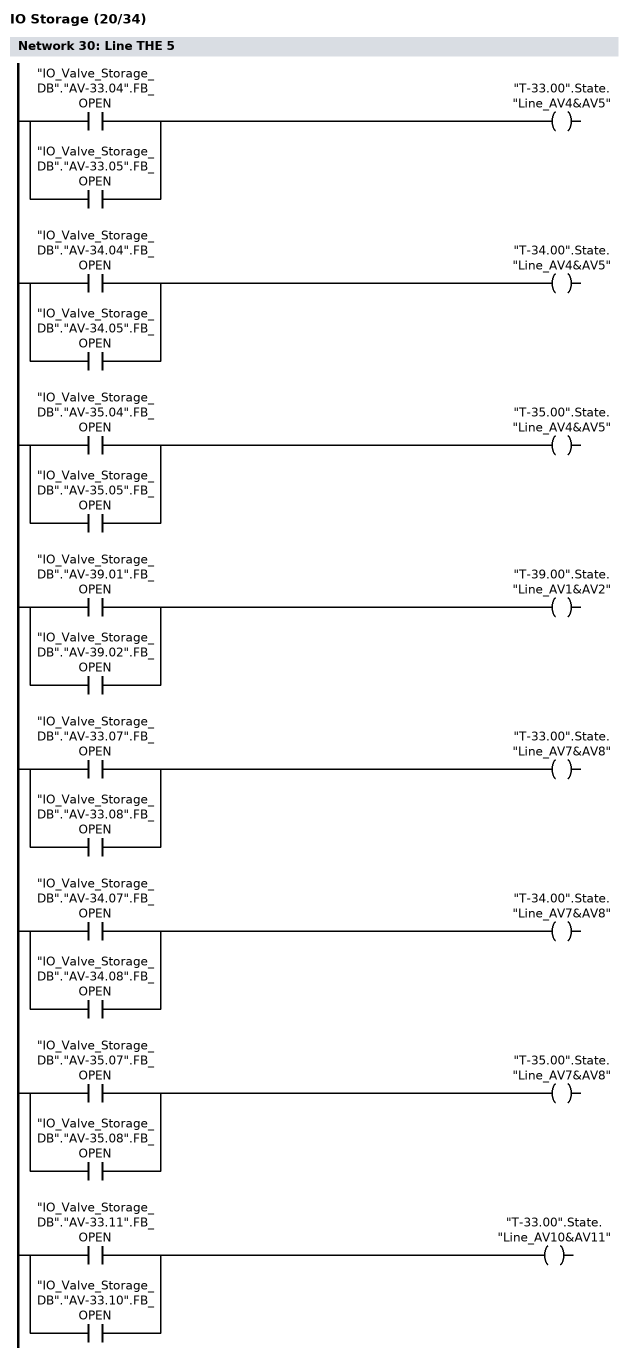
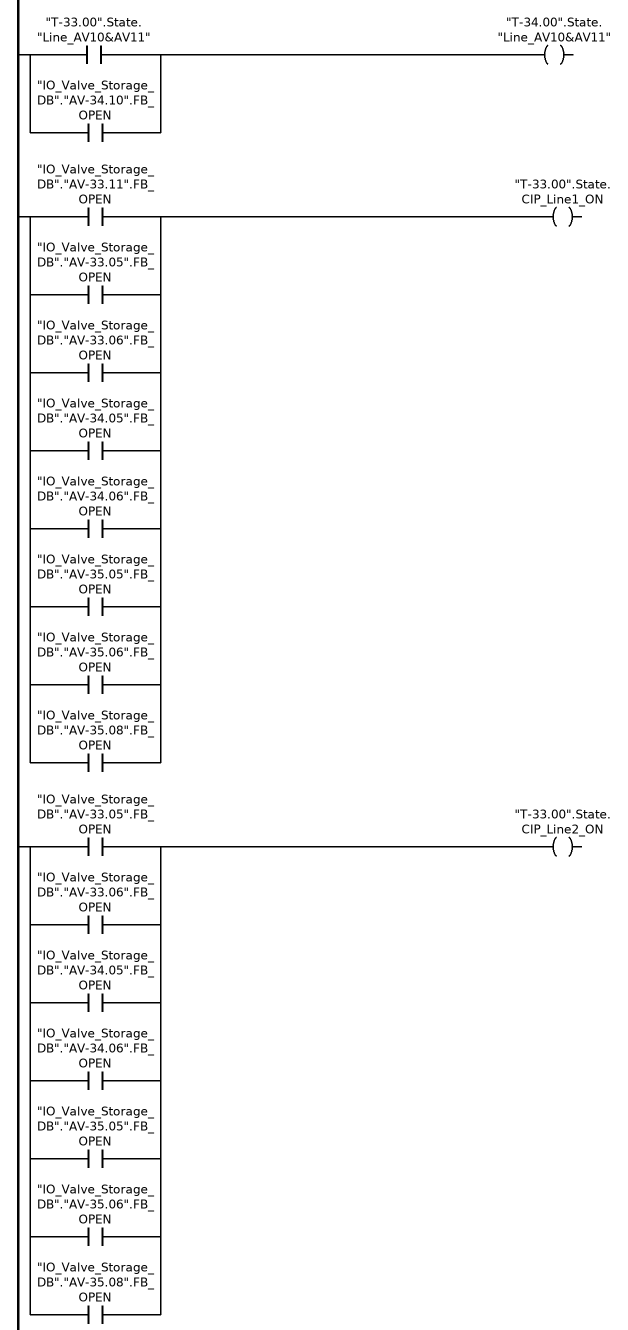
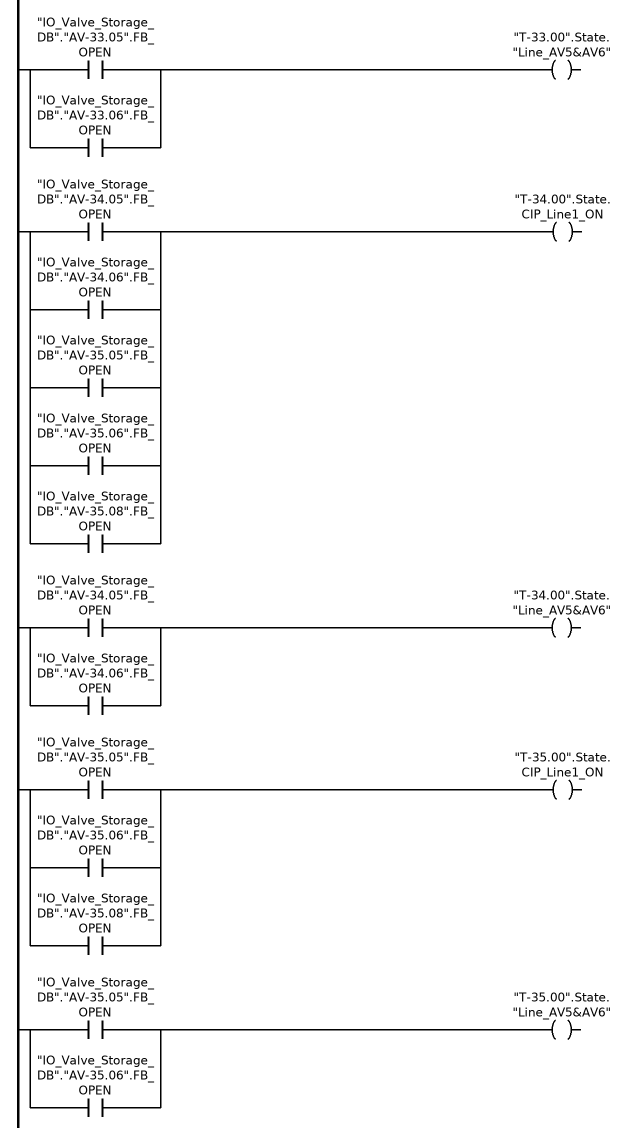
   RUNG wire#powerrail
      Contact( "IO_Valve_Storage_DB"."AV-33.04".FB_OPEN )
      wire#w1
      Coil( "T-33.00".State."Line_AV4&AV5" )
   END_RUNG
   RUNG wire#powerrail
      Contact( "IO_Valve_Storage_DB"."AV-33.05".FB_OPEN )
   END_RUNG wire#w1
   RUNG wire#powerrail
      Contact( "IO_Valve_Storage_DB"."AV-34.04".FB_OPEN )
      wire#w2
      Coil( "T-34.00".State."Line_AV4&AV5" )
   END_RUNG
   RUNG wire#powerrail
      Contact( "IO_Valve_Storage_DB"."AV-34.05".FB_OPEN )
   END_RUNG wire#w2
   RUNG wire#powerrail
      Contact( "IO_Valve_Storage_DB"."AV-35.04".FB_OPEN )
      wire#w3
      Coil( "T-35.00".State."Line_AV4&AV5" )
   END_RUNG
   RUNG wire#powerrail
      Contact( "IO_Valve_Storage_DB"."AV-35.05".FB_OPEN )
   END_RUNG wire#w3
   RUNG wire#powerrail
      Contact( "IO_Valve_Storage_DB"."AV-39.01".FB_OPEN )
      wire#w4
      Coil( "T-39.00".State."Line_AV1&AV2" )
   END_RUNG
   RUNG wire#powerrail
      Contact( "IO_Valve_Storage_DB"."AV-39.02".FB_OPEN )
   END_RUNG wire#w4
   RUNG wire#powerrail
      Contact( "IO_Valve_Storage_DB"."AV-33.07".FB_OPEN )
      wire#w5
      Coil( "T-33.00".State."Line_AV7&AV8" )
   END_RUNG
   RUNG wire#powerrail
      Contact( "IO_Valve_Storage_DB"."AV-33.08".FB_OPEN )
   END_RUNG wire#w5
   RUNG wire#powerrail
      Contact( "IO_Valve_Storage_DB"."AV-34.07".FB_OPEN )
      wire#w6
      Coil( "T-34.00".State."Line_AV7&AV8" )
   END_RUNG
   RUNG wire#powerrail
      Contact( "IO_Valve_Storage_DB"."AV-34.08".FB_OPEN )
   END_RUNG wire#w6
   RUNG wire#powerrail
      Contact( "IO_Valve_Storage_DB"."AV-35.07".FB_OPEN )
      wire#w7
      Coil( "T-35.00".State."Line_AV7&AV8" )
   END_RUNG
   RUNG wire#powerrail
      Contact( "IO_Valve_Storage_DB"."AV-35.08".FB_OPEN )
   END_RUNG wire#w7
   RUNG wire#powerrail
      Contact( "IO_Valve_Storage_DB"."AV-33.11".FB_OPEN )
      wire#w8
      Coil( "T-33.00".State."Line_AV10&AV11" )
   END_RUNG
   RUNG wire#powerrail
      Contact( "IO_Valve_Storage_DB"."AV-33.10".FB_OPEN )
   END_RUNG wire#w8
   RUNG wire#powerrail
      Contact( "T-33.00".State."Line_AV10&AV11" )
      wire#w9
      Coil( "T-34.00".State."Line_AV10&AV11" )
   END_RUNG
   RUNG wire#powerrail
      Contact( "IO_Valve_Storage_DB"."AV-34.10".FB_OPEN )
   END_RUNG wire#w9
   RUNG wire#powerrail
      Contact( "IO_Valve_Storage_DB"."AV-33.11".FB_OPEN )
      wire#w10
      Coil( "T-33.00".State.CIP_Line1_ON )
   END_RUNG
   RUNG wire#powerrail
      Contact( "IO_Valve_Storage_DB"."AV-33.05".FB_OPEN )
   END_RUNG wire#w10
   RUNG wire#powerrail
      Contact( "IO_Valve_Storage_DB"."AV-33.06".FB_OPEN )
   END_RUNG wire#w10
   RUNG wire#powerrail
      Contact( "IO_Valve_Storage_DB"."AV-34.05".FB_OPEN )
   END_RUNG wire#w10
   RUNG wire#powerrail
      Contact( "IO_Valve_Storage_DB"."AV-34.06".FB_OPEN )
   END_RUNG wire#w10
   RUNG wire#powerrail
      Contact( "IO_Valve_Storage_DB"."AV-35.05".FB_OPEN )
   END_RUNG wire#w10
   RUNG wire#powerrail
      Contact( "IO_Valve_Storage_DB"."AV-35.06".FB_OPEN )
   END_RUNG wire#w10
   RUNG wire#powerrail
      Contact( "IO_Valve_Storage_DB"."AV-35.08".FB_OPEN )
   END_RUNG wire#w10
   RUNG wire#powerrail
      Contact( "IO_Valve_Storage_DB"."AV-33.05".FB_OPEN )
      wire#w11
      Coil( "T-33.00".State.CIP_Line2_ON )
   END_RUNG
   RUNG wire#powerrail
      Contact( "IO_Valve_Storage_DB"."AV-33.06".FB_OPEN )
   END_RUNG wire#w11
   RUNG wire#powerrail
      Contact( "IO_Valve_Storage_DB"."AV-34.05".FB_OPEN )
   END_RUNG wire#w11
   RUNG wire#powerrail
      Contact( "IO_Valve_Storage_DB"."AV-34.06".FB_OPEN )
   END_RUNG wire#w11
   RUNG wire#powerrail
      Contact( "IO_Valve_Storage_DB"."AV-35.05".FB_OPEN )
   END_RUNG wire#w11
   RUNG wire#powerrail
      Contact( "IO_Valve_Storage_DB"."AV-35.06".FB_OPEN )
   END_RUNG wire#w11
   RUNG wire#powerrail
      Contact( "IO_Valve_Storage_DB"."AV-35.08".FB_OPEN )
   END_RUNG wire#w11
   RUNG wire#powerrail
      Contact( "IO_Valve_Storage_DB"."AV-33.05".FB_OPEN )
      wire#w12
      Coil( "T-33.00".State."Line_AV5&AV6" )
   END_RUNG
   RUNG wire#powerrail
      Contact( "IO_Valve_Storage_DB"."AV-33.06".FB_OPEN )
   END_RUNG wire#w12
   RUNG wire#powerrail
      Contact( "IO_Valve_Storage_DB"."AV-34.05".FB_OPEN )
      wire#w13
      Coil( "T-34.00".State.CIP_Line1_ON )
   END_RUNG
   RUNG wire#powerrail
      Contact( "IO_Valve_Storage_DB"."AV-34.06".FB_OPEN )
   END_RUNG wire#w13
   RUNG wire#powerrail
      Contact( "IO_Valve_Storage_DB"."AV-35.05".FB_OPEN )
   END_RUNG wire#w13
   RUNG wire#powerrail
      Contact( "IO_Valve_Storage_DB"."AV-35.06".FB_OPEN )
   END_RUNG wire#w13
   RUNG wire#powerrail
      Contact( "IO_Valve_Storage_DB"."AV-35.08".FB_OPEN )
   END_RUNG wire#w13
   RUNG wire#powerrail
      Contact( "IO_Valve_Storage_DB"."AV-34.05".FB_OPEN )
      wire#w14
      Coil( "T-34.00".State."Line_AV5&AV6" )
   END_RUNG
   RUNG wire#powerrail
      Contact( "IO_Valve_Storage_DB"."AV-34.06".FB_OPEN )
   END_RUNG wire#w14
   RUNG wire#powerrail
      Contact( "IO_Valve_Storage_DB"."AV-35.05".FB_OPEN )
      wire#w15
      Coil( "T-35.00".State.CIP_Line1_ON )
   END_RUNG
   RUNG wire#powerrail
      Contact( "IO_Valve_Storage_DB"."AV-35.06".FB_OPEN )
   END_RUNG wire#w15
   RUNG wire#powerrail
      Contact( "IO_Valve_Storage_DB"."AV-35.08".FB_OPEN )
   END_RUNG wire#w15
   RUNG wire#powerrail
      Contact( "IO_Valve_Storage_DB"."AV-35.05".FB_OPEN )
      wire#w16
      Coil( "T-35.00".State."Line_AV5&AV6" )
   END_RUNG
   RUNG wire#powerrail
      Contact( "IO_Valve_Storage_DB"."AV-35.06".FB_OPEN )
   END_RUNG wire#w16
   // the same network as SCL:
   "T-33.00".State."Line_AV4&AV5" := "IO_Valve_Storage_DB"."AV-33.04".FB_OPEN OR "IO_Valve_Storage_DB"."AV-33.05".FB_OPEN;
   "T-34.00".State."Line_AV4&AV5" := "IO_Valve_Storage_DB"."AV-34.04".FB_OPEN OR "IO_Valve_Storage_DB"."AV-34.05".FB_OPEN;
   "T-35.00".State."Line_AV4&AV5" := "IO_Valve_Storage_DB"."AV-35.04".FB_OPEN OR "IO_Valve_Storage_DB"."AV-35.05".FB_OPEN;
   "T-39.00".State."Line_AV1&AV2" := "IO_Valve_Storage_DB"."AV-39.01".FB_OPEN OR "IO_Valve_Storage_DB"."AV-39.02".FB_OPEN;
   "T-33.00".State."Line_AV7&AV8" := "IO_Valve_Storage_DB"."AV-33.07".FB_OPEN OR "IO_Valve_Storage_DB"."AV-33.08".FB_OPEN;
   "T-34.00".State."Line_AV7&AV8" := "IO_Valve_Storage_DB"."AV-34.07".FB_OPEN OR "IO_Valve_Storage_DB"."AV-34.08".FB_OPEN;
   "T-35.00".State."Line_AV7&AV8" := "IO_Valve_Storage_DB"."AV-35.07".FB_OPEN OR "IO_Valve_Storage_DB"."AV-35.08".FB_OPEN;
   "T-33.00".State."Line_AV10&AV11" := "IO_Valve_Storage_DB"."AV-33.11".FB_OPEN OR "IO_Valve_Storage_DB"."AV-33.10".FB_OPEN;
   "T-34.00".State."Line_AV10&AV11" := "T-33.00".State."Line_AV10&AV11" OR "IO_Valve_Storage_DB"."AV-34.10".FB_OPEN;
   "T-33.00".State.CIP_Line1_ON := "IO_Valve_Storage_DB"."AV-33.11".FB_OPEN OR "IO_Valve_Storage_DB"."AV-33.05".FB_OPEN OR "IO_Valve_Storage_DB"."AV-33.06".FB_OPEN OR "IO_Valve_Storage_DB"."AV-34.05".FB_OPEN OR "IO_Valve_Storage_DB"."AV-34.06".FB_OPEN OR "IO_Valve_Storage_DB"."AV-35.05".FB_OPEN OR "IO_Valve_Storage_DB"."AV-35.06".FB_OPEN OR "IO_Valve_Storage_DB"."AV-35.08".FB_OPEN;
   "T-33.00".State.CIP_Line2_ON := "IO_Valve_Storage_DB"."AV-33.05".FB_OPEN OR "IO_Valve_Storage_DB"."AV-33.06".FB_OPEN OR "IO_Valve_Storage_DB"."AV-34.05".FB_OPEN OR "IO_Valve_Storage_DB"."AV-34.06".FB_OPEN OR "IO_Valve_Storage_DB"."AV-35.05".FB_OPEN OR "IO_Valve_Storage_DB"."AV-35.06".FB_OPEN OR "IO_Valve_Storage_DB"."AV-35.08".FB_OPEN;
   "T-33.00".State."Line_AV5&AV6" := "IO_Valve_Storage_DB"."AV-33.05".FB_OPEN OR "IO_Valve_Storage_DB"."AV-33.06".FB_OPEN;
   "T-34.00".State.CIP_Line1_ON := "IO_Valve_Storage_DB"."AV-34.05".FB_OPEN OR "IO_Valve_Storage_DB"."AV-34.06".FB_OPEN OR "IO_Valve_Storage_DB"."AV-35.05".FB_OPEN OR "IO_Valve_Storage_DB"."AV-35.06".FB_OPEN OR "IO_Valve_Storage_DB"."AV-35.08".FB_OPEN;
   "T-34.00".State."Line_AV5&AV6" := "IO_Valve_Storage_DB"."AV-34.05".FB_OPEN OR "IO_Valve_Storage_DB"."AV-34.06".FB_OPEN;
   "T-35.00".State.CIP_Line1_ON := "IO_Valve_Storage_DB"."AV-35.05".FB_OPEN OR "IO_Valve_Storage_DB"."AV-35.06".FB_OPEN OR "IO_Valve_Storage_DB"."AV-35.08".FB_OPEN;
   "T-35.00".State."Line_AV5&AV6" := "IO_Valve_Storage_DB"."AV-35.05".FB_OPEN OR "IO_Valve_Storage_DB"."AV-35.06".FB_OPEN;
END_REGION

REGION Network 32: T-81.00
   // Inload 1 : PHE-2
   // Inload 2 : THE-1
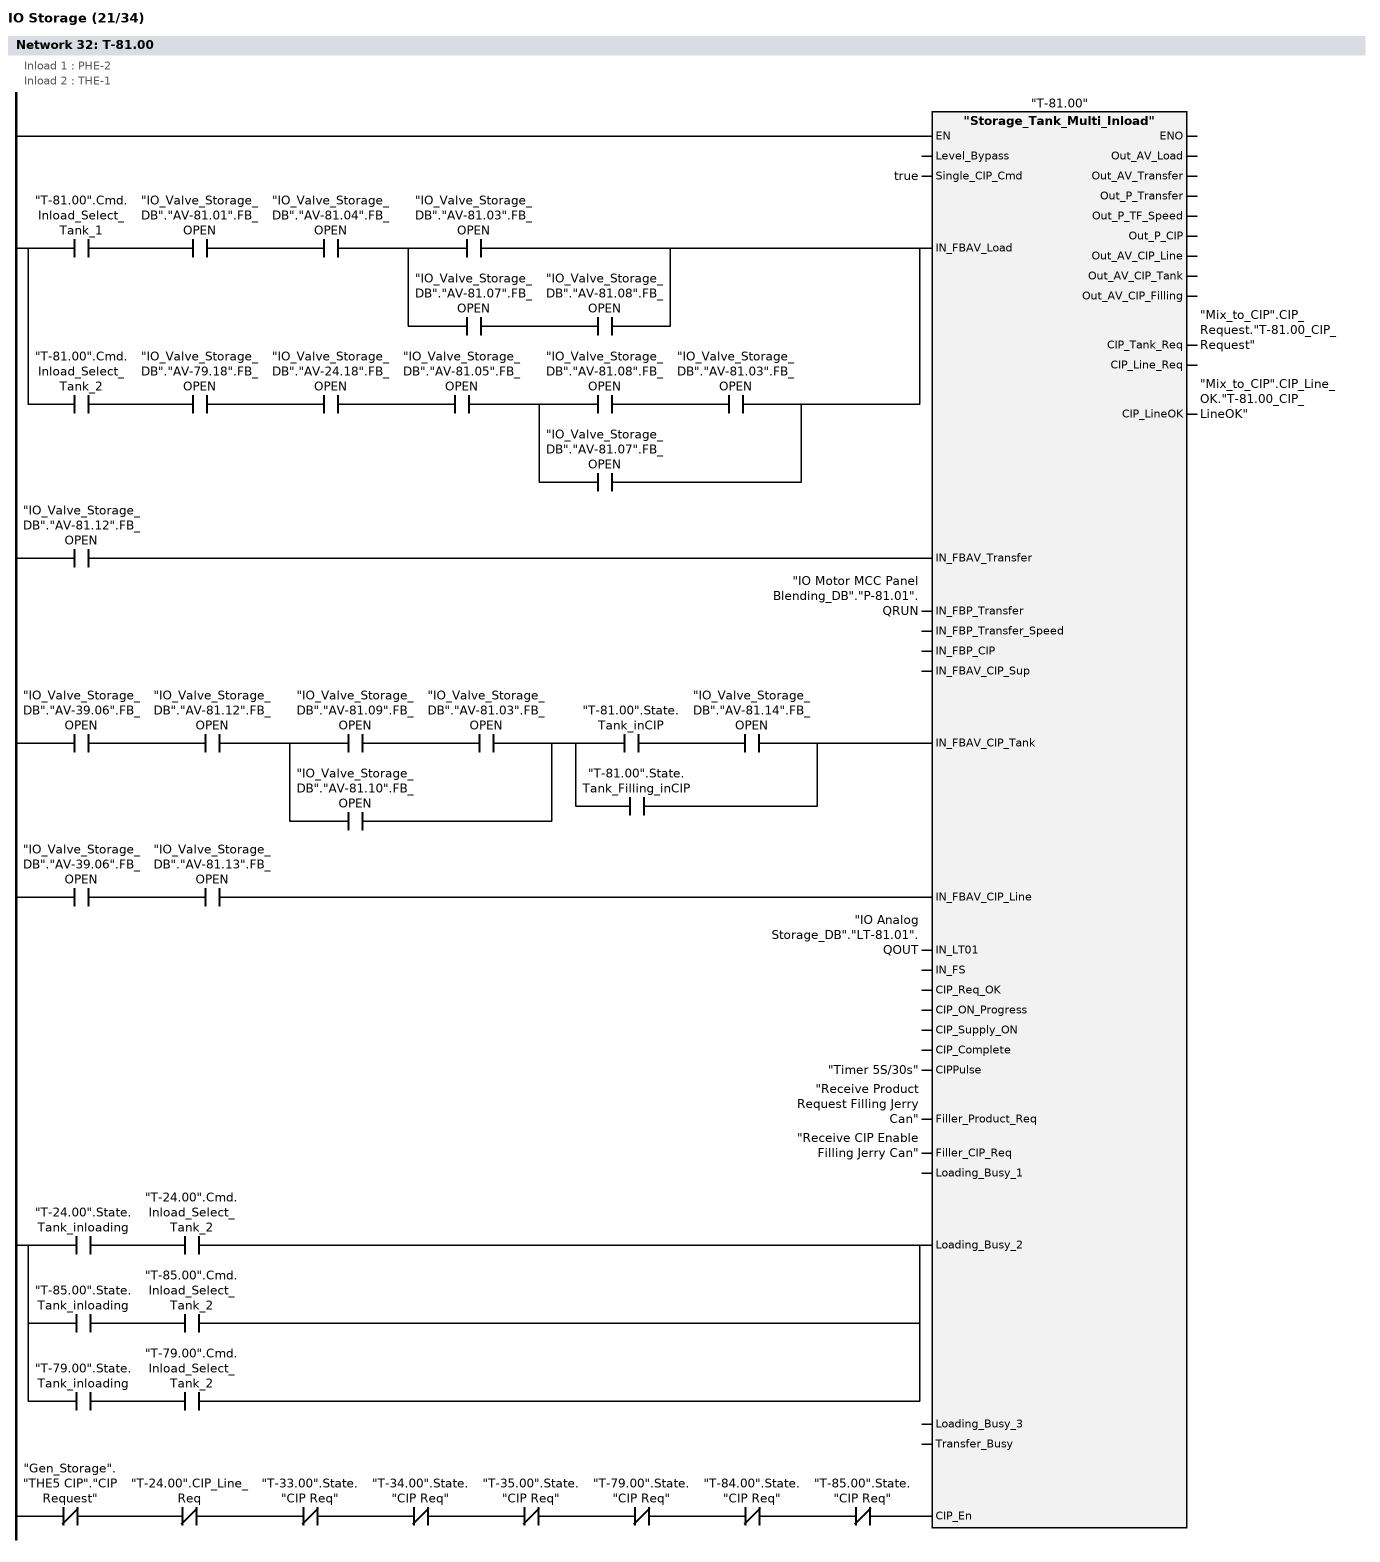
   RUNG wire#powerrail
      "T-81.00"(IN_FBAV_Load := wire#w3, IN_FBAV_Transfer := wire#w4, IN_FBAV_CIP_Tank := wire#w7, IN_FBAV_CIP_Line := wire#w8, Loading_Busy_2 := wire#w9, CIP_En := wire#w10, Level_Bypass :=, Single_CIP_Cmd := true, IN_FBP_Transfer := "IO Motor MCC Panel Blending_DB"."P-81.01".QRUN, IN_FBP_Transfer_Speed :=, IN_FBP_CIP :=, IN_FBAV_CIP_Sup :=, IN_LT01 := "IO Analog Storage_DB"."LT-81.01".QOUT, IN_FS :=, CIP_Req_OK :=, CIP_ON_Progress :=, CIP_Supply_ON :=, CIP_Complete :=, CIPPulse := "Timer 5S/30s", Filler_Product_Req := "Receive Product Request Filling Jerry Can", Filler_CIP_Req := "Receive CIP Enable Filling Jerry Can", Loading_Busy_1 :=, Loading_Busy_3 :=, Transfer_Busy :=, Out_AV_Load =>, Out_AV_Transfer =>, Out_P_Transfer =>, Out_P_TF_Speed =>, Out_P_CIP =>, Out_AV_CIP_Line =>, Out_AV_CIP_Tank =>, Out_AV_CIP_Filling =>, CIP_Tank_Req => "Mix_to_CIP".CIP_Request."T-81.00_CIP_Request", CIP_Line_Req =>, CIP_LineOK => "Mix_to_CIP".CIP_Line_OK."T-81.00_CIP_LineOK")
   END_RUNG
   RUNG wire#powerrail
      Contact( "T-81.00".Cmd.Inload_Select_Tank_1 )
      Contact( "IO_Valve_Storage_DB"."AV-81.01".FB_OPEN )
      Contact( "IO_Valve_Storage_DB"."AV-81.04".FB_OPEN )
      wire#w1
      Contact( "IO_Valve_Storage_DB"."AV-81.03".FB_OPEN )
   END_RUNG wire#w3
   RUNG wire#w1
      Contact( "IO_Valve_Storage_DB"."AV-81.07".FB_OPEN )
      Contact( "IO_Valve_Storage_DB"."AV-81.08".FB_OPEN )
   END_RUNG wire#w3
   RUNG wire#powerrail
      Contact( "T-81.00".Cmd.Inload_Select_Tank_2 )
      Contact( "IO_Valve_Storage_DB"."AV-79.18".FB_OPEN )
      Contact( "IO_Valve_Storage_DB"."AV-24.18".FB_OPEN )
      Contact( "IO_Valve_Storage_DB"."AV-81.05".FB_OPEN )
      wire#w2
      Contact( "IO_Valve_Storage_DB"."AV-81.08".FB_OPEN )
      Contact( "IO_Valve_Storage_DB"."AV-81.03".FB_OPEN )
   END_RUNG wire#w3
   RUNG wire#w2
      Contact( "IO_Valve_Storage_DB"."AV-81.07".FB_OPEN )
   END_RUNG wire#w3
   RUNG wire#powerrail
      Contact( "IO_Valve_Storage_DB"."AV-81.12".FB_OPEN )
   END_RUNG wire#w4
   RUNG wire#powerrail
      Contact( "IO_Valve_Storage_DB"."AV-39.06".FB_OPEN )
      Contact( "IO_Valve_Storage_DB"."AV-81.12".FB_OPEN )
      wire#w5
      Contact( "IO_Valve_Storage_DB"."AV-81.09".FB_OPEN )
      Contact( "IO_Valve_Storage_DB"."AV-81.03".FB_OPEN )
      wire#w6
      Contact( "T-81.00".State.Tank_inCIP )
      Contact( "IO_Valve_Storage_DB"."AV-81.14".FB_OPEN )
   END_RUNG wire#w7
   RUNG wire#w5
      Contact( "IO_Valve_Storage_DB"."AV-81.10".FB_OPEN )
   END_RUNG wire#w6
   RUNG wire#w6
      Contact( "T-81.00".State.Tank_Filling_inCIP )
   END_RUNG wire#w7
   RUNG wire#powerrail
      Contact( "IO_Valve_Storage_DB"."AV-39.06".FB_OPEN )
      Contact( "IO_Valve_Storage_DB"."AV-81.13".FB_OPEN )
   END_RUNG wire#w8
   RUNG wire#powerrail
      Contact( "T-24.00".State.Tank_inloading )
      Contact( "T-24.00".Cmd.Inload_Select_Tank_2 )
   END_RUNG wire#w9
   RUNG wire#powerrail
      Contact( "T-85.00".State.Tank_inloading )
      Contact( "T-85.00".Cmd.Inload_Select_Tank_2 )
   END_RUNG wire#w9
   RUNG wire#powerrail
      Contact( "T-79.00".State.Tank_inloading )
      Contact( "T-79.00".Cmd.Inload_Select_Tank_2 )
   END_RUNG wire#w9
   RUNG wire#powerrail
      I_Contact( "Gen_Storage"."THE5 CIP"."CIP Request" )
      I_Contact( "T-24.00".CIP_Line_Req )
      I_Contact( "T-33.00".State."CIP Req" )
      I_Contact( "T-34.00".State."CIP Req" )
      I_Contact( "T-35.00".State."CIP Req" )
      I_Contact( "T-79.00".State."CIP Req" )
      I_Contact( "T-84.00".State."CIP Req" )
      I_Contact( "T-85.00".State."CIP Req" )
   END_RUNG wire#w10
   // the same network as SCL:
   "T-81.00"(Single_CIP_Cmd := true,   // "Storage_Tank_Multi_Inload"
             IN_FBAV_Load := ("T-81.00".Cmd.Inload_Select_Tank_1 AND "IO_Valve_Storage_DB"."AV-81.01".FB_OPEN AND "IO_Valve_Storage_DB"."AV-81.04".FB_OPEN AND ("IO_Valve_Storage_DB"."AV-81.03".FB_OPEN OR ("IO_Valve_Storage_DB"."AV-81.07".FB_OPEN AND "IO_Valve_Storage_DB"."AV-81.08".FB_OPEN))) OR ("T-81.00".Cmd.Inload_Select_Tank_2 AND "IO_Valve_Storage_DB"."AV-79.18".FB_OPEN AND "IO_Valve_Storage_DB"."AV-24.18".FB_OPEN AND "IO_Valve_Storage_DB"."AV-81.05".FB_OPEN AND (("IO_Valve_Storage_DB"."AV-81.08".FB_OPEN AND "IO_Valve_Storage_DB"."AV-81.03".FB_OPEN) OR "IO_Valve_Storage_DB"."AV-81.07".FB_OPEN)),
             IN_FBAV_Transfer := "IO_Valve_Storage_DB"."AV-81.12".FB_OPEN,
             IN_FBP_Transfer := "IO Motor MCC Panel Blending_DB"."P-81.01".QRUN,
             IN_FBAV_CIP_Tank := "IO_Valve_Storage_DB"."AV-39.06".FB_OPEN AND "IO_Valve_Storage_DB"."AV-81.12".FB_OPEN AND (("IO_Valve_Storage_DB"."AV-81.09".FB_OPEN AND "IO_Valve_Storage_DB"."AV-81.03".FB_OPEN) OR "IO_Valve_Storage_DB"."AV-81.10".FB_OPEN) AND (("T-81.00".State.Tank_inCIP AND "IO_Valve_Storage_DB"."AV-81.14".FB_OPEN) OR "T-81.00".State.Tank_Filling_inCIP),
             IN_FBAV_CIP_Line := "IO_Valve_Storage_DB"."AV-39.06".FB_OPEN AND "IO_Valve_Storage_DB"."AV-81.13".FB_OPEN,
             IN_LT01 := "IO Analog Storage_DB"."LT-81.01".QOUT,
             CIPPulse := "Timer 5S/30s",
             Filler_Product_Req := "Receive Product Request Filling Jerry Can",
             Filler_CIP_Req := "Receive CIP Enable Filling Jerry Can",
             Loading_Busy_2 := ("T-24.00".State.Tank_inloading AND "T-24.00".Cmd.Inload_Select_Tank_2) OR ("T-85.00".State.Tank_inloading AND "T-85.00".Cmd.Inload_Select_Tank_2) OR ("T-79.00".State.Tank_inloading AND "T-79.00".Cmd.Inload_Select_Tank_2),
             CIP_En := NOT "Gen_Storage"."THE5 CIP"."CIP Request" AND NOT "T-24.00".CIP_Line_Req AND NOT "T-33.00".State."CIP Req" AND NOT "T-34.00".State."CIP Req" AND NOT "T-35.00".State."CIP Req" AND NOT "T-79.00".State."CIP Req" AND NOT "T-84.00".State."CIP Req" AND NOT "T-85.00".State."CIP Req",
             CIP_Tank_Req => "Mix_to_CIP".CIP_Request."T-81.00_CIP_Request",
             CIP_LineOK => "Mix_to_CIP".CIP_Line_OK."T-81.00_CIP_LineOK");
END_REGION

REGION Network 33: T-81 Valve
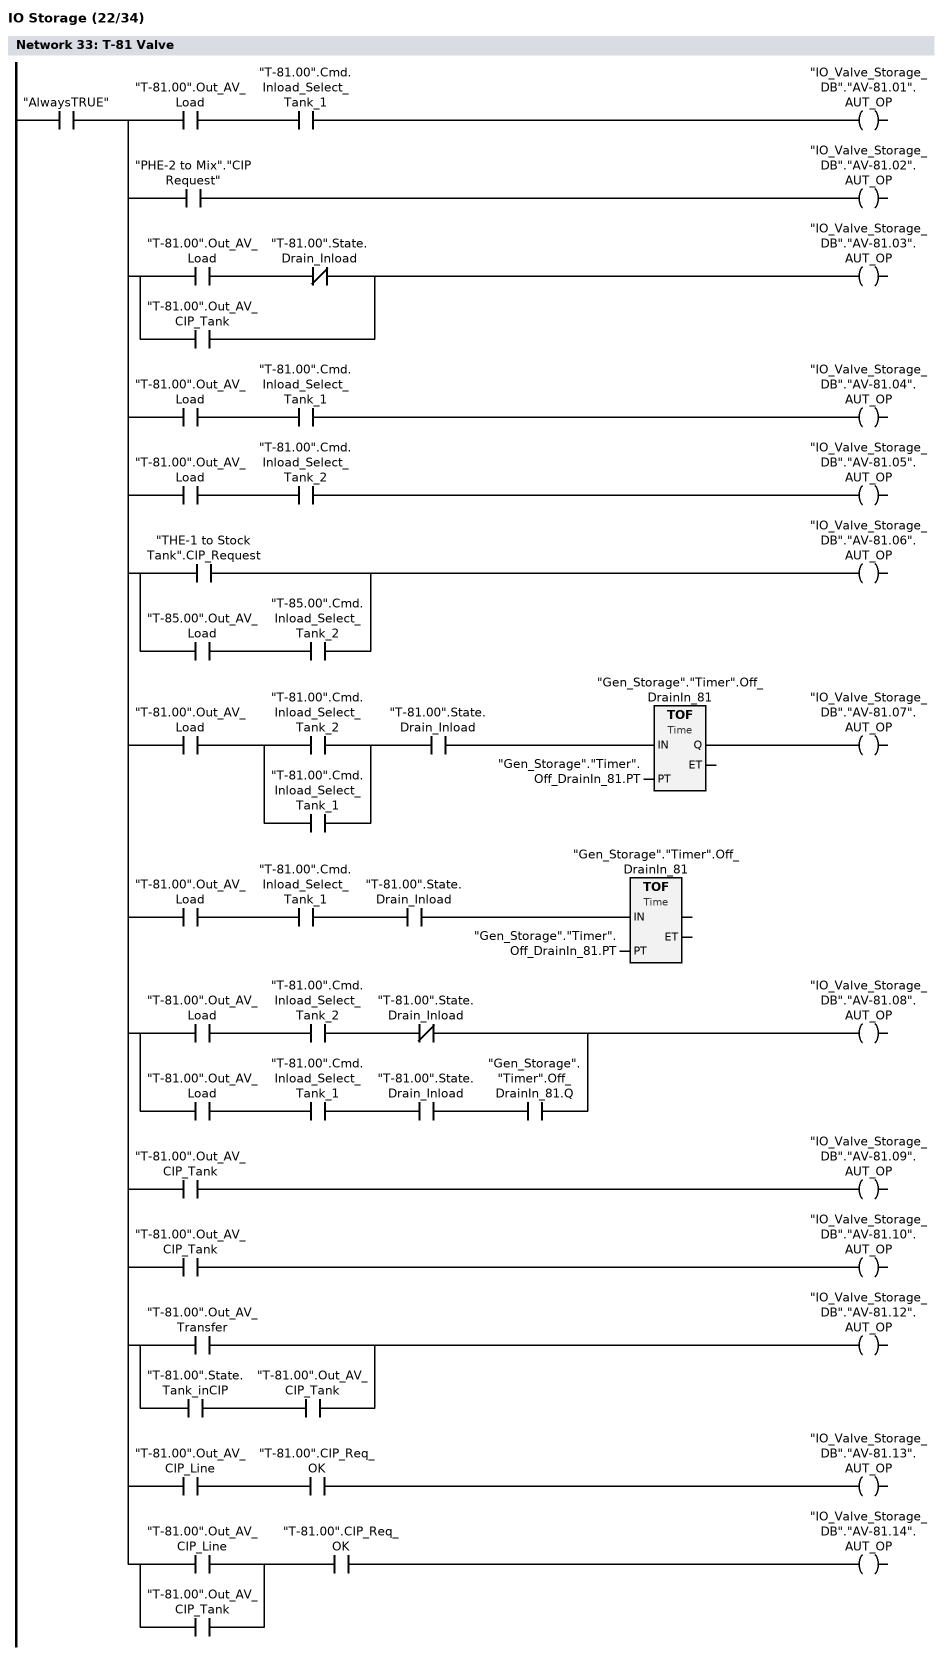
   RUNG wire#powerrail
      Contact( "AlwaysTRUE" )
      wire#w1
      Contact( "T-81.00".Out_AV_Load )
      Contact( "T-81.00".Cmd.Inload_Select_Tank_1 )
      Coil( "IO_Valve_Storage_DB"."AV-81.01".AUT_OP )
   END_RUNG
   RUNG wire#w1
      Contact( "PHE-2 to Mix"."CIP Request" )
      Coil( "IO_Valve_Storage_DB"."AV-81.02".AUT_OP )
   END_RUNG
   RUNG wire#w1
      Contact( "T-81.00".Out_AV_Load )
      I_Contact( "T-81.00".State.Drain_Inload )
      wire#w2
      Coil( "IO_Valve_Storage_DB"."AV-81.03".AUT_OP )
   END_RUNG
   RUNG wire#w1
      Contact( "T-81.00".Out_AV_CIP_Tank )
   END_RUNG wire#w2
   RUNG wire#w1
      Contact( "T-81.00".Out_AV_Load )
      Contact( "T-81.00".Cmd.Inload_Select_Tank_1 )
      Coil( "IO_Valve_Storage_DB"."AV-81.04".AUT_OP )
   END_RUNG
   RUNG wire#w1
      Contact( "T-81.00".Out_AV_Load )
      Contact( "T-81.00".Cmd.Inload_Select_Tank_2 )
      Coil( "IO_Valve_Storage_DB"."AV-81.05".AUT_OP )
   END_RUNG
   RUNG wire#w1
      Contact( "THE-1 to Stock Tank".CIP_Request )
      wire#w3
      Coil( "IO_Valve_Storage_DB"."AV-81.06".AUT_OP )
   END_RUNG
   RUNG wire#w1
      Contact( "T-85.00".Out_AV_Load )
      Contact( "T-85.00".Cmd.Inload_Select_Tank_2 )
   END_RUNG wire#w3
   RUNG wire#w1
      Contact( "T-81.00".Out_AV_Load )
      wire#w4
      Contact( "T-81.00".Cmd.Inload_Select_Tank_2 )
      wire#w5
      Contact( "T-81.00".State.Drain_Inload )
      { S7_Templates := "time_type := Time" } "Gen_Storage"."Timer".Off_DrainIn_81.TOF(pt := "Gen_Storage"."Timer".Off_DrainIn_81.PT, et =>)
      Coil( "IO_Valve_Storage_DB"."AV-81.07".AUT_OP )
   END_RUNG
   RUNG wire#w4
      Contact( "T-81.00".Cmd.Inload_Select_Tank_1 )
   END_RUNG wire#w5
   RUNG wire#w1
      Contact( "T-81.00".Out_AV_Load )
      Contact( "T-81.00".Cmd.Inload_Select_Tank_1 )
      Contact( "T-81.00".State.Drain_Inload )
      { S7_Templates := "time_type := Time" } "Gen_Storage"."Timer".Off_DrainIn_81.TOF(pt := "Gen_Storage"."Timer".Off_DrainIn_81.PT, et =>)
   END_RUNG
   RUNG wire#w1
      Contact( "T-81.00".Out_AV_Load )
      Contact( "T-81.00".Cmd.Inload_Select_Tank_2 )
      I_Contact( "T-81.00".State.Drain_Inload )
      wire#w6
      Coil( "IO_Valve_Storage_DB"."AV-81.08".AUT_OP )
   END_RUNG
   RUNG wire#w1
      Contact( "T-81.00".Out_AV_Load )
      Contact( "T-81.00".Cmd.Inload_Select_Tank_1 )
      Contact( "T-81.00".State.Drain_Inload )
      Contact( "Gen_Storage"."Timer".Off_DrainIn_81.Q )
   END_RUNG wire#w6
   RUNG wire#w1
      Contact( "T-81.00".Out_AV_CIP_Tank )
      Coil( "IO_Valve_Storage_DB"."AV-81.09".AUT_OP )
   END_RUNG
   RUNG wire#w1
      Contact( "T-81.00".Out_AV_CIP_Tank )
      Coil( "IO_Valve_Storage_DB"."AV-81.10".AUT_OP )
   END_RUNG
   RUNG wire#w1
      Contact( "T-81.00".Out_AV_Transfer )
      wire#w7
      Coil( "IO_Valve_Storage_DB"."AV-81.12".AUT_OP )
   END_RUNG
   RUNG wire#w1
      Contact( "T-81.00".State.Tank_inCIP )
      Contact( "T-81.00".Out_AV_CIP_Tank )
   END_RUNG wire#w7
   RUNG wire#w1
      Contact( "T-81.00".Out_AV_CIP_Line )
      Contact( "T-81.00".CIP_Req_OK )
      Coil( "IO_Valve_Storage_DB"."AV-81.13".AUT_OP )
   END_RUNG
   RUNG wire#w1
      Contact( "T-81.00".Out_AV_CIP_Line )
      wire#w8
      Contact( "T-81.00".CIP_Req_OK )
      Coil( "IO_Valve_Storage_DB"."AV-81.14".AUT_OP )
   END_RUNG
   RUNG wire#w1
      Contact( "T-81.00".Out_AV_CIP_Tank )
   END_RUNG wire#w8
   // the same network as SCL:
   "IO_Valve_Storage_DB"."AV-81.01".AUT_OP := "AlwaysTRUE" AND "T-81.00".Out_AV_Load AND "T-81.00".Cmd.Inload_Select_Tank_1;
   "IO_Valve_Storage_DB"."AV-81.02".AUT_OP := "AlwaysTRUE" AND "PHE-2 to Mix"."CIP Request";
   "IO_Valve_Storage_DB"."AV-81.03".AUT_OP := "AlwaysTRUE" AND (("T-81.00".Out_AV_Load AND NOT "T-81.00".State.Drain_Inload) OR "T-81.00".Out_AV_CIP_Tank);
   "IO_Valve_Storage_DB"."AV-81.04".AUT_OP := "AlwaysTRUE" AND "T-81.00".Out_AV_Load AND "T-81.00".Cmd.Inload_Select_Tank_1;
   "IO_Valve_Storage_DB"."AV-81.05".AUT_OP := "AlwaysTRUE" AND "T-81.00".Out_AV_Load AND "T-81.00".Cmd.Inload_Select_Tank_2;
   "IO_Valve_Storage_DB"."AV-81.06".AUT_OP := "AlwaysTRUE" AND ("THE-1 to Stock Tank".CIP_Request OR ("T-85.00".Out_AV_Load AND "T-85.00".Cmd.Inload_Select_Tank_2));
   "Gen_Storage"."Timer".Off_DrainIn_81.TOF(IN := "AlwaysTRUE" AND "T-81.00".Out_AV_Load AND ("T-81.00".Cmd.Inload_Select_Tank_2 OR "T-81.00".Cmd.Inload_Select_Tank_1) AND "T-81.00".State.Drain_Inload,
                           PT := "Gen_Storage"."Timer".Off_DrainIn_81.PT);
   "IO_Valve_Storage_DB"."AV-81.07".AUT_OP := "Gen_Storage"."Timer".Off_DrainIn_81.Q;
   "Gen_Storage"."Timer".Off_DrainIn_81.TOF(IN := "AlwaysTRUE" AND "T-81.00".Out_AV_Load AND "T-81.00".Cmd.Inload_Select_Tank_1 AND "T-81.00".State.Drain_Inload,
                           PT := "Gen_Storage"."Timer".Off_DrainIn_81.PT);
   "IO_Valve_Storage_DB"."AV-81.08".AUT_OP := "AlwaysTRUE" AND (("T-81.00".Out_AV_Load AND "T-81.00".Cmd.Inload_Select_Tank_2 AND NOT "T-81.00".State.Drain_Inload) OR ("T-81.00".Out_AV_Load AND "T-81.00".Cmd.Inload_Select_Tank_1 AND "T-81.00".State.Drain_Inload AND "Gen_Storage"."Timer".Off_DrainIn_81.Q));
   "IO_Valve_Storage_DB"."AV-81.09".AUT_OP := "AlwaysTRUE" AND "T-81.00".Out_AV_CIP_Tank;
   "IO_Valve_Storage_DB"."AV-81.10".AUT_OP := "AlwaysTRUE" AND "T-81.00".Out_AV_CIP_Tank;
   "IO_Valve_Storage_DB"."AV-81.12".AUT_OP := "AlwaysTRUE" AND ("T-81.00".Out_AV_Transfer OR ("T-81.00".State.Tank_inCIP AND "T-81.00".Out_AV_CIP_Tank));
   "IO_Valve_Storage_DB"."AV-81.13".AUT_OP := "AlwaysTRUE" AND "T-81.00".Out_AV_CIP_Line AND "T-81.00".CIP_Req_OK;
   "IO_Valve_Storage_DB"."AV-81.14".AUT_OP := "AlwaysTRUE" AND ("T-81.00".Out_AV_CIP_Line OR "T-81.00".Out_AV_CIP_Tank) AND "T-81.00".CIP_Req_OK;
END_REGION

REGION Network 34: Comm T-81 to THE-1
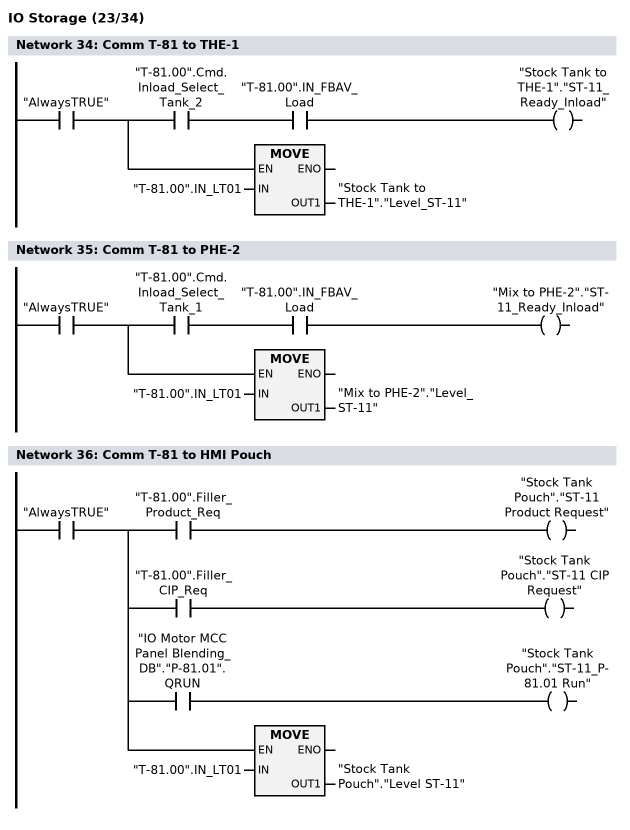
   RUNG wire#powerrail
      Contact( "AlwaysTRUE" )
      wire#w1
      Contact( "T-81.00".Cmd.Inload_Select_Tank_2 )
      Contact( "T-81.00".IN_FBAV_Load )
      Coil( "Stock Tank to THE-1"."ST-11_Ready_Inload" )
   END_RUNG
   RUNG wire#w1
      Move(in := "T-81.00".IN_LT01, out1 => "Stock Tank to THE-1"."Level_ST-11")
   END_RUNG
   // the same network as SCL:
   "Stock Tank to THE-1"."ST-11_Ready_Inload" := "AlwaysTRUE" AND "T-81.00".Cmd.Inload_Select_Tank_2 AND "T-81.00".IN_FBAV_Load;
   IF "AlwaysTRUE" THEN "Stock Tank to THE-1"."Level_ST-11" := "T-81.00".IN_LT01; END_IF;
END_REGION

REGION Network 35: Comm T-81 to PHE-2
   RUNG wire#powerrail
      Contact( "AlwaysTRUE" )
      wire#w1
      Contact( "T-81.00".Cmd.Inload_Select_Tank_1 )
      Contact( "T-81.00".IN_FBAV_Load )
      Coil( "Mix to PHE-2"."ST-11_Ready_Inload" )
   END_RUNG
   RUNG wire#w1
      Move(in := "T-81.00".IN_LT01, out1 => "Mix to PHE-2"."Level_ST-11")
   END_RUNG
   // the same network as SCL:
   "Mix to PHE-2"."ST-11_Ready_Inload" := "AlwaysTRUE" AND "T-81.00".Cmd.Inload_Select_Tank_1 AND "T-81.00".IN_FBAV_Load;
   IF "AlwaysTRUE" THEN "Mix to PHE-2"."Level_ST-11" := "T-81.00".IN_LT01; END_IF;
END_REGION

REGION Network 36: Comm T-81 to HMI Pouch
   RUNG wire#powerrail
      Contact( "AlwaysTRUE" )
      wire#w1
      Contact( "T-81.00".Filler_Product_Req )
      Coil( "Stock Tank Pouch"."ST-11 Product Request" )
   END_RUNG
   RUNG wire#w1
      Contact( "T-81.00".Filler_CIP_Req )
      Coil( "Stock Tank Pouch"."ST-11 CIP Request" )
   END_RUNG
   RUNG wire#w1
      Contact( "IO Motor MCC Panel Blending_DB"."P-81.01".QRUN )
      Coil( "Stock Tank Pouch"."ST-11_P-81.01 Run" )
   END_RUNG
   RUNG wire#w1
      Move(in := "T-81.00".IN_LT01, out1 => "Stock Tank Pouch"."Level ST-11")
   END_RUNG
   // the same network as SCL:
   "Stock Tank Pouch"."ST-11 Product Request" := "AlwaysTRUE" AND "T-81.00".Filler_Product_Req;
   "Stock Tank Pouch"."ST-11 CIP Request" := "AlwaysTRUE" AND "T-81.00".Filler_CIP_Req;
   "Stock Tank Pouch"."ST-11_P-81.01 Run" := "AlwaysTRUE" AND "IO Motor MCC Panel Blending_DB"."P-81.01".QRUN;
   IF "AlwaysTRUE" THEN "Stock Tank Pouch"."Level ST-11" := "T-81.00".IN_LT01; END_IF;
END_REGION

REGION Network 38: T-85.00 ST-16
   // Inload 1 : PHE-1
   // Inload 2 : THE-1
   // Inload 3 : THE-3
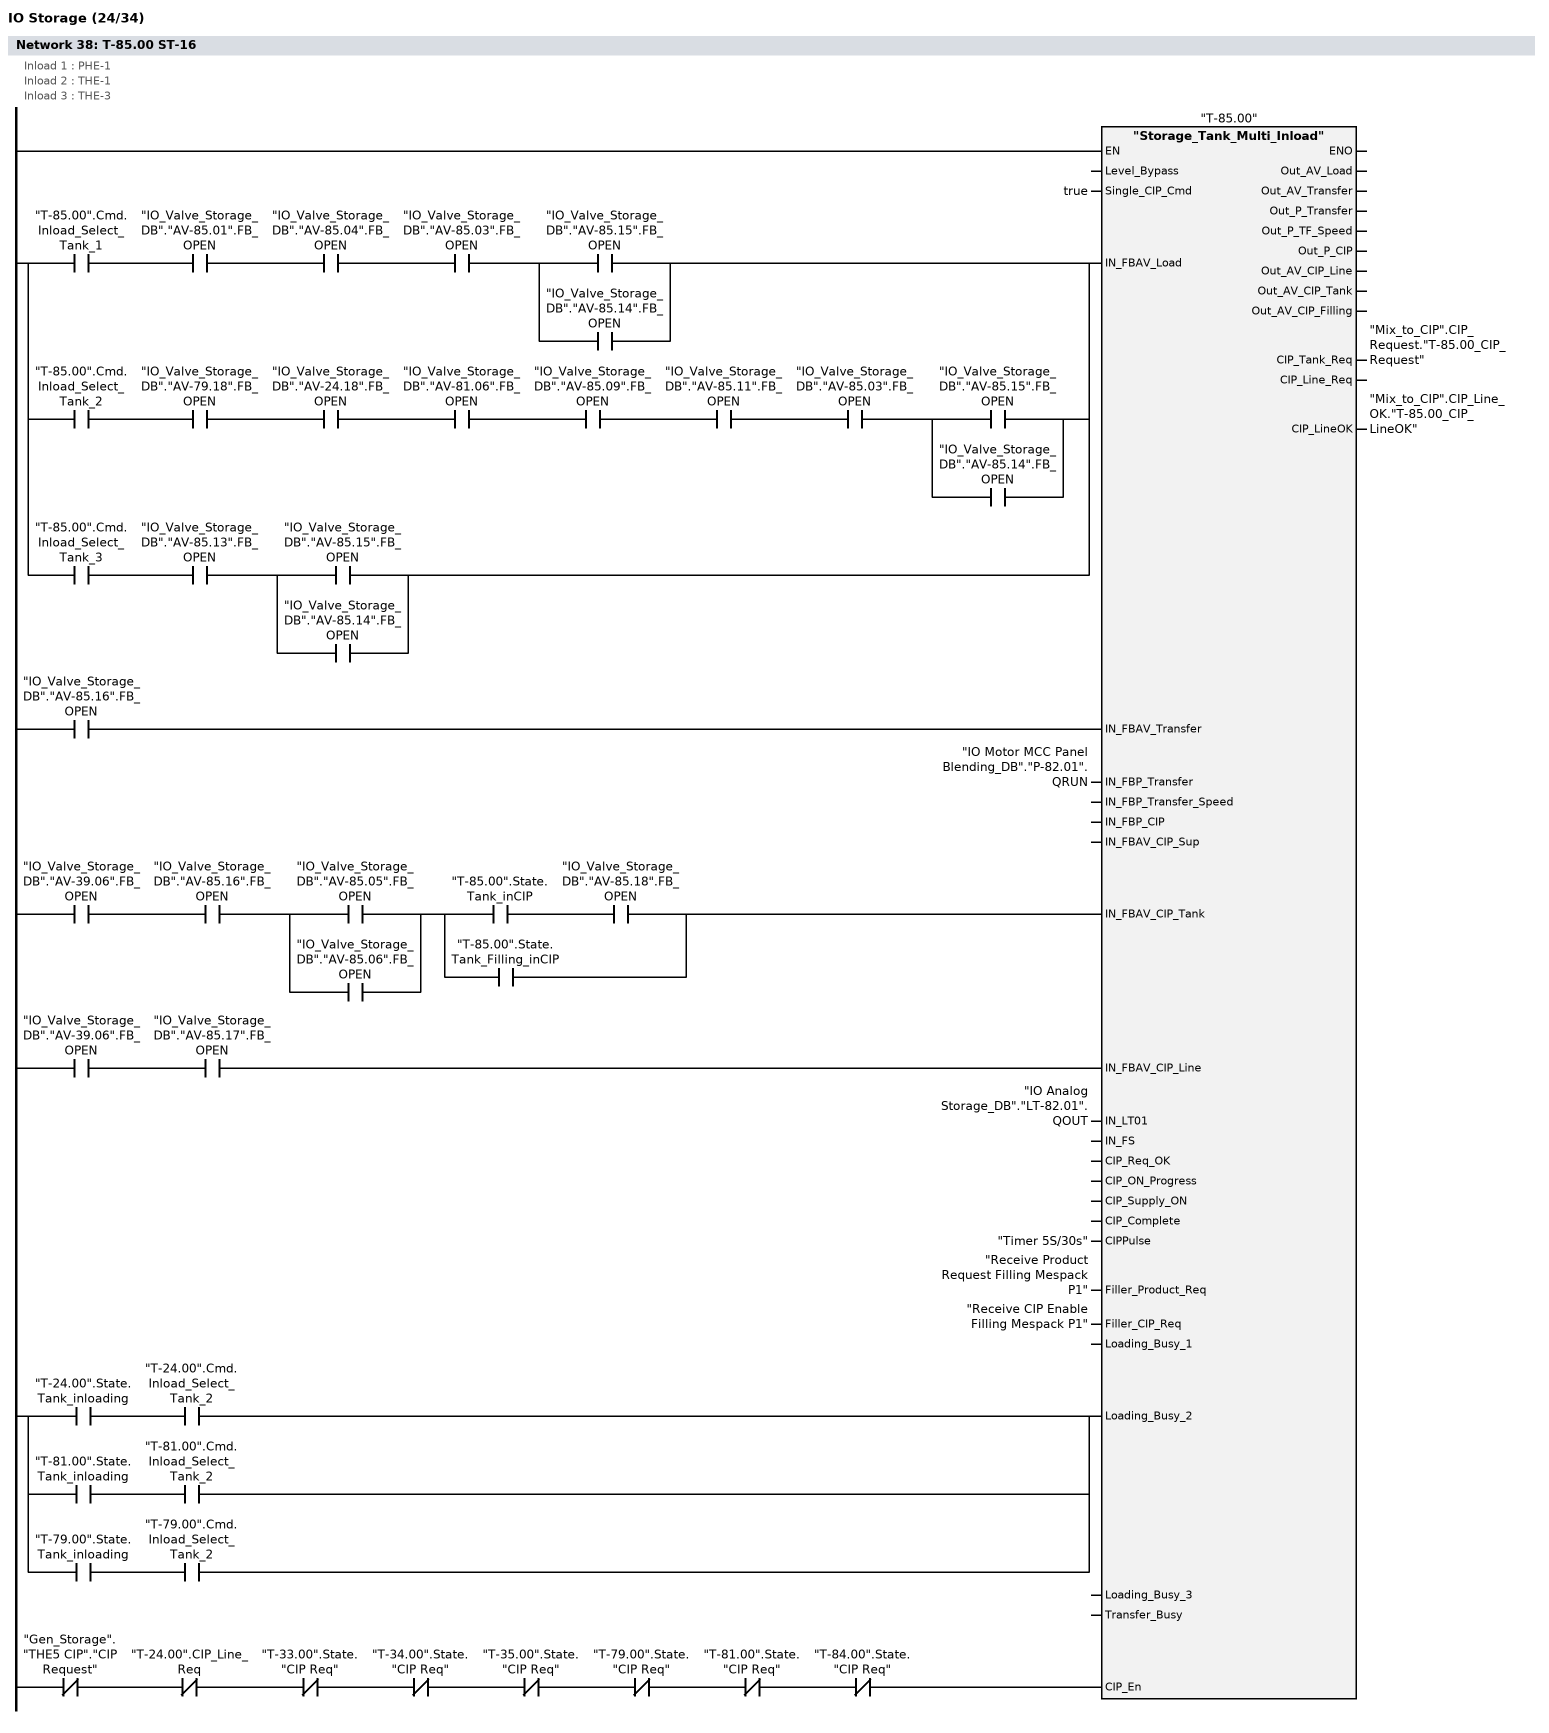
   RUNG wire#powerrail
      "T-85.00"(IN_FBAV_Load := wire#w4, IN_FBAV_Transfer := wire#w5, IN_FBAV_CIP_Tank := wire#w8, IN_FBAV_CIP_Line := wire#w9, Loading_Busy_2 := wire#w10, CIP_En := wire#w11, Level_Bypass :=, Single_CIP_Cmd := true, IN_FBP_Transfer := "IO Motor MCC Panel Blending_DB"."P-82.01".QRUN, IN_FBP_Transfer_Speed :=, IN_FBP_CIP :=, IN_FBAV_CIP_Sup :=, IN_LT01 := "IO Analog Storage_DB"."LT-82.01".QOUT, IN_FS :=, CIP_Req_OK :=, CIP_ON_Progress :=, CIP_Supply_ON :=, CIP_Complete :=, CIPPulse := "Timer 5S/30s", Filler_Product_Req := "Receive Product Request Filling Mespack P1", Filler_CIP_Req := "Receive CIP Enable Filling Mespack P1", Loading_Busy_1 :=, Loading_Busy_3 :=, Transfer_Busy :=, Out_AV_Load =>, Out_AV_Transfer =>, Out_P_Transfer =>, Out_P_TF_Speed =>, Out_P_CIP =>, Out_AV_CIP_Line =>, Out_AV_CIP_Tank =>, Out_AV_CIP_Filling =>, CIP_Tank_Req => "Mix_to_CIP".CIP_Request."T-85.00_CIP_Request", CIP_Line_Req =>, CIP_LineOK => "Mix_to_CIP".CIP_Line_OK."T-85.00_CIP_LineOK")
   END_RUNG
   RUNG wire#powerrail
      Contact( "T-85.00".Cmd.Inload_Select_Tank_1 )
      Contact( "IO_Valve_Storage_DB"."AV-85.01".FB_OPEN )
      Contact( "IO_Valve_Storage_DB"."AV-85.04".FB_OPEN )
      Contact( "IO_Valve_Storage_DB"."AV-85.03".FB_OPEN )
      wire#w1
      Contact( "IO_Valve_Storage_DB"."AV-85.15".FB_OPEN )
   END_RUNG wire#w4
   RUNG wire#w1
      Contact( "IO_Valve_Storage_DB"."AV-85.14".FB_OPEN )
   END_RUNG wire#w4
   RUNG wire#powerrail
      Contact( "T-85.00".Cmd.Inload_Select_Tank_2 )
      Contact( "IO_Valve_Storage_DB"."AV-79.18".FB_OPEN )
      Contact( "IO_Valve_Storage_DB"."AV-24.18".FB_OPEN )
      Contact( "IO_Valve_Storage_DB"."AV-81.06".FB_OPEN )
      Contact( "IO_Valve_Storage_DB"."AV-85.09".FB_OPEN )
      Contact( "IO_Valve_Storage_DB"."AV-85.11".FB_OPEN )
      Contact( "IO_Valve_Storage_DB"."AV-85.03".FB_OPEN )
      wire#w2
      Contact( "IO_Valve_Storage_DB"."AV-85.15".FB_OPEN )
   END_RUNG wire#w4
   RUNG wire#w2
      Contact( "IO_Valve_Storage_DB"."AV-85.14".FB_OPEN )
   END_RUNG wire#w4
   RUNG wire#powerrail
      Contact( "T-85.00".Cmd.Inload_Select_Tank_3 )
      Contact( "IO_Valve_Storage_DB"."AV-85.13".FB_OPEN )
      wire#w3
      Contact( "IO_Valve_Storage_DB"."AV-85.15".FB_OPEN )
   END_RUNG wire#w4
   RUNG wire#w3
      Contact( "IO_Valve_Storage_DB"."AV-85.14".FB_OPEN )
   END_RUNG wire#w4
   RUNG wire#powerrail
      Contact( "IO_Valve_Storage_DB"."AV-85.16".FB_OPEN )
   END_RUNG wire#w5
   RUNG wire#powerrail
      Contact( "IO_Valve_Storage_DB"."AV-39.06".FB_OPEN )
      Contact( "IO_Valve_Storage_DB"."AV-85.16".FB_OPEN )
      wire#w6
      Contact( "IO_Valve_Storage_DB"."AV-85.05".FB_OPEN )
      wire#w7
      Contact( "T-85.00".State.Tank_inCIP )
      Contact( "IO_Valve_Storage_DB"."AV-85.18".FB_OPEN )
   END_RUNG wire#w8
   RUNG wire#w6
      Contact( "IO_Valve_Storage_DB"."AV-85.06".FB_OPEN )
   END_RUNG wire#w7
   RUNG wire#w7
      Contact( "T-85.00".State.Tank_Filling_inCIP )
   END_RUNG wire#w8
   RUNG wire#powerrail
      Contact( "IO_Valve_Storage_DB"."AV-39.06".FB_OPEN )
      Contact( "IO_Valve_Storage_DB"."AV-85.17".FB_OPEN )
   END_RUNG wire#w9
   RUNG wire#powerrail
      Contact( "T-24.00".State.Tank_inloading )
      Contact( "T-24.00".Cmd.Inload_Select_Tank_2 )
   END_RUNG wire#w10
   RUNG wire#powerrail
      Contact( "T-81.00".State.Tank_inloading )
      Contact( "T-81.00".Cmd.Inload_Select_Tank_2 )
   END_RUNG wire#w10
   RUNG wire#powerrail
      Contact( "T-79.00".State.Tank_inloading )
      Contact( "T-79.00".Cmd.Inload_Select_Tank_2 )
   END_RUNG wire#w10
   RUNG wire#powerrail
      I_Contact( "Gen_Storage"."THE5 CIP"."CIP Request" )
      I_Contact( "T-24.00".CIP_Line_Req )
      I_Contact( "T-33.00".State."CIP Req" )
      I_Contact( "T-34.00".State."CIP Req" )
      I_Contact( "T-35.00".State."CIP Req" )
      I_Contact( "T-79.00".State."CIP Req" )
      I_Contact( "T-81.00".State."CIP Req" )
      I_Contact( "T-84.00".State."CIP Req" )
   END_RUNG wire#w11
   // the same network as SCL:
   "T-85.00"(Single_CIP_Cmd := true,   // "Storage_Tank_Multi_Inload"
             IN_FBAV_Load := ("T-85.00".Cmd.Inload_Select_Tank_1 AND "IO_Valve_Storage_DB"."AV-85.01".FB_OPEN AND "IO_Valve_Storage_DB"."AV-85.04".FB_OPEN AND "IO_Valve_Storage_DB"."AV-85.03".FB_OPEN AND ("IO_Valve_Storage_DB"."AV-85.15".FB_OPEN OR "IO_Valve_Storage_DB"."AV-85.14".FB_OPEN)) OR ("T-85.00".Cmd.Inload_Select_Tank_2 AND "IO_Valve_Storage_DB"."AV-79.18".FB_OPEN AND "IO_Valve_Storage_DB"."AV-24.18".FB_OPEN AND "IO_Valve_Storage_DB"."AV-81.06".FB_OPEN AND "IO_Valve_Storage_DB"."AV-85.09".FB_OPEN AND "IO_Valve_Storage_DB"."AV-85.11".FB_OPEN AND "IO_Valve_Storage_DB"."AV-85.03".FB_OPEN AND ("IO_Valve_Storage_DB"."AV-85.15".FB_OPEN OR "IO_Valve_Storage_DB"."AV-85.14".FB_OPEN)) OR ("T-85.00".Cmd.Inload_Select_Tank_3 AND "IO_Valve_Storage_DB"."AV-85.13".FB_OPEN AND ("IO_Valve_Storage_DB"."AV-85.15".FB_OPEN OR "IO_Valve_Storage_DB"."AV-85.14".FB_OPEN)),
             IN_FBAV_Transfer := "IO_Valve_Storage_DB"."AV-85.16".FB_OPEN,
             IN_FBP_Transfer := "IO Motor MCC Panel Blending_DB"."P-82.01".QRUN,
             IN_FBAV_CIP_Tank := "IO_Valve_Storage_DB"."AV-39.06".FB_OPEN AND "IO_Valve_Storage_DB"."AV-85.16".FB_OPEN AND ("IO_Valve_Storage_DB"."AV-85.05".FB_OPEN OR "IO_Valve_Storage_DB"."AV-85.06".FB_OPEN) AND (("T-85.00".State.Tank_inCIP AND "IO_Valve_Storage_DB"."AV-85.18".FB_OPEN) OR "T-85.00".State.Tank_Filling_inCIP),
             IN_FBAV_CIP_Line := "IO_Valve_Storage_DB"."AV-39.06".FB_OPEN AND "IO_Valve_Storage_DB"."AV-85.17".FB_OPEN,
             IN_LT01 := "IO Analog Storage_DB"."LT-82.01".QOUT,
             CIPPulse := "Timer 5S/30s",
             Filler_Product_Req := "Receive Product Request Filling Mespack P1",
             Filler_CIP_Req := "Receive CIP Enable Filling Mespack P1",
             Loading_Busy_2 := ("T-24.00".State.Tank_inloading AND "T-24.00".Cmd.Inload_Select_Tank_2) OR ("T-81.00".State.Tank_inloading AND "T-81.00".Cmd.Inload_Select_Tank_2) OR ("T-79.00".State.Tank_inloading AND "T-79.00".Cmd.Inload_Select_Tank_2),
             CIP_En := NOT "Gen_Storage"."THE5 CIP"."CIP Request" AND NOT "T-24.00".CIP_Line_Req AND NOT "T-33.00".State."CIP Req" AND NOT "T-34.00".State."CIP Req" AND NOT "T-35.00".State."CIP Req" AND NOT "T-79.00".State."CIP Req" AND NOT "T-81.00".State."CIP Req" AND NOT "T-84.00".State."CIP Req",
             CIP_Tank_Req => "Mix_to_CIP".CIP_Request."T-85.00_CIP_Request",
             CIP_LineOK => "Mix_to_CIP".CIP_Line_OK."T-85.00_CIP_LineOK");
END_REGION

REGION Network 39: T-85 Valve
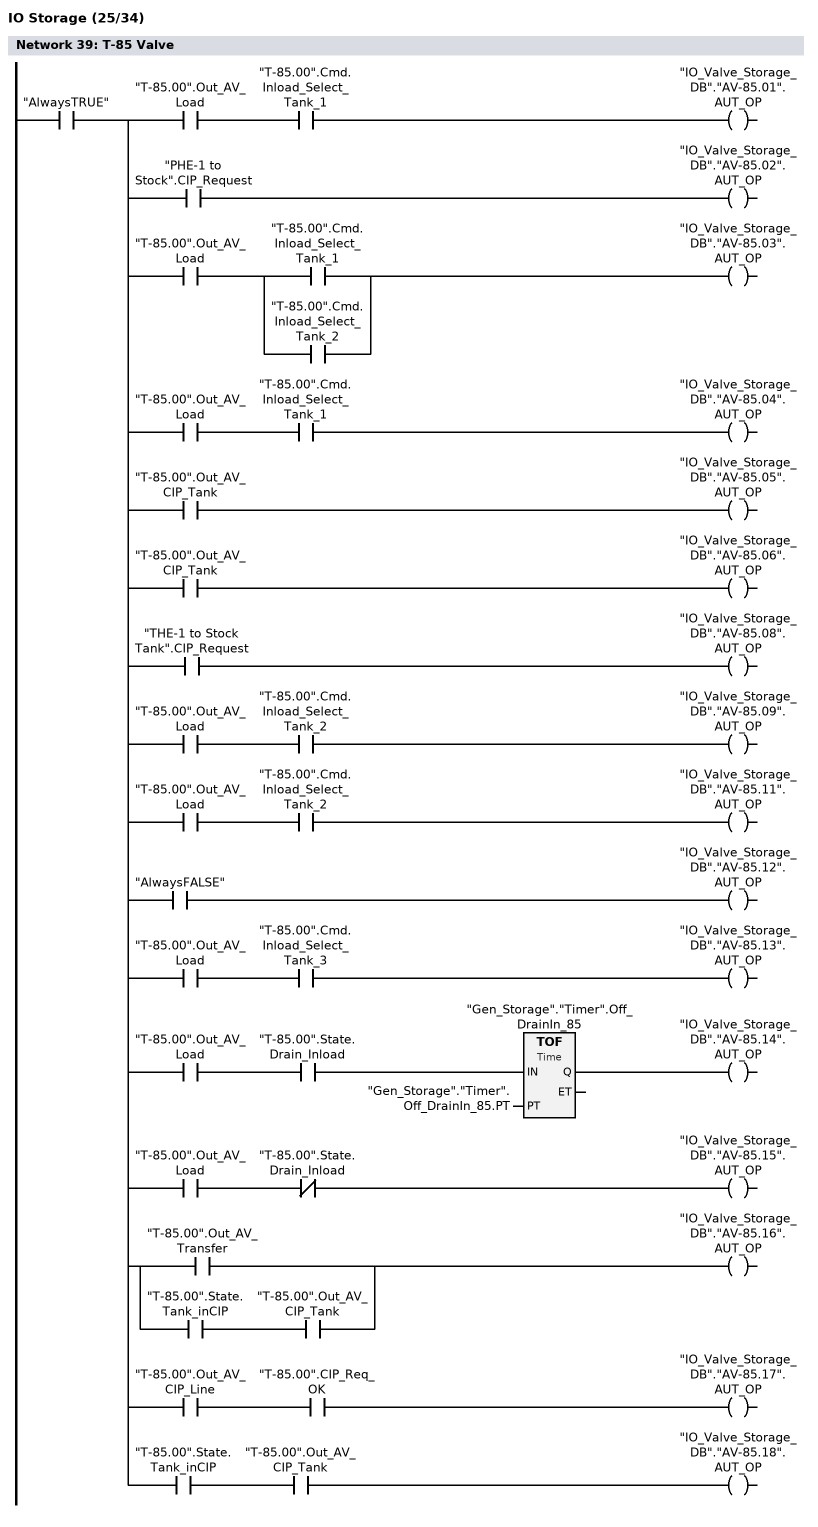
   RUNG wire#powerrail
      Contact( "AlwaysTRUE" )
      wire#w1
      Contact( "T-85.00".Out_AV_Load )
      Contact( "T-85.00".Cmd.Inload_Select_Tank_1 )
      Coil( "IO_Valve_Storage_DB"."AV-85.01".AUT_OP )
   END_RUNG
   RUNG wire#w1
      Contact( "PHE-1 to Stock".CIP_Request )
      Coil( "IO_Valve_Storage_DB"."AV-85.02".AUT_OP )
   END_RUNG
   RUNG wire#w1
      Contact( "T-85.00".Out_AV_Load )
      wire#w2
      Contact( "T-85.00".Cmd.Inload_Select_Tank_1 )
      wire#w3
      Coil( "IO_Valve_Storage_DB"."AV-85.03".AUT_OP )
   END_RUNG
   RUNG wire#w2
      Contact( "T-85.00".Cmd.Inload_Select_Tank_2 )
   END_RUNG wire#w3
   RUNG wire#w1
      Contact( "T-85.00".Out_AV_Load )
      Contact( "T-85.00".Cmd.Inload_Select_Tank_1 )
      Coil( "IO_Valve_Storage_DB"."AV-85.04".AUT_OP )
   END_RUNG
   RUNG wire#w1
      Contact( "T-85.00".Out_AV_CIP_Tank )
      Coil( "IO_Valve_Storage_DB"."AV-85.05".AUT_OP )
   END_RUNG
   RUNG wire#w1
      Contact( "T-85.00".Out_AV_CIP_Tank )
      Coil( "IO_Valve_Storage_DB"."AV-85.06".AUT_OP )
   END_RUNG
   RUNG wire#w1
      Contact( "THE-1 to Stock Tank".CIP_Request )
      Coil( "IO_Valve_Storage_DB"."AV-85.08".AUT_OP )
   END_RUNG
   RUNG wire#w1
      Contact( "T-85.00".Out_AV_Load )
      Contact( "T-85.00".Cmd.Inload_Select_Tank_2 )
      Coil( "IO_Valve_Storage_DB"."AV-85.09".AUT_OP )
   END_RUNG
   RUNG wire#w1
      Contact( "T-85.00".Out_AV_Load )
      Contact( "T-85.00".Cmd.Inload_Select_Tank_2 )
      Coil( "IO_Valve_Storage_DB"."AV-85.11".AUT_OP )
   END_RUNG
   RUNG wire#w1
      Contact( "AlwaysFALSE" )
      Coil( "IO_Valve_Storage_DB"."AV-85.12".AUT_OP )
   END_RUNG
   RUNG wire#w1
      Contact( "T-85.00".Out_AV_Load )
      Contact( "T-85.00".Cmd.Inload_Select_Tank_3 )
      Coil( "IO_Valve_Storage_DB"."AV-85.13".AUT_OP )
   END_RUNG
   RUNG wire#w1
      Contact( "T-85.00".Out_AV_Load )
      Contact( "T-85.00".State.Drain_Inload )
      { S7_Templates := "time_type := Time" } "Gen_Storage"."Timer".Off_DrainIn_85.TOF(pt := "Gen_Storage"."Timer".Off_DrainIn_85.PT, et =>)
      Coil( "IO_Valve_Storage_DB"."AV-85.14".AUT_OP )
   END_RUNG
   RUNG wire#w1
      Contact( "T-85.00".Out_AV_Load )
      I_Contact( "T-85.00".State.Drain_Inload )
      Coil( "IO_Valve_Storage_DB"."AV-85.15".AUT_OP )
   END_RUNG
   RUNG wire#w1
      Contact( "T-85.00".Out_AV_Transfer )
      wire#w4
      Coil( "IO_Valve_Storage_DB"."AV-85.16".AUT_OP )
   END_RUNG
   RUNG wire#w1
      Contact( "T-85.00".State.Tank_inCIP )
      Contact( "T-85.00".Out_AV_CIP_Tank )
   END_RUNG wire#w4
   RUNG wire#w1
      Contact( "T-85.00".Out_AV_CIP_Line )
      Contact( "T-85.00".CIP_Req_OK )
      Coil( "IO_Valve_Storage_DB"."AV-85.17".AUT_OP )
   END_RUNG
   RUNG wire#w1
      Contact( "T-85.00".State.Tank_inCIP )
      Contact( "T-85.00".Out_AV_CIP_Tank )
      Coil( "IO_Valve_Storage_DB"."AV-85.18".AUT_OP )
   END_RUNG
   // the same network as SCL:
   "IO_Valve_Storage_DB"."AV-85.01".AUT_OP := "AlwaysTRUE" AND "T-85.00".Out_AV_Load AND "T-85.00".Cmd.Inload_Select_Tank_1;
   "IO_Valve_Storage_DB"."AV-85.02".AUT_OP := "AlwaysTRUE" AND "PHE-1 to Stock".CIP_Request;
   "IO_Valve_Storage_DB"."AV-85.03".AUT_OP := "AlwaysTRUE" AND "T-85.00".Out_AV_Load AND ("T-85.00".Cmd.Inload_Select_Tank_1 OR "T-85.00".Cmd.Inload_Select_Tank_2);
   "IO_Valve_Storage_DB"."AV-85.04".AUT_OP := "AlwaysTRUE" AND "T-85.00".Out_AV_Load AND "T-85.00".Cmd.Inload_Select_Tank_1;
   "IO_Valve_Storage_DB"."AV-85.05".AUT_OP := "AlwaysTRUE" AND "T-85.00".Out_AV_CIP_Tank;
   "IO_Valve_Storage_DB"."AV-85.06".AUT_OP := "AlwaysTRUE" AND "T-85.00".Out_AV_CIP_Tank;
   "IO_Valve_Storage_DB"."AV-85.08".AUT_OP := "AlwaysTRUE" AND "THE-1 to Stock Tank".CIP_Request;
   "IO_Valve_Storage_DB"."AV-85.09".AUT_OP := "AlwaysTRUE" AND "T-85.00".Out_AV_Load AND "T-85.00".Cmd.Inload_Select_Tank_2;
   "IO_Valve_Storage_DB"."AV-85.11".AUT_OP := "AlwaysTRUE" AND "T-85.00".Out_AV_Load AND "T-85.00".Cmd.Inload_Select_Tank_2;
   "IO_Valve_Storage_DB"."AV-85.12".AUT_OP := "AlwaysTRUE" AND "AlwaysFALSE";
   "IO_Valve_Storage_DB"."AV-85.13".AUT_OP := "AlwaysTRUE" AND "T-85.00".Out_AV_Load AND "T-85.00".Cmd.Inload_Select_Tank_3;
   "Gen_Storage"."Timer".Off_DrainIn_85.TOF(IN := "AlwaysTRUE" AND "T-85.00".Out_AV_Load AND "T-85.00".State.Drain_Inload,
                           PT := "Gen_Storage"."Timer".Off_DrainIn_85.PT);
   "IO_Valve_Storage_DB"."AV-85.14".AUT_OP := "Gen_Storage"."Timer".Off_DrainIn_85.Q;
   "IO_Valve_Storage_DB"."AV-85.15".AUT_OP := "AlwaysTRUE" AND "T-85.00".Out_AV_Load AND NOT "T-85.00".State.Drain_Inload;
   "IO_Valve_Storage_DB"."AV-85.16".AUT_OP := "AlwaysTRUE" AND ("T-85.00".Out_AV_Transfer OR ("T-85.00".State.Tank_inCIP AND "T-85.00".Out_AV_CIP_Tank));
   "IO_Valve_Storage_DB"."AV-85.17".AUT_OP := "AlwaysTRUE" AND "T-85.00".Out_AV_CIP_Line AND "T-85.00".CIP_Req_OK;
   "IO_Valve_Storage_DB"."AV-85.18".AUT_OP := "AlwaysTRUE" AND "T-85.00".State.Tank_inCIP AND "T-85.00".Out_AV_CIP_Tank;
END_REGION

REGION Network 40: Comm T-85 to THE-1
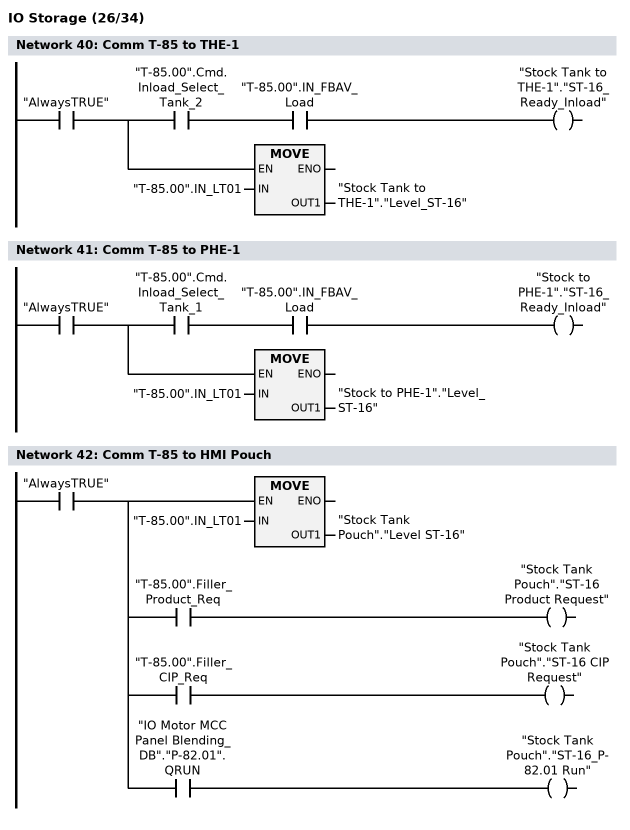
   RUNG wire#powerrail
      Contact( "AlwaysTRUE" )
      wire#w1
      Contact( "T-85.00".Cmd.Inload_Select_Tank_2 )
      Contact( "T-85.00".IN_FBAV_Load )
      Coil( "Stock Tank to THE-1"."ST-16_Ready_Inload" )
   END_RUNG
   RUNG wire#w1
      Move(in := "T-85.00".IN_LT01, out1 => "Stock Tank to THE-1"."Level_ST-16")
   END_RUNG
   // the same network as SCL:
   "Stock Tank to THE-1"."ST-16_Ready_Inload" := "AlwaysTRUE" AND "T-85.00".Cmd.Inload_Select_Tank_2 AND "T-85.00".IN_FBAV_Load;
   IF "AlwaysTRUE" THEN "Stock Tank to THE-1"."Level_ST-16" := "T-85.00".IN_LT01; END_IF;
END_REGION

REGION Network 41: Comm T-85 to PHE-1
   RUNG wire#powerrail
      Contact( "AlwaysTRUE" )
      wire#w1
      Contact( "T-85.00".Cmd.Inload_Select_Tank_1 )
      Contact( "T-85.00".IN_FBAV_Load )
      Coil( "Stock to PHE-1"."ST-16_Ready_Inload" )
   END_RUNG
   RUNG wire#w1
      Move(in := "T-85.00".IN_LT01, out1 => "Stock to PHE-1"."Level_ST-16")
   END_RUNG
   // the same network as SCL:
   "Stock to PHE-1"."ST-16_Ready_Inload" := "AlwaysTRUE" AND "T-85.00".Cmd.Inload_Select_Tank_1 AND "T-85.00".IN_FBAV_Load;
   IF "AlwaysTRUE" THEN "Stock to PHE-1"."Level_ST-16" := "T-85.00".IN_LT01; END_IF;
END_REGION

REGION Network 42: Comm T-85 to HMI Pouch
   RUNG wire#powerrail
      Contact( "AlwaysTRUE" )
      wire#w1
      Move(in := "T-85.00".IN_LT01, out1 => "Stock Tank Pouch"."Level ST-16")
   END_RUNG
   RUNG wire#w1
      Contact( "T-85.00".Filler_Product_Req )
      Coil( "Stock Tank Pouch"."ST-16 Product Request" )
   END_RUNG
   RUNG wire#w1
      Contact( "T-85.00".Filler_CIP_Req )
      Coil( "Stock Tank Pouch"."ST-16 CIP Request" )
   END_RUNG
   RUNG wire#w1
      Contact( "IO Motor MCC Panel Blending_DB"."P-82.01".QRUN )
      Coil( "Stock Tank Pouch"."ST-16_P-82.01 Run" )
   END_RUNG
   // the same network as SCL:
   IF "AlwaysTRUE" THEN "Stock Tank Pouch"."Level ST-16" := "T-85.00".IN_LT01; END_IF;
   "Stock Tank Pouch"."ST-16 Product Request" := "AlwaysTRUE" AND "T-85.00".Filler_Product_Req;
   "Stock Tank Pouch"."ST-16 CIP Request" := "AlwaysTRUE" AND "T-85.00".Filler_CIP_Req;
   "Stock Tank Pouch"."ST-16_P-82.01 Run" := "AlwaysTRUE" AND "IO Motor MCC Panel Blending_DB"."P-82.01".QRUN;
END_REGION

REGION Network 44: T-84.00 ST-14
   // Inload 1 : THE 5
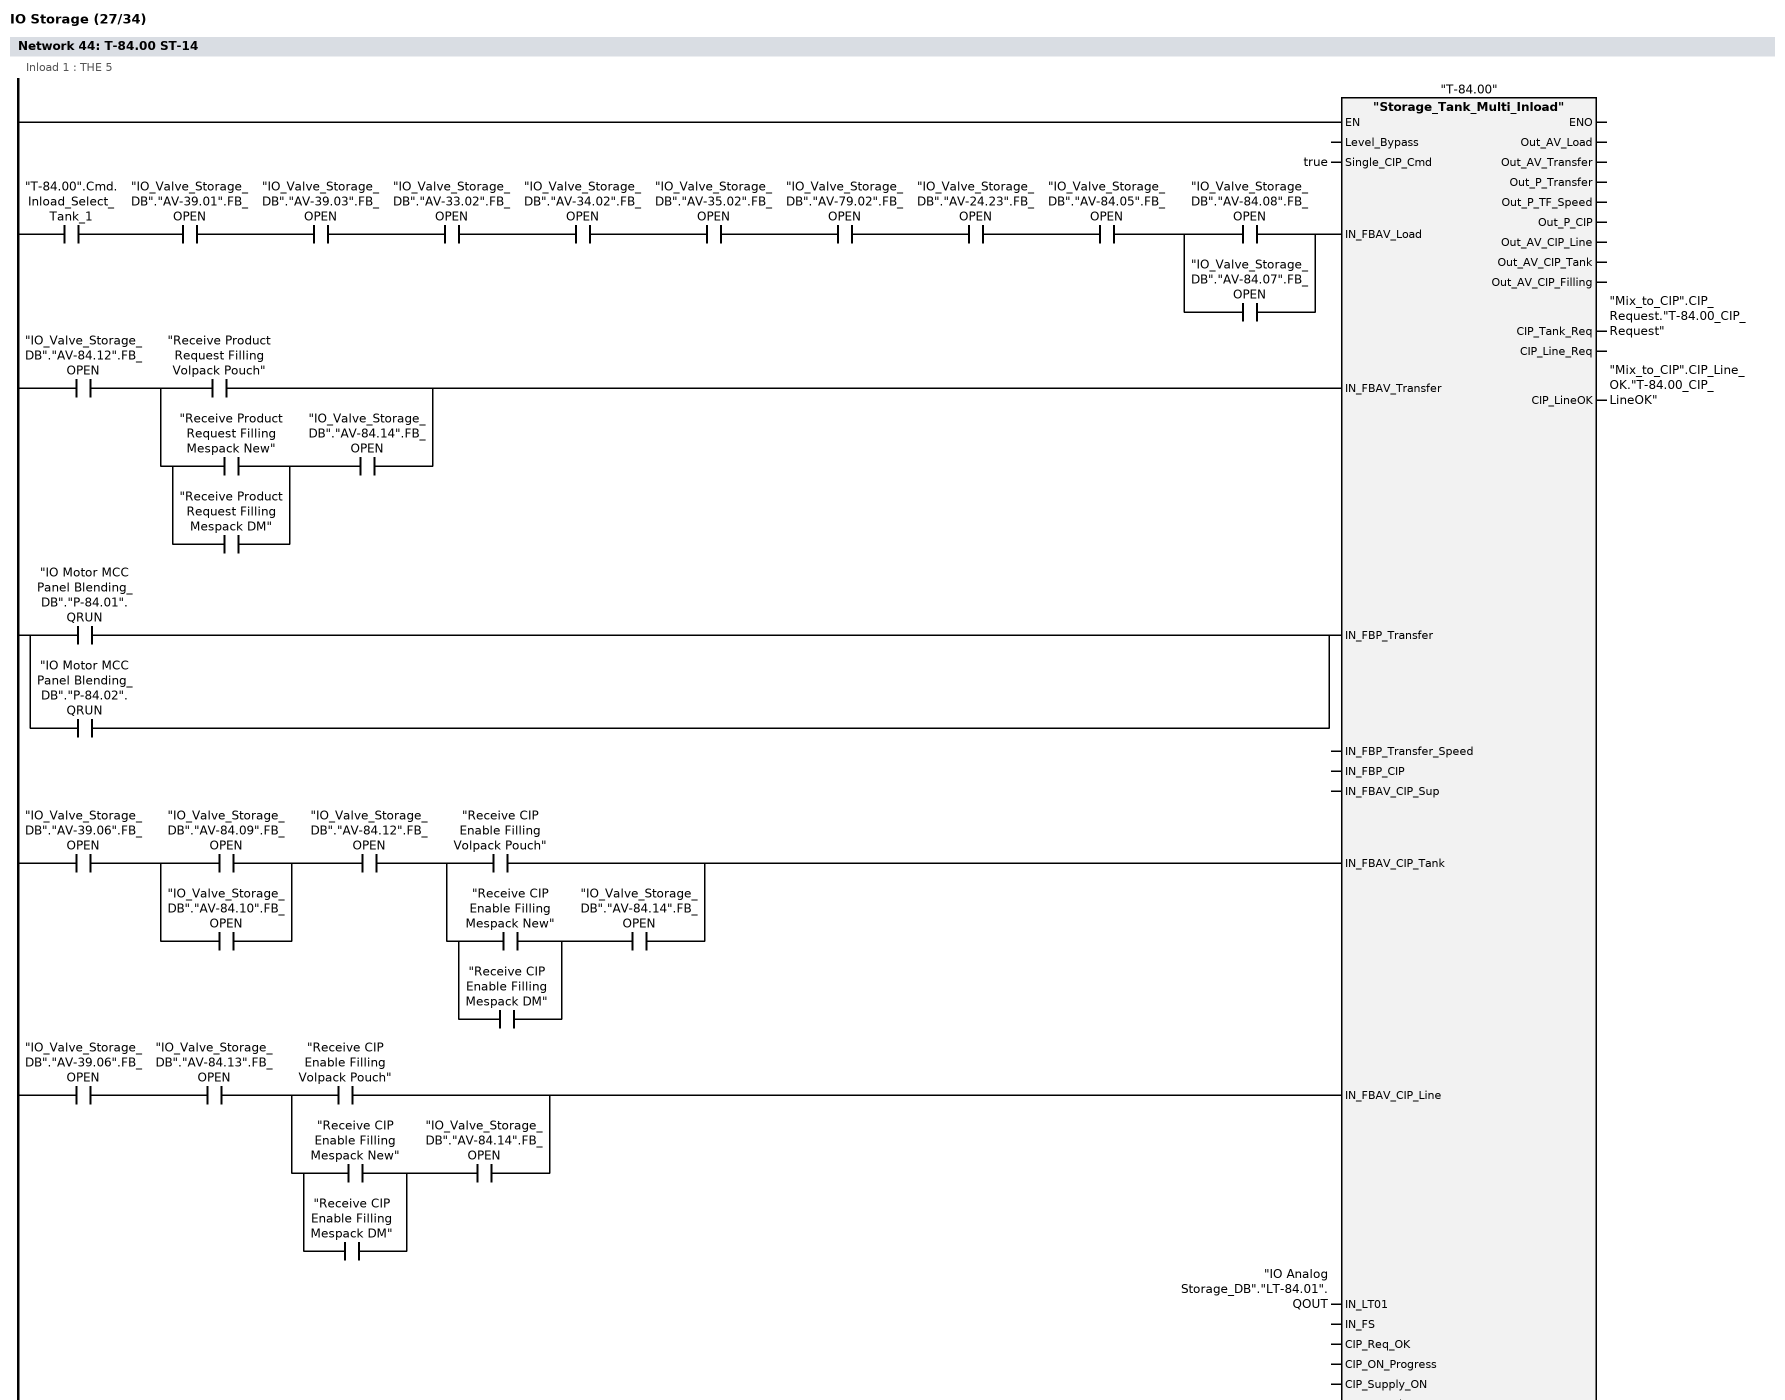
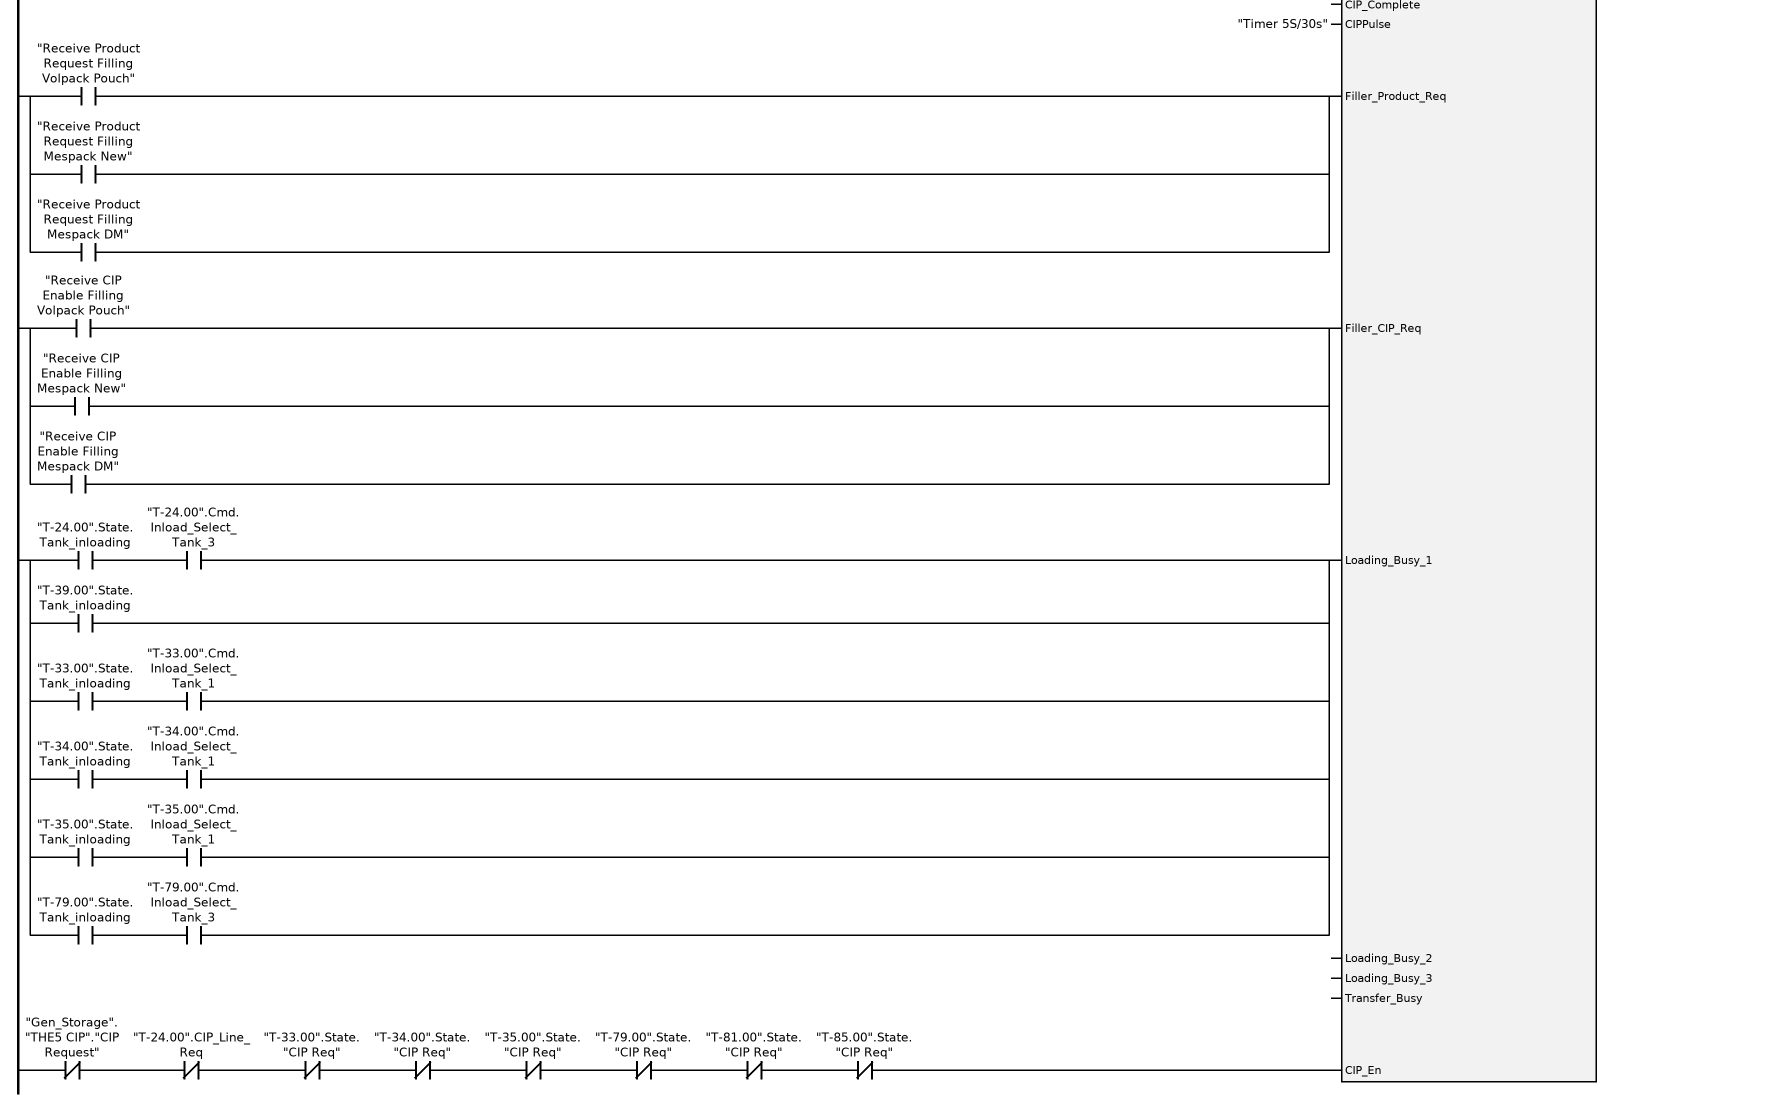
   RUNG wire#powerrail
      "T-84.00"(IN_FBAV_Load := wire#w2, IN_FBAV_Transfer := wire#w5, IN_FBP_Transfer := wire#w6, IN_FBAV_CIP_Tank := wire#w11, IN_FBAV_CIP_Line := wire#w14, Filler_Product_Req := wire#w15, Filler_CIP_Req := wire#w16, Loading_Busy_1 := wire#w17, CIP_En := wire#w18, Level_Bypass :=, Single_CIP_Cmd := true, IN_FBP_Transfer_Speed :=, IN_FBP_CIP :=, IN_FBAV_CIP_Sup :=, IN_LT01 := "IO Analog Storage_DB"."LT-84.01".QOUT, IN_FS :=, CIP_Req_OK :=, CIP_ON_Progress :=, CIP_Supply_ON :=, CIP_Complete :=, CIPPulse := "Timer 5S/30s", Loading_Busy_2 :=, Loading_Busy_3 :=, Transfer_Busy :=, Out_AV_Load =>, Out_AV_Transfer =>, Out_P_Transfer =>, Out_P_TF_Speed =>, Out_P_CIP =>, Out_AV_CIP_Line =>, Out_AV_CIP_Tank =>, Out_AV_CIP_Filling =>, CIP_Tank_Req => "Mix_to_CIP".CIP_Request."T-84.00_CIP_Request", CIP_Line_Req =>, CIP_LineOK => "Mix_to_CIP".CIP_Line_OK."T-84.00_CIP_LineOK")
   END_RUNG
   RUNG wire#powerrail
      Contact( "T-84.00".Cmd.Inload_Select_Tank_1 )
      Contact( "IO_Valve_Storage_DB"."AV-39.01".FB_OPEN )
      Contact( "IO_Valve_Storage_DB"."AV-39.03".FB_OPEN )
      Contact( "IO_Valve_Storage_DB"."AV-33.02".FB_OPEN )
      Contact( "IO_Valve_Storage_DB"."AV-34.02".FB_OPEN )
      Contact( "IO_Valve_Storage_DB"."AV-35.02".FB_OPEN )
      Contact( "IO_Valve_Storage_DB"."AV-79.02".FB_OPEN )
      Contact( "IO_Valve_Storage_DB"."AV-24.23".FB_OPEN )
      Contact( "IO_Valve_Storage_DB"."AV-84.05".FB_OPEN )
      wire#w1
      Contact( "IO_Valve_Storage_DB"."AV-84.08".FB_OPEN )
   END_RUNG wire#w2
   RUNG wire#w1
      Contact( "IO_Valve_Storage_DB"."AV-84.07".FB_OPEN )
   END_RUNG wire#w2
   RUNG wire#powerrail
      Contact( "IO_Valve_Storage_DB"."AV-84.12".FB_OPEN )
      wire#w3
      Contact( "Receive Product Request Filling Volpack Pouch" )
   END_RUNG wire#w5
   RUNG wire#w3
      Contact( "Receive Product Request Filling Mespack New" )
      wire#w4
      Contact( "IO_Valve_Storage_DB"."AV-84.14".FB_OPEN )
   END_RUNG wire#w5
   RUNG wire#w3
      Contact( "Receive Product Request Filling Mespack DM" )
   END_RUNG wire#w4
   RUNG wire#powerrail
      Contact( "IO Motor MCC Panel Blending_DB"."P-84.01".QRUN )
   END_RUNG wire#w6
   RUNG wire#powerrail
      Contact( "IO Motor MCC Panel Blending_DB"."P-84.02".QRUN )
   END_RUNG wire#w6
   RUNG wire#powerrail
      Contact( "IO_Valve_Storage_DB"."AV-39.06".FB_OPEN )
      wire#w7
      Contact( "IO_Valve_Storage_DB"."AV-84.09".FB_OPEN )
      wire#w8
      Contact( "IO_Valve_Storage_DB"."AV-84.12".FB_OPEN )
      wire#w9
      Contact( "Receive CIP Enable Filling Volpack Pouch" )
   END_RUNG wire#w11
   RUNG wire#w7
      Contact( "IO_Valve_Storage_DB"."AV-84.10".FB_OPEN )
   END_RUNG wire#w8
   RUNG wire#w9
      Contact( "Receive CIP Enable Filling Mespack New" )
      wire#w10
      Contact( "IO_Valve_Storage_DB"."AV-84.14".FB_OPEN )
   END_RUNG wire#w11
   RUNG wire#w9
      Contact( "Receive CIP Enable Filling Mespack DM" )
   END_RUNG wire#w10
   RUNG wire#powerrail
      Contact( "IO_Valve_Storage_DB"."AV-39.06".FB_OPEN )
      Contact( "IO_Valve_Storage_DB"."AV-84.13".FB_OPEN )
      wire#w12
      Contact( "Receive CIP Enable Filling Volpack Pouch" )
   END_RUNG wire#w14
   RUNG wire#w12
      Contact( "Receive CIP Enable Filling Mespack New" )
      wire#w13
      Contact( "IO_Valve_Storage_DB"."AV-84.14".FB_OPEN )
   END_RUNG wire#w14
   RUNG wire#w12
      Contact( "Receive CIP Enable Filling Mespack DM" )
   END_RUNG wire#w13
   RUNG wire#powerrail
      Contact( "Receive Product Request Filling Volpack Pouch" )
   END_RUNG wire#w15
   RUNG wire#powerrail
      Contact( "Receive Product Request Filling Mespack New" )
   END_RUNG wire#w15
   RUNG wire#powerrail
      Contact( "Receive Product Request Filling Mespack DM" )
   END_RUNG wire#w15
   RUNG wire#powerrail
      Contact( "Receive CIP Enable Filling Volpack Pouch" )
   END_RUNG wire#w16
   RUNG wire#powerrail
      Contact( "Receive CIP Enable Filling Mespack New" )
   END_RUNG wire#w16
   RUNG wire#powerrail
      Contact( "Receive CIP Enable Filling Mespack DM" )
   END_RUNG wire#w16
   RUNG wire#powerrail
      Contact( "T-24.00".State.Tank_inloading )
      Contact( "T-24.00".Cmd.Inload_Select_Tank_3 )
   END_RUNG wire#w17
   RUNG wire#powerrail
      Contact( "T-39.00".State.Tank_inloading )
   END_RUNG wire#w17
   RUNG wire#powerrail
      Contact( "T-33.00".State.Tank_inloading )
      Contact( "T-33.00".Cmd.Inload_Select_Tank_1 )
   END_RUNG wire#w17
   RUNG wire#powerrail
      Contact( "T-34.00".State.Tank_inloading )
      Contact( "T-34.00".Cmd.Inload_Select_Tank_1 )
   END_RUNG wire#w17
   RUNG wire#powerrail
      Contact( "T-35.00".State.Tank_inloading )
      Contact( "T-35.00".Cmd.Inload_Select_Tank_1 )
   END_RUNG wire#w17
   RUNG wire#powerrail
      Contact( "T-79.00".State.Tank_inloading )
      Contact( "T-79.00".Cmd.Inload_Select_Tank_3 )
   END_RUNG wire#w17
   RUNG wire#powerrail
      I_Contact( "Gen_Storage"."THE5 CIP"."CIP Request" )
      I_Contact( "T-24.00".CIP_Line_Req )
      I_Contact( "T-33.00".State."CIP Req" )
      I_Contact( "T-34.00".State."CIP Req" )
      I_Contact( "T-35.00".State."CIP Req" )
      I_Contact( "T-79.00".State."CIP Req" )
      I_Contact( "T-81.00".State."CIP Req" )
      I_Contact( "T-85.00".State."CIP Req" )
   END_RUNG wire#w18
   // the same network as SCL:
   "T-84.00"(Single_CIP_Cmd := true,   // "Storage_Tank_Multi_Inload"
             IN_FBAV_Load := "T-84.00".Cmd.Inload_Select_Tank_1 AND "IO_Valve_Storage_DB"."AV-39.01".FB_OPEN AND "IO_Valve_Storage_DB"."AV-39.03".FB_OPEN AND "IO_Valve_Storage_DB"."AV-33.02".FB_OPEN AND "IO_Valve_Storage_DB"."AV-34.02".FB_OPEN AND "IO_Valve_Storage_DB"."AV-35.02".FB_OPEN AND "IO_Valve_Storage_DB"."AV-79.02".FB_OPEN AND "IO_Valve_Storage_DB"."AV-24.23".FB_OPEN AND "IO_Valve_Storage_DB"."AV-84.05".FB_OPEN AND ("IO_Valve_Storage_DB"."AV-84.08".FB_OPEN OR "IO_Valve_Storage_DB"."AV-84.07".FB_OPEN),
             IN_FBAV_Transfer := "IO_Valve_Storage_DB"."AV-84.12".FB_OPEN AND ("Receive Product Request Filling Volpack Pouch" OR (("Receive Product Request Filling Mespack New" OR "Receive Product Request Filling Mespack DM") AND "IO_Valve_Storage_DB"."AV-84.14".FB_OPEN)),
             IN_FBP_Transfer := "IO Motor MCC Panel Blending_DB"."P-84.01".QRUN OR "IO Motor MCC Panel Blending_DB"."P-84.02".QRUN,
             IN_FBAV_CIP_Tank := "IO_Valve_Storage_DB"."AV-39.06".FB_OPEN AND ("IO_Valve_Storage_DB"."AV-84.09".FB_OPEN OR "IO_Valve_Storage_DB"."AV-84.10".FB_OPEN) AND "IO_Valve_Storage_DB"."AV-84.12".FB_OPEN AND ("Receive CIP Enable Filling Volpack Pouch" OR (("Receive CIP Enable Filling Mespack New" OR "Receive CIP Enable Filling Mespack DM") AND "IO_Valve_Storage_DB"."AV-84.14".FB_OPEN)),
             IN_FBAV_CIP_Line := "IO_Valve_Storage_DB"."AV-39.06".FB_OPEN AND "IO_Valve_Storage_DB"."AV-84.13".FB_OPEN AND ("Receive CIP Enable Filling Volpack Pouch" OR (("Receive CIP Enable Filling Mespack New" OR "Receive CIP Enable Filling Mespack DM") AND "IO_Valve_Storage_DB"."AV-84.14".FB_OPEN)),
             IN_LT01 := "IO Analog Storage_DB"."LT-84.01".QOUT,
             CIPPulse := "Timer 5S/30s",
             Filler_Product_Req := "Receive Product Request Filling Volpack Pouch" OR "Receive Product Request Filling Mespack New" OR "Receive Product Request Filling Mespack DM",
             Filler_CIP_Req := "Receive CIP Enable Filling Volpack Pouch" OR "Receive CIP Enable Filling Mespack New" OR "Receive CIP Enable Filling Mespack DM",
             Loading_Busy_1 := ("T-24.00".State.Tank_inloading AND "T-24.00".Cmd.Inload_Select_Tank_3) OR "T-39.00".State.Tank_inloading OR ("T-33.00".State.Tank_inloading AND "T-33.00".Cmd.Inload_Select_Tank_1) OR ("T-34.00".State.Tank_inloading AND "T-34.00".Cmd.Inload_Select_Tank_1) OR ("T-35.00".State.Tank_inloading AND "T-35.00".Cmd.Inload_Select_Tank_1) OR ("T-79.00".State.Tank_inloading AND "T-79.00".Cmd.Inload_Select_Tank_3),
             CIP_En := NOT "Gen_Storage"."THE5 CIP"."CIP Request" AND NOT "T-24.00".CIP_Line_Req AND NOT "T-33.00".State."CIP Req" AND NOT "T-34.00".State."CIP Req" AND NOT "T-35.00".State."CIP Req" AND NOT "T-79.00".State."CIP Req" AND NOT "T-81.00".State."CIP Req" AND NOT "T-85.00".State."CIP Req",
             CIP_Tank_Req => "Mix_to_CIP".CIP_Request."T-84.00_CIP_Request",
             CIP_LineOK => "Mix_to_CIP".CIP_Line_OK."T-84.00_CIP_LineOK");
END_REGION

REGION Network 45: T-84 Valve
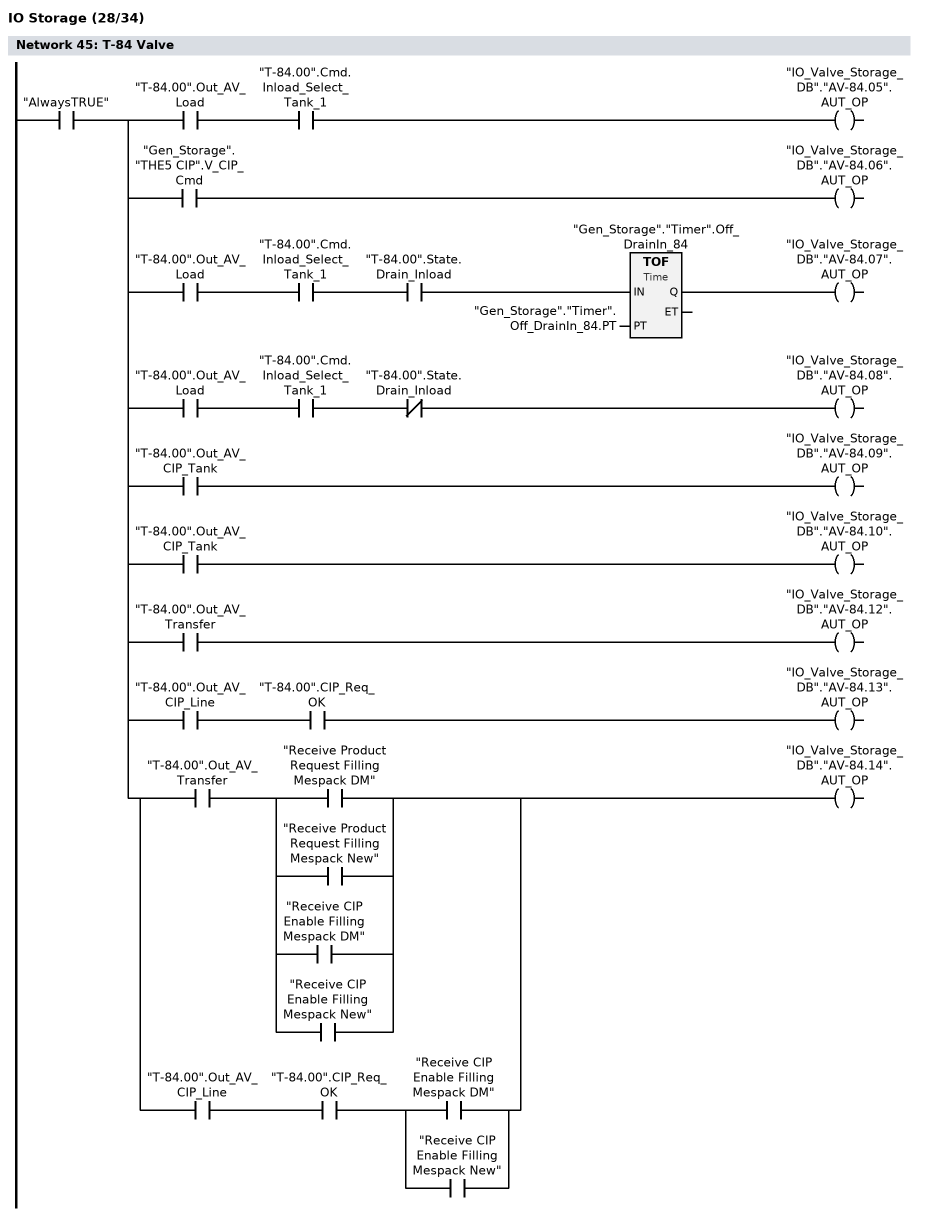
   RUNG wire#powerrail
      Contact( "AlwaysTRUE" )
      wire#w1
      Contact( "T-84.00".Out_AV_Load )
      Contact( "T-84.00".Cmd.Inload_Select_Tank_1 )
      Coil( "IO_Valve_Storage_DB"."AV-84.05".AUT_OP )
   END_RUNG
   RUNG wire#w1
      Contact( "Gen_Storage"."THE5 CIP".V_CIP_Cmd )
      Coil( "IO_Valve_Storage_DB"."AV-84.06".AUT_OP )
   END_RUNG
   RUNG wire#w1
      Contact( "T-84.00".Out_AV_Load )
      Contact( "T-84.00".Cmd.Inload_Select_Tank_1 )
      Contact( "T-84.00".State.Drain_Inload )
      { S7_Templates := "time_type := Time" } "Gen_Storage"."Timer".Off_DrainIn_84.TOF(pt := "Gen_Storage"."Timer".Off_DrainIn_84.PT, et =>)
      Coil( "IO_Valve_Storage_DB"."AV-84.07".AUT_OP )
   END_RUNG
   RUNG wire#w1
      Contact( "T-84.00".Out_AV_Load )
      Contact( "T-84.00".Cmd.Inload_Select_Tank_1 )
      I_Contact( "T-84.00".State.Drain_Inload )
      Coil( "IO_Valve_Storage_DB"."AV-84.08".AUT_OP )
   END_RUNG
   RUNG wire#w1
      Contact( "T-84.00".Out_AV_CIP_Tank )
      Coil( "IO_Valve_Storage_DB"."AV-84.09".AUT_OP )
   END_RUNG
   RUNG wire#w1
      Contact( "T-84.00".Out_AV_CIP_Tank )
      Coil( "IO_Valve_Storage_DB"."AV-84.10".AUT_OP )
   END_RUNG
   RUNG wire#w1
      Contact( "T-84.00".Out_AV_Transfer )
      Coil( "IO_Valve_Storage_DB"."AV-84.12".AUT_OP )
   END_RUNG
   RUNG wire#w1
      Contact( "T-84.00".Out_AV_CIP_Line )
      Contact( "T-84.00".CIP_Req_OK )
      Coil( "IO_Valve_Storage_DB"."AV-84.13".AUT_OP )
   END_RUNG
   RUNG wire#w1
      Contact( "T-84.00".Out_AV_Transfer )
      wire#w2
      Contact( "Receive Product Request Filling Mespack DM" )
      wire#w3
      Coil( "IO_Valve_Storage_DB"."AV-84.14".AUT_OP )
   END_RUNG
   RUNG wire#w2
      Contact( "Receive Product Request Filling Mespack New" )
   END_RUNG wire#w3
   RUNG wire#w2
      Contact( "Receive CIP Enable Filling Mespack DM" )
   END_RUNG wire#w3
   RUNG wire#w2
      Contact( "Receive CIP Enable Filling Mespack New" )
   END_RUNG wire#w3
   RUNG wire#w1
      Contact( "T-84.00".Out_AV_CIP_Line )
      Contact( "T-84.00".CIP_Req_OK )
      wire#w4
      Contact( "Receive CIP Enable Filling Mespack DM" )
   END_RUNG wire#w3
   RUNG wire#w4
      Contact( "Receive CIP Enable Filling Mespack New" )
   END_RUNG wire#w3
   // the same network as SCL:
   "IO_Valve_Storage_DB"."AV-84.05".AUT_OP := "AlwaysTRUE" AND "T-84.00".Out_AV_Load AND "T-84.00".Cmd.Inload_Select_Tank_1;
   "IO_Valve_Storage_DB"."AV-84.06".AUT_OP := "AlwaysTRUE" AND "Gen_Storage"."THE5 CIP".V_CIP_Cmd;
   "Gen_Storage"."Timer".Off_DrainIn_84.TOF(IN := "AlwaysTRUE" AND "T-84.00".Out_AV_Load AND "T-84.00".Cmd.Inload_Select_Tank_1 AND "T-84.00".State.Drain_Inload,
                           PT := "Gen_Storage"."Timer".Off_DrainIn_84.PT);
   "IO_Valve_Storage_DB"."AV-84.07".AUT_OP := "Gen_Storage"."Timer".Off_DrainIn_84.Q;
   "IO_Valve_Storage_DB"."AV-84.08".AUT_OP := "AlwaysTRUE" AND "T-84.00".Out_AV_Load AND "T-84.00".Cmd.Inload_Select_Tank_1 AND NOT "T-84.00".State.Drain_Inload;
   "IO_Valve_Storage_DB"."AV-84.09".AUT_OP := "AlwaysTRUE" AND "T-84.00".Out_AV_CIP_Tank;
   "IO_Valve_Storage_DB"."AV-84.10".AUT_OP := "AlwaysTRUE" AND "T-84.00".Out_AV_CIP_Tank;
   "IO_Valve_Storage_DB"."AV-84.12".AUT_OP := "AlwaysTRUE" AND "T-84.00".Out_AV_Transfer;
   "IO_Valve_Storage_DB"."AV-84.13".AUT_OP := "AlwaysTRUE" AND "T-84.00".Out_AV_CIP_Line AND "T-84.00".CIP_Req_OK;
   "IO_Valve_Storage_DB"."AV-84.14".AUT_OP := "AlwaysTRUE" AND (("T-84.00".Out_AV_Transfer AND ("Receive Product Request Filling Mespack DM" OR "Receive Product Request Filling Mespack New" OR "Receive CIP Enable Filling Mespack DM" OR "Receive CIP Enable Filling Mespack New")) OR ("T-84.00".Out_AV_CIP_Line AND "T-84.00".CIP_Req_OK AND ("Receive CIP Enable Filling Mespack DM" OR "Receive CIP Enable Filling Mespack New")));
END_REGION

REGION Network 46: Comm T-84 to HMI Pouch
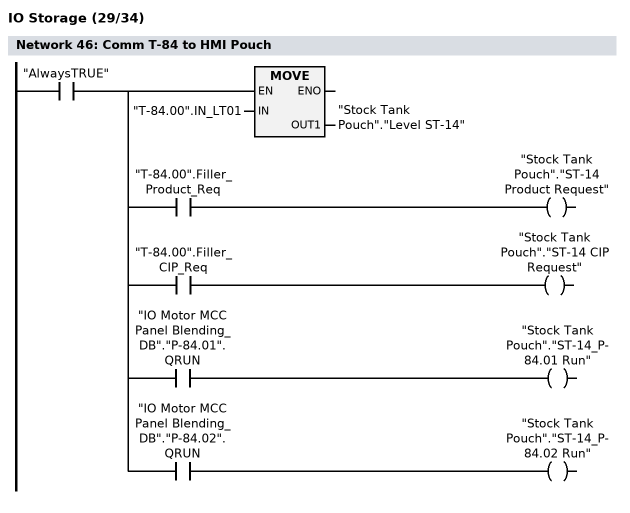
   RUNG wire#powerrail
      Contact( "AlwaysTRUE" )
      wire#w1
      Move(in := "T-84.00".IN_LT01, out1 => "Stock Tank Pouch"."Level ST-14")
   END_RUNG
   RUNG wire#w1
      Contact( "T-84.00".Filler_Product_Req )
      Coil( "Stock Tank Pouch"."ST-14 Product Request" )
   END_RUNG
   RUNG wire#w1
      Contact( "T-84.00".Filler_CIP_Req )
      Coil( "Stock Tank Pouch"."ST-14 CIP Request" )
   END_RUNG
   RUNG wire#w1
      Contact( "IO Motor MCC Panel Blending_DB"."P-84.01".QRUN )
      Coil( "Stock Tank Pouch"."ST-14_P-84.01 Run" )
   END_RUNG
   RUNG wire#w1
      Contact( "IO Motor MCC Panel Blending_DB"."P-84.02".QRUN )
      Coil( "Stock Tank Pouch"."ST-14_P-84.02 Run" )
   END_RUNG
   // the same network as SCL:
   IF "AlwaysTRUE" THEN "Stock Tank Pouch"."Level ST-14" := "T-84.00".IN_LT01; END_IF;
   "Stock Tank Pouch"."ST-14 Product Request" := "AlwaysTRUE" AND "T-84.00".Filler_Product_Req;
   "Stock Tank Pouch"."ST-14 CIP Request" := "AlwaysTRUE" AND "T-84.00".Filler_CIP_Req;
   "Stock Tank Pouch"."ST-14_P-84.01 Run" := "AlwaysTRUE" AND "IO Motor MCC Panel Blending_DB"."P-84.01".QRUN;
   "Stock Tank Pouch"."ST-14_P-84.02 Run" := "AlwaysTRUE" AND "IO Motor MCC Panel Blending_DB"."P-84.02".QRUN;
END_REGION

REGION Network 48: T-79.00 ST-9
   // Inload 1 : THE 4
   // Inload 2 : THE 1
   // Inload 3 : THE 5
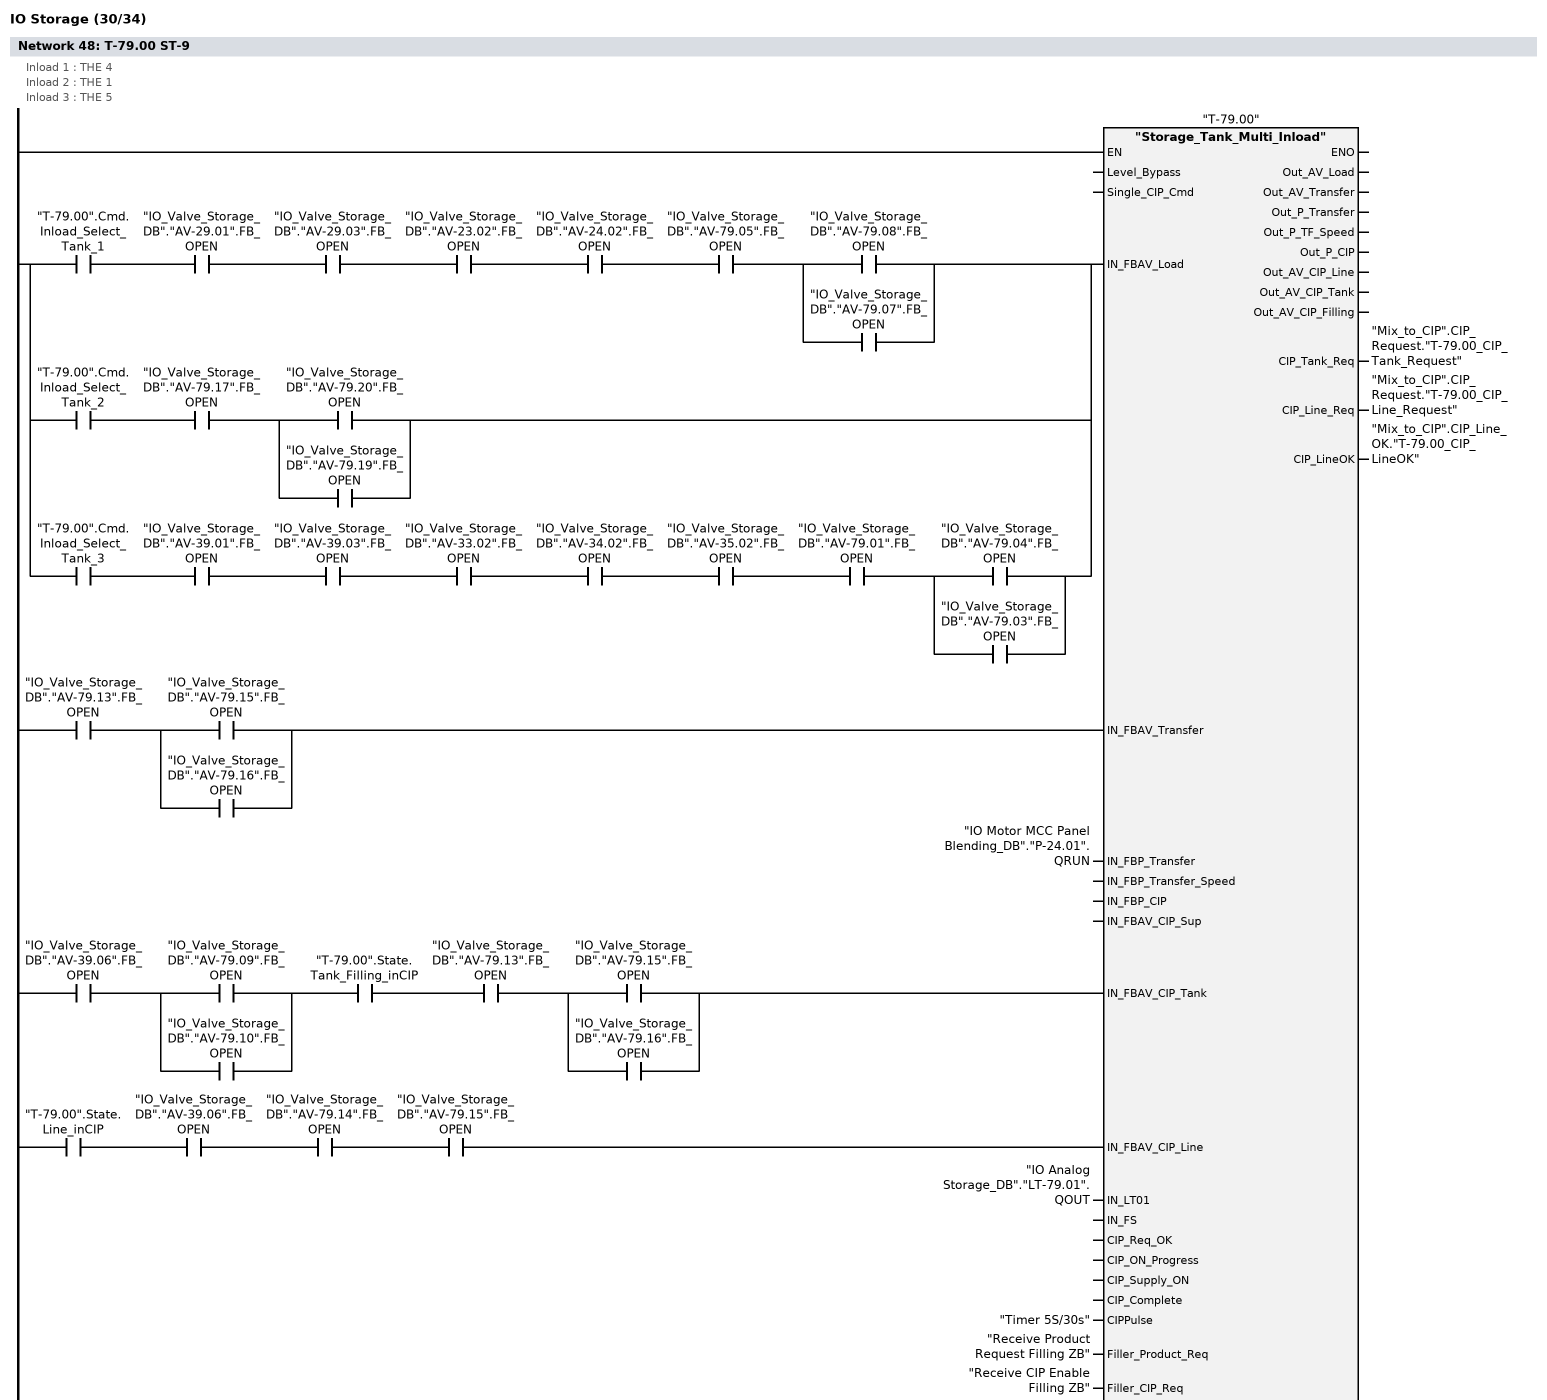
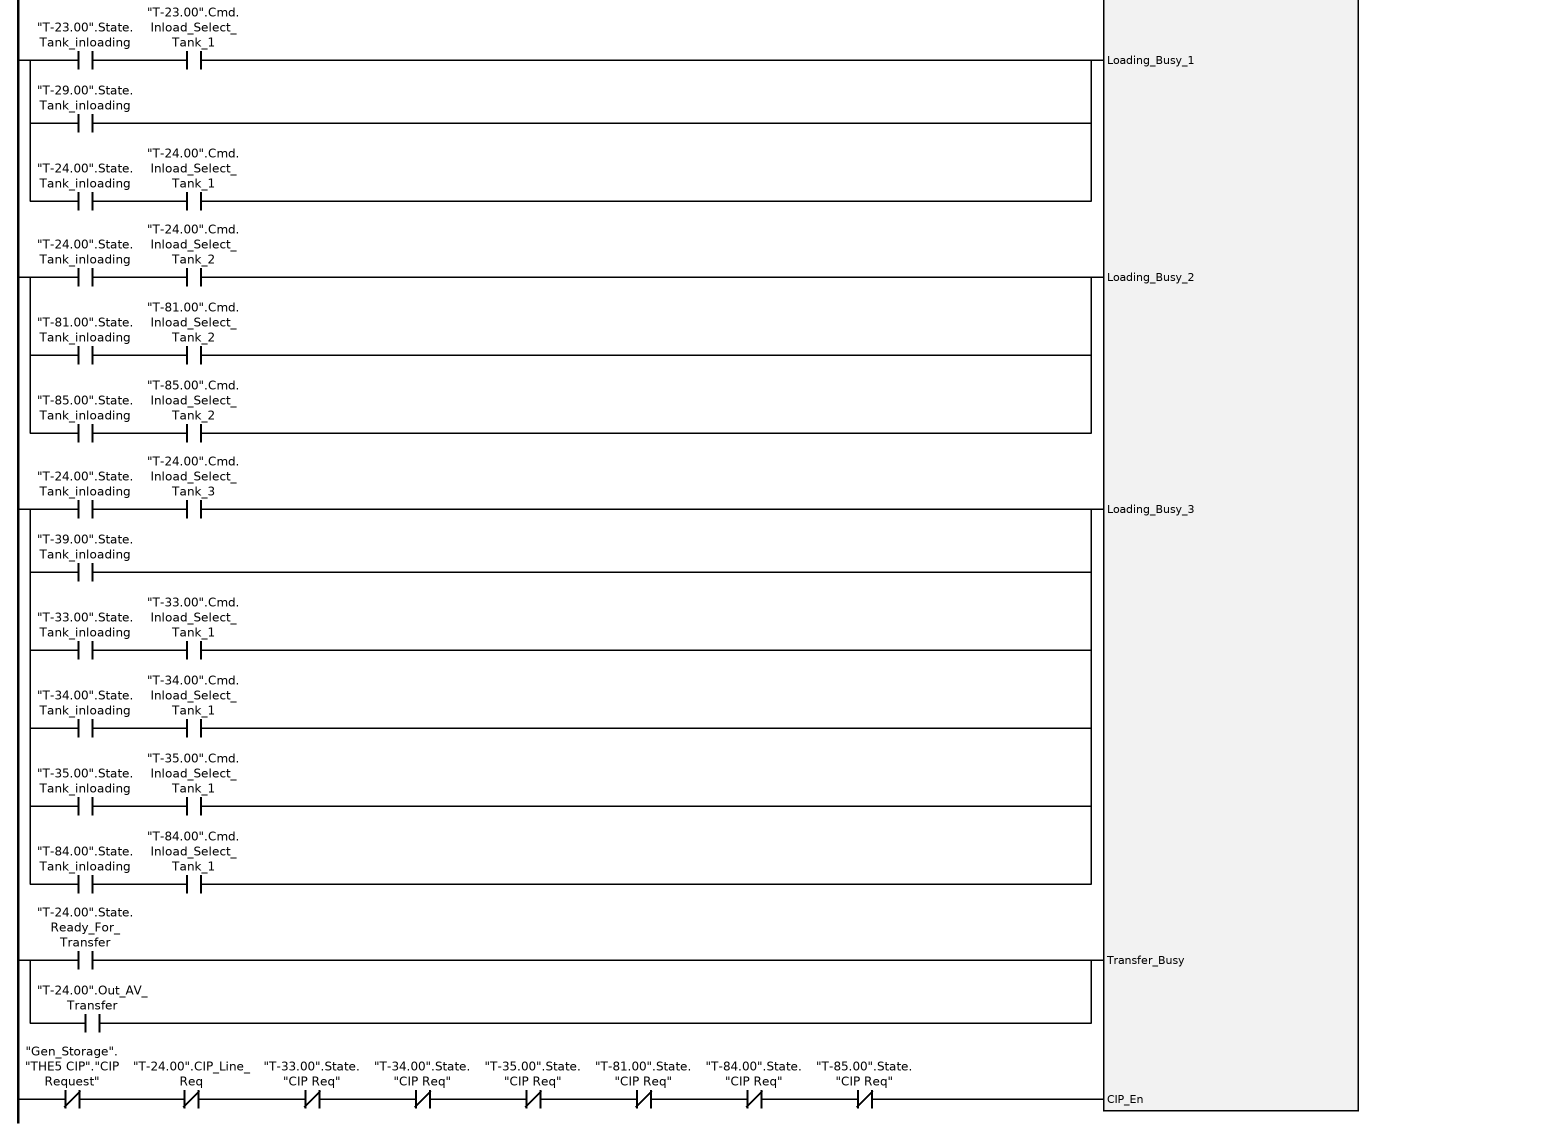
   RUNG wire#powerrail
      "T-79.00"(IN_FBAV_Load := wire#w4, IN_FBAV_Transfer := wire#w6, IN_FBAV_CIP_Tank := wire#w10, IN_FBAV_CIP_Line := wire#w11, Loading_Busy_1 := wire#w12, Loading_Busy_2 := wire#w13, Loading_Busy_3 := wire#w14, Transfer_Busy := wire#w15, CIP_En := wire#w16, Level_Bypass :=, Single_CIP_Cmd :=, IN_FBP_Transfer := "IO Motor MCC Panel Blending_DB"."P-24.01".QRUN, IN_FBP_Transfer_Speed :=, IN_FBP_CIP :=, IN_FBAV_CIP_Sup :=, IN_LT01 := "IO Analog Storage_DB"."LT-79.01".QOUT, IN_FS :=, CIP_Req_OK :=, CIP_ON_Progress :=, CIP_Supply_ON :=, CIP_Complete :=, CIPPulse := "Timer 5S/30s", Filler_Product_Req := "Receive Product Request Filling ZB", Filler_CIP_Req := "Receive CIP Enable Filling ZB", Out_AV_Load =>, Out_AV_Transfer =>, Out_P_Transfer =>, Out_P_TF_Speed =>, Out_P_CIP =>, Out_AV_CIP_Line =>, Out_AV_CIP_Tank =>, Out_AV_CIP_Filling =>, CIP_Tank_Req => "Mix_to_CIP".CIP_Request."T-79.00_CIP_Tank_Request", CIP_Line_Req => "Mix_to_CIP".CIP_Request."T-79.00_CIP_Line_Request", CIP_LineOK => "Mix_to_CIP".CIP_Line_OK."T-79.00_CIP_LineOK")
   END_RUNG
   RUNG wire#powerrail
      Contact( "T-79.00".Cmd.Inload_Select_Tank_1 )
      Contact( "IO_Valve_Storage_DB"."AV-29.01".FB_OPEN )
      Contact( "IO_Valve_Storage_DB"."AV-29.03".FB_OPEN )
      Contact( "IO_Valve_Storage_DB"."AV-23.02".FB_OPEN )
      Contact( "IO_Valve_Storage_DB"."AV-24.02".FB_OPEN )
      Contact( "IO_Valve_Storage_DB"."AV-79.05".FB_OPEN )
      wire#w1
      Contact( "IO_Valve_Storage_DB"."AV-79.08".FB_OPEN )
   END_RUNG wire#w4
   RUNG wire#w1
      Contact( "IO_Valve_Storage_DB"."AV-79.07".FB_OPEN )
   END_RUNG wire#w4
   RUNG wire#powerrail
      Contact( "T-79.00".Cmd.Inload_Select_Tank_2 )
      Contact( "IO_Valve_Storage_DB"."AV-79.17".FB_OPEN )
      wire#w2
      Contact( "IO_Valve_Storage_DB"."AV-79.20".FB_OPEN )
   END_RUNG wire#w4
   RUNG wire#w2
      Contact( "IO_Valve_Storage_DB"."AV-79.19".FB_OPEN )
   END_RUNG wire#w4
   RUNG wire#powerrail
      Contact( "T-79.00".Cmd.Inload_Select_Tank_3 )
      Contact( "IO_Valve_Storage_DB"."AV-39.01".FB_OPEN )
      Contact( "IO_Valve_Storage_DB"."AV-39.03".FB_OPEN )
      Contact( "IO_Valve_Storage_DB"."AV-33.02".FB_OPEN )
      Contact( "IO_Valve_Storage_DB"."AV-34.02".FB_OPEN )
      Contact( "IO_Valve_Storage_DB"."AV-35.02".FB_OPEN )
      Contact( "IO_Valve_Storage_DB"."AV-79.01".FB_OPEN )
      wire#w3
      Contact( "IO_Valve_Storage_DB"."AV-79.04".FB_OPEN )
   END_RUNG wire#w4
   RUNG wire#w3
      Contact( "IO_Valve_Storage_DB"."AV-79.03".FB_OPEN )
   END_RUNG wire#w4
   RUNG wire#powerrail
      Contact( "IO_Valve_Storage_DB"."AV-79.13".FB_OPEN )
      wire#w5
      Contact( "IO_Valve_Storage_DB"."AV-79.15".FB_OPEN )
   END_RUNG wire#w6
   RUNG wire#w5
      Contact( "IO_Valve_Storage_DB"."AV-79.16".FB_OPEN )
   END_RUNG wire#w6
   RUNG wire#powerrail
      Contact( "IO_Valve_Storage_DB"."AV-39.06".FB_OPEN )
      wire#w7
      Contact( "IO_Valve_Storage_DB"."AV-79.09".FB_OPEN )
      wire#w8
      Contact( "T-79.00".State.Tank_Filling_inCIP )
      Contact( "IO_Valve_Storage_DB"."AV-79.13".FB_OPEN )
      wire#w9
      Contact( "IO_Valve_Storage_DB"."AV-79.15".FB_OPEN )
   END_RUNG wire#w10
   RUNG wire#w7
      Contact( "IO_Valve_Storage_DB"."AV-79.10".FB_OPEN )
   END_RUNG wire#w8
   RUNG wire#w9
      Contact( "IO_Valve_Storage_DB"."AV-79.16".FB_OPEN )
   END_RUNG wire#w10
   RUNG wire#powerrail
      Contact( "T-79.00".State.Line_inCIP )
      Contact( "IO_Valve_Storage_DB"."AV-39.06".FB_OPEN )
      Contact( "IO_Valve_Storage_DB"."AV-79.14".FB_OPEN )
      Contact( "IO_Valve_Storage_DB"."AV-79.15".FB_OPEN )
   END_RUNG wire#w11
   RUNG wire#powerrail
      Contact( "T-23.00".State.Tank_inloading )
      Contact( "T-23.00".Cmd.Inload_Select_Tank_1 )
   END_RUNG wire#w12
   RUNG wire#powerrail
      Contact( "T-29.00".State.Tank_inloading )
   END_RUNG wire#w12
   RUNG wire#powerrail
      Contact( "T-24.00".State.Tank_inloading )
      Contact( "T-24.00".Cmd.Inload_Select_Tank_1 )
   END_RUNG wire#w12
   RUNG wire#powerrail
      Contact( "T-24.00".State.Tank_inloading )
      Contact( "T-24.00".Cmd.Inload_Select_Tank_2 )
   END_RUNG wire#w13
   RUNG wire#powerrail
      Contact( "T-81.00".State.Tank_inloading )
      Contact( "T-81.00".Cmd.Inload_Select_Tank_2 )
   END_RUNG wire#w13
   RUNG wire#powerrail
      Contact( "T-85.00".State.Tank_inloading )
      Contact( "T-85.00".Cmd.Inload_Select_Tank_2 )
   END_RUNG wire#w13
   RUNG wire#powerrail
      Contact( "T-24.00".State.Tank_inloading )
      Contact( "T-24.00".Cmd.Inload_Select_Tank_3 )
   END_RUNG wire#w14
   RUNG wire#powerrail
      Contact( "T-39.00".State.Tank_inloading )
   END_RUNG wire#w14
   RUNG wire#powerrail
      Contact( "T-33.00".State.Tank_inloading )
      Contact( "T-33.00".Cmd.Inload_Select_Tank_1 )
   END_RUNG wire#w14
   RUNG wire#powerrail
      Contact( "T-34.00".State.Tank_inloading )
      Contact( "T-34.00".Cmd.Inload_Select_Tank_1 )
   END_RUNG wire#w14
   RUNG wire#powerrail
      Contact( "T-35.00".State.Tank_inloading )
      Contact( "T-35.00".Cmd.Inload_Select_Tank_1 )
   END_RUNG wire#w14
   RUNG wire#powerrail
      Contact( "T-84.00".State.Tank_inloading )
      Contact( "T-84.00".Cmd.Inload_Select_Tank_1 )
   END_RUNG wire#w14
   RUNG wire#powerrail
      Contact( "T-24.00".State.Ready_For_Transfer )
   END_RUNG wire#w15
   RUNG wire#powerrail
      Contact( "T-24.00".Out_AV_Transfer )
   END_RUNG wire#w15
   RUNG wire#powerrail
      I_Contact( "Gen_Storage"."THE5 CIP"."CIP Request" )
      I_Contact( "T-24.00".CIP_Line_Req )
      I_Contact( "T-33.00".State."CIP Req" )
      I_Contact( "T-34.00".State."CIP Req" )
      I_Contact( "T-35.00".State."CIP Req" )
      I_Contact( "T-81.00".State."CIP Req" )
      I_Contact( "T-84.00".State."CIP Req" )
      I_Contact( "T-85.00".State."CIP Req" )
   END_RUNG wire#w16
   // the same network as SCL:
   "T-79.00"(IN_FBAV_Load := ("T-79.00".Cmd.Inload_Select_Tank_1 AND "IO_Valve_Storage_DB"."AV-29.01".FB_OPEN AND "IO_Valve_Storage_DB"."AV-29.03".FB_OPEN AND "IO_Valve_Storage_DB"."AV-23.02".FB_OPEN AND "IO_Valve_Storage_DB"."AV-24.02".FB_OPEN AND "IO_Valve_Storage_DB"."AV-79.05".FB_OPEN AND ("IO_Valve_Storage_DB"."AV-79.08".FB_OPEN OR "IO_Valve_Storage_DB"."AV-79.07".FB_OPEN)) OR ("T-79.00".Cmd.Inload_Select_Tank_2 AND "IO_Valve_Storage_DB"."AV-79.17".FB_OPEN AND ("IO_Valve_Storage_DB"."AV-79.20".FB_OPEN OR "IO_Valve_Storage_DB"."AV-79.19".FB_OPEN)) OR ("T-79.00".Cmd.Inload_Select_Tank_3 AND "IO_Valve_Storage_DB"."AV-39.01".FB_OPEN AND "IO_Valve_Storage_DB"."AV-39.03".FB_OPEN AND "IO_Valve_Storage_DB"."AV-33.02".FB_OPEN AND "IO_Valve_Storage_DB"."AV-34.02".FB_OPEN AND "IO_Valve_Storage_DB"."AV-35.02".FB_OPEN AND "IO_Valve_Storage_DB"."AV-79.01".FB_OPEN AND ("IO_Valve_Storage_DB"."AV-79.04".FB_OPEN OR "IO_Valve_Storage_DB"."AV-79.03".FB_OPEN)),   // "Storage_Tank_Multi_Inload"
             IN_FBAV_Transfer := "IO_Valve_Storage_DB"."AV-79.13".FB_OPEN AND ("IO_Valve_Storage_DB"."AV-79.15".FB_OPEN OR "IO_Valve_Storage_DB"."AV-79.16".FB_OPEN),
             IN_FBP_Transfer := "IO Motor MCC Panel Blending_DB"."P-24.01".QRUN,
             IN_FBAV_CIP_Tank := "IO_Valve_Storage_DB"."AV-39.06".FB_OPEN AND ("IO_Valve_Storage_DB"."AV-79.09".FB_OPEN OR "IO_Valve_Storage_DB"."AV-79.10".FB_OPEN) AND "T-79.00".State.Tank_Filling_inCIP AND "IO_Valve_Storage_DB"."AV-79.13".FB_OPEN AND ("IO_Valve_Storage_DB"."AV-79.15".FB_OPEN OR "IO_Valve_Storage_DB"."AV-79.16".FB_OPEN),
             IN_FBAV_CIP_Line := "T-79.00".State.Line_inCIP AND "IO_Valve_Storage_DB"."AV-39.06".FB_OPEN AND "IO_Valve_Storage_DB"."AV-79.14".FB_OPEN AND "IO_Valve_Storage_DB"."AV-79.15".FB_OPEN,
             IN_LT01 := "IO Analog Storage_DB"."LT-79.01".QOUT,
             CIPPulse := "Timer 5S/30s",
             Filler_Product_Req := "Receive Product Request Filling ZB",
             Filler_CIP_Req := "Receive CIP Enable Filling ZB",
             Loading_Busy_1 := ("T-23.00".State.Tank_inloading AND "T-23.00".Cmd.Inload_Select_Tank_1) OR "T-29.00".State.Tank_inloading OR ("T-24.00".State.Tank_inloading AND "T-24.00".Cmd.Inload_Select_Tank_1),
             Loading_Busy_2 := ("T-24.00".State.Tank_inloading AND "T-24.00".Cmd.Inload_Select_Tank_2) OR ("T-81.00".State.Tank_inloading AND "T-81.00".Cmd.Inload_Select_Tank_2) OR ("T-85.00".State.Tank_inloading AND "T-85.00".Cmd.Inload_Select_Tank_2),
             Loading_Busy_3 := ("T-24.00".State.Tank_inloading AND "T-24.00".Cmd.Inload_Select_Tank_3) OR "T-39.00".State.Tank_inloading OR ("T-33.00".State.Tank_inloading AND "T-33.00".Cmd.Inload_Select_Tank_1) OR ("T-34.00".State.Tank_inloading AND "T-34.00".Cmd.Inload_Select_Tank_1) OR ("T-35.00".State.Tank_inloading AND "T-35.00".Cmd.Inload_Select_Tank_1) OR ("T-84.00".State.Tank_inloading AND "T-84.00".Cmd.Inload_Select_Tank_1),
             Transfer_Busy := "T-24.00".State.Ready_For_Transfer OR "T-24.00".Out_AV_Transfer,
             CIP_En := NOT "Gen_Storage"."THE5 CIP"."CIP Request" AND NOT "T-24.00".CIP_Line_Req AND NOT "T-33.00".State."CIP Req" AND NOT "T-34.00".State."CIP Req" AND NOT "T-35.00".State."CIP Req" AND NOT "T-81.00".State."CIP Req" AND NOT "T-84.00".State."CIP Req" AND NOT "T-85.00".State."CIP Req",
             CIP_Tank_Req => "Mix_to_CIP".CIP_Request."T-79.00_CIP_Tank_Request",
             CIP_Line_Req => "Mix_to_CIP".CIP_Request."T-79.00_CIP_Line_Request",
             CIP_LineOK => "Mix_to_CIP".CIP_Line_OK."T-79.00_CIP_LineOK");
END_REGION

REGION Network 49: T-79 Valve
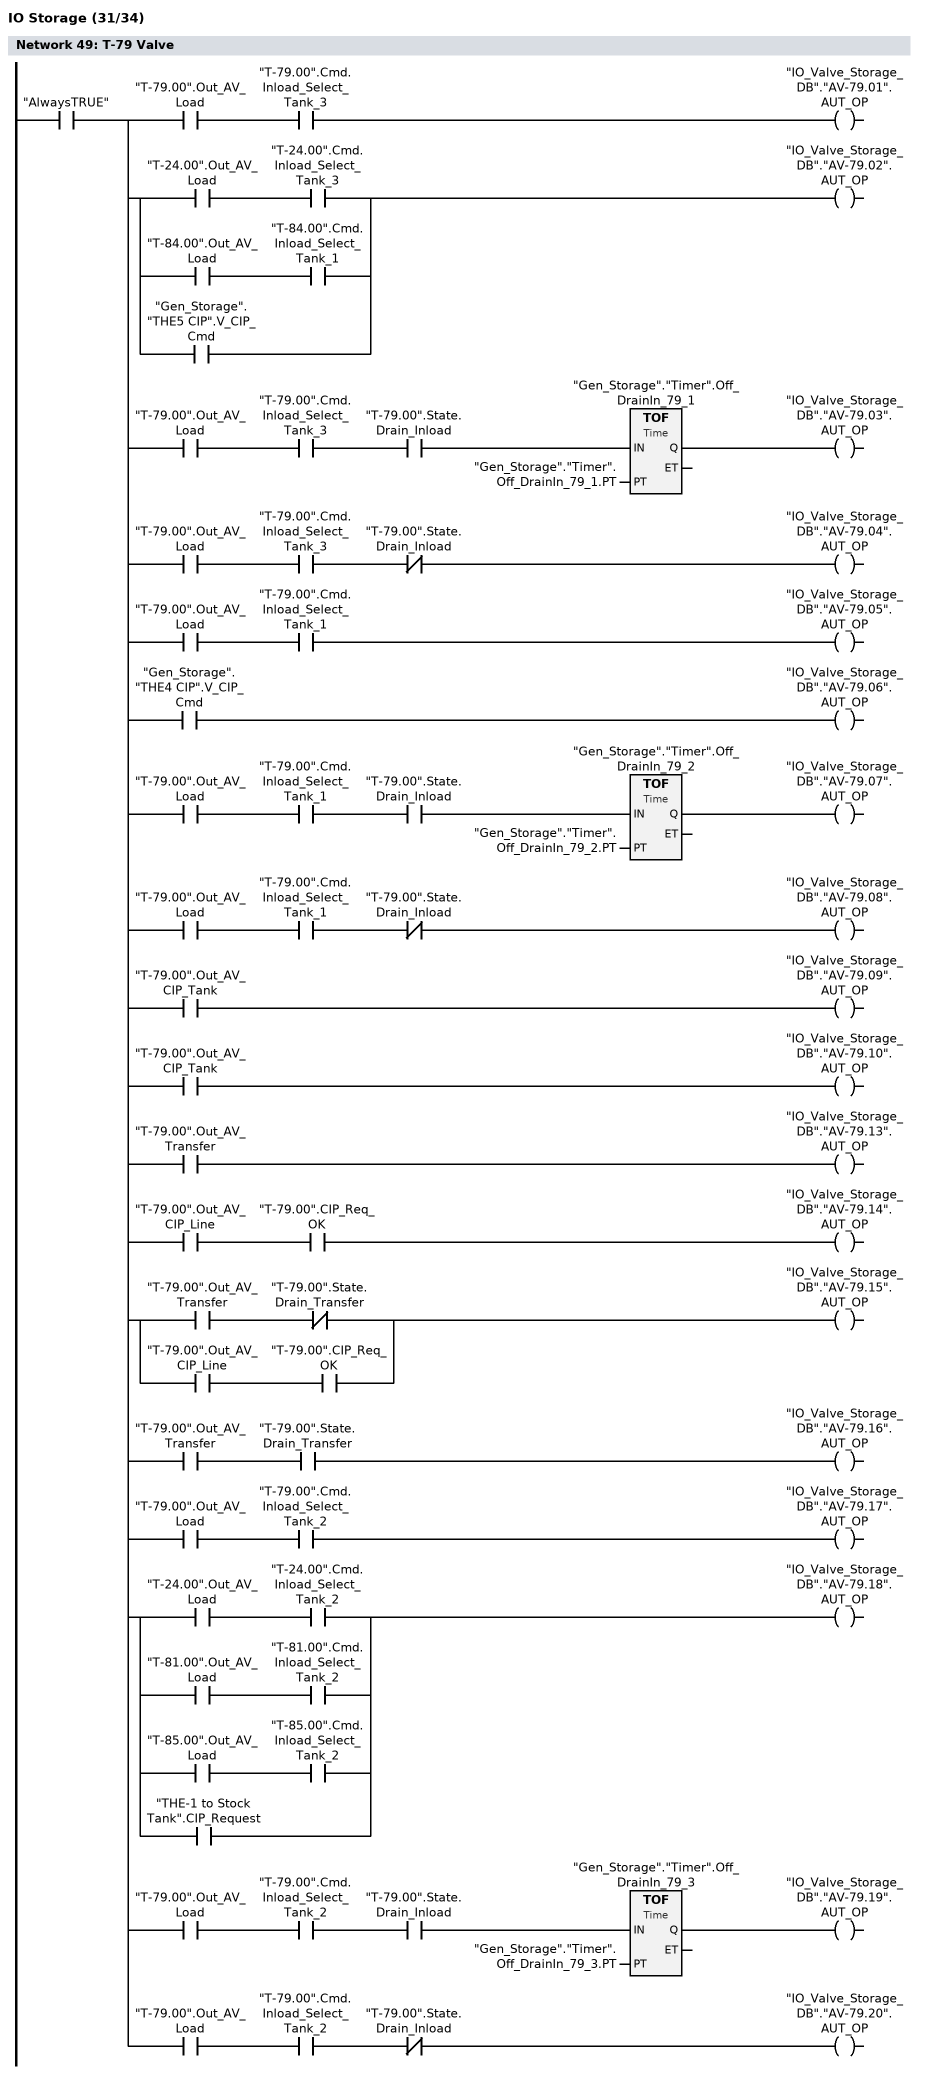
   RUNG wire#powerrail
      Contact( "AlwaysTRUE" )
      wire#w1
      Contact( "T-79.00".Out_AV_Load )
      Contact( "T-79.00".Cmd.Inload_Select_Tank_3 )
      Coil( "IO_Valve_Storage_DB"."AV-79.01".AUT_OP )
   END_RUNG
   RUNG wire#w1
      Contact( "T-24.00".Out_AV_Load )
      Contact( "T-24.00".Cmd.Inload_Select_Tank_3 )
      wire#w2
      Coil( "IO_Valve_Storage_DB"."AV-79.02".AUT_OP )
   END_RUNG
   RUNG wire#w1
      Contact( "T-84.00".Out_AV_Load )
      Contact( "T-84.00".Cmd.Inload_Select_Tank_1 )
   END_RUNG wire#w2
   RUNG wire#w1
      Contact( "Gen_Storage"."THE5 CIP".V_CIP_Cmd )
   END_RUNG wire#w2
   RUNG wire#w1
      Contact( "T-79.00".Out_AV_Load )
      Contact( "T-79.00".Cmd.Inload_Select_Tank_3 )
      Contact( "T-79.00".State.Drain_Inload )
      { S7_Templates := "time_type := Time" } "Gen_Storage"."Timer".Off_DrainIn_79_1.TOF(pt := "Gen_Storage"."Timer".Off_DrainIn_79_1.PT, et =>)
      Coil( "IO_Valve_Storage_DB"."AV-79.03".AUT_OP )
   END_RUNG
   RUNG wire#w1
      Contact( "T-79.00".Out_AV_Load )
      Contact( "T-79.00".Cmd.Inload_Select_Tank_3 )
      I_Contact( "T-79.00".State.Drain_Inload )
      Coil( "IO_Valve_Storage_DB"."AV-79.04".AUT_OP )
   END_RUNG
   RUNG wire#w1
      Contact( "T-79.00".Out_AV_Load )
      Contact( "T-79.00".Cmd.Inload_Select_Tank_1 )
      Coil( "IO_Valve_Storage_DB"."AV-79.05".AUT_OP )
   END_RUNG
   RUNG wire#w1
      Contact( "Gen_Storage"."THE4 CIP".V_CIP_Cmd )
      Coil( "IO_Valve_Storage_DB"."AV-79.06".AUT_OP )
   END_RUNG
   RUNG wire#w1
      Contact( "T-79.00".Out_AV_Load )
      Contact( "T-79.00".Cmd.Inload_Select_Tank_1 )
      Contact( "T-79.00".State.Drain_Inload )
      { S7_Templates := "time_type := Time" } "Gen_Storage"."Timer".Off_DrainIn_79_2.TOF(pt := "Gen_Storage"."Timer".Off_DrainIn_79_2.PT, et =>)
      Coil( "IO_Valve_Storage_DB"."AV-79.07".AUT_OP )
   END_RUNG
   RUNG wire#w1
      Contact( "T-79.00".Out_AV_Load )
      Contact( "T-79.00".Cmd.Inload_Select_Tank_1 )
      I_Contact( "T-79.00".State.Drain_Inload )
      Coil( "IO_Valve_Storage_DB"."AV-79.08".AUT_OP )
   END_RUNG
   RUNG wire#w1
      Contact( "T-79.00".Out_AV_CIP_Tank )
      Coil( "IO_Valve_Storage_DB"."AV-79.09".AUT_OP )
   END_RUNG
   RUNG wire#w1
      Contact( "T-79.00".Out_AV_CIP_Tank )
      Coil( "IO_Valve_Storage_DB"."AV-79.10".AUT_OP )
   END_RUNG
   RUNG wire#w1
      Contact( "T-79.00".Out_AV_Transfer )
      Coil( "IO_Valve_Storage_DB"."AV-79.13".AUT_OP )
   END_RUNG
   RUNG wire#w1
      Contact( "T-79.00".Out_AV_CIP_Line )
      Contact( "T-79.00".CIP_Req_OK )
      Coil( "IO_Valve_Storage_DB"."AV-79.14".AUT_OP )
   END_RUNG
   RUNG wire#w1
      Contact( "T-79.00".Out_AV_Transfer )
      I_Contact( "T-79.00".State.Drain_Transfer )
      wire#w3
      Coil( "IO_Valve_Storage_DB"."AV-79.15".AUT_OP )
   END_RUNG
   RUNG wire#w1
      Contact( "T-79.00".Out_AV_CIP_Line )
      Contact( "T-79.00".CIP_Req_OK )
   END_RUNG wire#w3
   RUNG wire#w1
      Contact( "T-79.00".Out_AV_Transfer )
      Contact( "T-79.00".State.Drain_Transfer )
      Coil( "IO_Valve_Storage_DB"."AV-79.16".AUT_OP )
   END_RUNG
   RUNG wire#w1
      Contact( "T-79.00".Out_AV_Load )
      Contact( "T-79.00".Cmd.Inload_Select_Tank_2 )
      Coil( "IO_Valve_Storage_DB"."AV-79.17".AUT_OP )
   END_RUNG
   RUNG wire#w1
      Contact( "T-24.00".Out_AV_Load )
      Contact( "T-24.00".Cmd.Inload_Select_Tank_2 )
      wire#w4
      Coil( "IO_Valve_Storage_DB"."AV-79.18".AUT_OP )
   END_RUNG
   RUNG wire#w1
      Contact( "T-81.00".Out_AV_Load )
      Contact( "T-81.00".Cmd.Inload_Select_Tank_2 )
   END_RUNG wire#w4
   RUNG wire#w1
      Contact( "T-85.00".Out_AV_Load )
      Contact( "T-85.00".Cmd.Inload_Select_Tank_2 )
   END_RUNG wire#w4
   RUNG wire#w1
      Contact( "THE-1 to Stock Tank".CIP_Request )
   END_RUNG wire#w4
   RUNG wire#w1
      Contact( "T-79.00".Out_AV_Load )
      Contact( "T-79.00".Cmd.Inload_Select_Tank_2 )
      Contact( "T-79.00".State.Drain_Inload )
      { S7_Templates := "time_type := Time" } "Gen_Storage"."Timer".Off_DrainIn_79_3.TOF(pt := "Gen_Storage"."Timer".Off_DrainIn_79_3.PT, et =>)
      Coil( "IO_Valve_Storage_DB"."AV-79.19".AUT_OP )
   END_RUNG
   RUNG wire#w1
      Contact( "T-79.00".Out_AV_Load )
      Contact( "T-79.00".Cmd.Inload_Select_Tank_2 )
      I_Contact( "T-79.00".State.Drain_Inload )
      Coil( "IO_Valve_Storage_DB"."AV-79.20".AUT_OP )
   END_RUNG
   // the same network as SCL:
   "IO_Valve_Storage_DB"."AV-79.01".AUT_OP := "AlwaysTRUE" AND "T-79.00".Out_AV_Load AND "T-79.00".Cmd.Inload_Select_Tank_3;
   "IO_Valve_Storage_DB"."AV-79.02".AUT_OP := "AlwaysTRUE" AND (("T-24.00".Out_AV_Load AND "T-24.00".Cmd.Inload_Select_Tank_3) OR ("T-84.00".Out_AV_Load AND "T-84.00".Cmd.Inload_Select_Tank_1) OR "Gen_Storage"."THE5 CIP".V_CIP_Cmd);
   "Gen_Storage"."Timer".Off_DrainIn_79_1.TOF(IN := "AlwaysTRUE" AND "T-79.00".Out_AV_Load AND "T-79.00".Cmd.Inload_Select_Tank_3 AND "T-79.00".State.Drain_Inload,
                           PT := "Gen_Storage"."Timer".Off_DrainIn_79_1.PT);
   "IO_Valve_Storage_DB"."AV-79.03".AUT_OP := "Gen_Storage"."Timer".Off_DrainIn_79_1.Q;
   "IO_Valve_Storage_DB"."AV-79.04".AUT_OP := "AlwaysTRUE" AND "T-79.00".Out_AV_Load AND "T-79.00".Cmd.Inload_Select_Tank_3 AND NOT "T-79.00".State.Drain_Inload;
   "IO_Valve_Storage_DB"."AV-79.05".AUT_OP := "AlwaysTRUE" AND "T-79.00".Out_AV_Load AND "T-79.00".Cmd.Inload_Select_Tank_1;
   "IO_Valve_Storage_DB"."AV-79.06".AUT_OP := "AlwaysTRUE" AND "Gen_Storage"."THE4 CIP".V_CIP_Cmd;
   "Gen_Storage"."Timer".Off_DrainIn_79_2.TOF(IN := "AlwaysTRUE" AND "T-79.00".Out_AV_Load AND "T-79.00".Cmd.Inload_Select_Tank_1 AND "T-79.00".State.Drain_Inload,
                           PT := "Gen_Storage"."Timer".Off_DrainIn_79_2.PT);
   "IO_Valve_Storage_DB"."AV-79.07".AUT_OP := "Gen_Storage"."Timer".Off_DrainIn_79_2.Q;
   "IO_Valve_Storage_DB"."AV-79.08".AUT_OP := "AlwaysTRUE" AND "T-79.00".Out_AV_Load AND "T-79.00".Cmd.Inload_Select_Tank_1 AND NOT "T-79.00".State.Drain_Inload;
   "IO_Valve_Storage_DB"."AV-79.09".AUT_OP := "AlwaysTRUE" AND "T-79.00".Out_AV_CIP_Tank;
   "IO_Valve_Storage_DB"."AV-79.10".AUT_OP := "AlwaysTRUE" AND "T-79.00".Out_AV_CIP_Tank;
   "IO_Valve_Storage_DB"."AV-79.13".AUT_OP := "AlwaysTRUE" AND "T-79.00".Out_AV_Transfer;
   "IO_Valve_Storage_DB"."AV-79.14".AUT_OP := "AlwaysTRUE" AND "T-79.00".Out_AV_CIP_Line AND "T-79.00".CIP_Req_OK;
   "IO_Valve_Storage_DB"."AV-79.15".AUT_OP := "AlwaysTRUE" AND (("T-79.00".Out_AV_Transfer AND NOT "T-79.00".State.Drain_Transfer) OR ("T-79.00".Out_AV_CIP_Line AND "T-79.00".CIP_Req_OK));
   "IO_Valve_Storage_DB"."AV-79.16".AUT_OP := "AlwaysTRUE" AND "T-79.00".Out_AV_Transfer AND "T-79.00".State.Drain_Transfer;
   "IO_Valve_Storage_DB"."AV-79.17".AUT_OP := "AlwaysTRUE" AND "T-79.00".Out_AV_Load AND "T-79.00".Cmd.Inload_Select_Tank_2;
   "IO_Valve_Storage_DB"."AV-79.18".AUT_OP := "AlwaysTRUE" AND (("T-24.00".Out_AV_Load AND "T-24.00".Cmd.Inload_Select_Tank_2) OR ("T-81.00".Out_AV_Load AND "T-81.00".Cmd.Inload_Select_Tank_2) OR ("T-85.00".Out_AV_Load AND "T-85.00".Cmd.Inload_Select_Tank_2) OR "THE-1 to Stock Tank".CIP_Request);
   "Gen_Storage"."Timer".Off_DrainIn_79_3.TOF(IN := "AlwaysTRUE" AND "T-79.00".Out_AV_Load AND "T-79.00".Cmd.Inload_Select_Tank_2 AND "T-79.00".State.Drain_Inload,
                           PT := "Gen_Storage"."Timer".Off_DrainIn_79_3.PT);
   "IO_Valve_Storage_DB"."AV-79.19".AUT_OP := "Gen_Storage"."Timer".Off_DrainIn_79_3.Q;
   "IO_Valve_Storage_DB"."AV-79.20".AUT_OP := "AlwaysTRUE" AND "T-79.00".Out_AV_Load AND "T-79.00".Cmd.Inload_Select_Tank_2 AND NOT "T-79.00".State.Drain_Inload;
END_REGION

REGION Network 50: Comm T-79 to THE-1
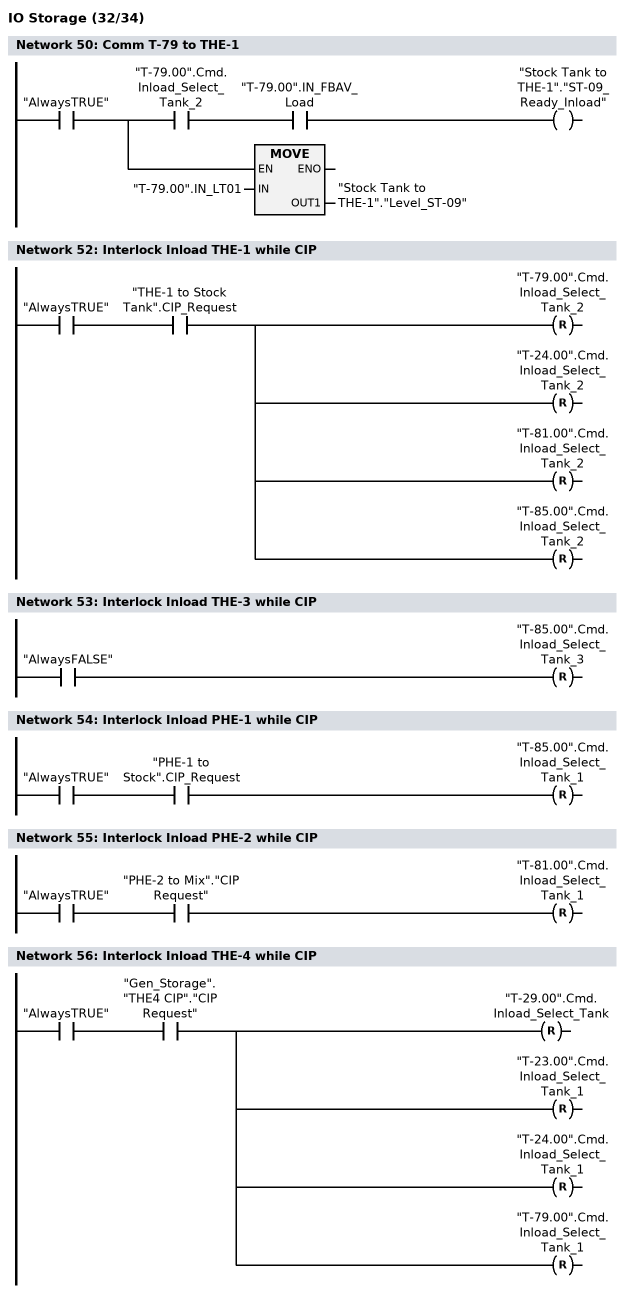
   RUNG wire#powerrail
      Contact( "AlwaysTRUE" )
      wire#w1
      Contact( "T-79.00".Cmd.Inload_Select_Tank_2 )
      Contact( "T-79.00".IN_FBAV_Load )
      Coil( "Stock Tank to THE-1"."ST-09_Ready_Inload" )
   END_RUNG
   RUNG wire#w1
      Move(in := "T-79.00".IN_LT01, out1 => "Stock Tank to THE-1"."Level_ST-09")
   END_RUNG
   // the same network as SCL:
   "Stock Tank to THE-1"."ST-09_Ready_Inload" := "AlwaysTRUE" AND "T-79.00".Cmd.Inload_Select_Tank_2 AND "T-79.00".IN_FBAV_Load;
   IF "AlwaysTRUE" THEN "Stock Tank to THE-1"."Level_ST-09" := "T-79.00".IN_LT01; END_IF;
END_REGION

REGION Network 52: Interlock Inload THE-1 while CIP
   RUNG wire#powerrail
      Contact( "AlwaysTRUE" )
      Contact( "THE-1 to Stock Tank".CIP_Request )
      wire#w1
      R_Coil( "T-79.00".Cmd.Inload_Select_Tank_2 )
   END_RUNG
   RUNG wire#w1
      R_Coil( "T-24.00".Cmd.Inload_Select_Tank_2 )
   END_RUNG
   RUNG wire#w1
      R_Coil( "T-81.00".Cmd.Inload_Select_Tank_2 )
   END_RUNG
   RUNG wire#w1
      R_Coil( "T-85.00".Cmd.Inload_Select_Tank_2 )
   END_RUNG
   // the same network as SCL:
   IF "AlwaysTRUE" AND "THE-1 to Stock Tank".CIP_Request THEN
       "T-79.00".Cmd.Inload_Select_Tank_2 := FALSE;
       "T-24.00".Cmd.Inload_Select_Tank_2 := FALSE;
       "T-81.00".Cmd.Inload_Select_Tank_2 := FALSE;
       "T-85.00".Cmd.Inload_Select_Tank_2 := FALSE;
   END_IF;
END_REGION

REGION Network 53: Interlock Inload THE-3 while CIP
   RUNG wire#powerrail
      Contact( "AlwaysFALSE" )
      R_Coil( "T-85.00".Cmd.Inload_Select_Tank_3 )
   END_RUNG
   // the same network as SCL:
   IF "AlwaysFALSE" THEN "T-85.00".Cmd.Inload_Select_Tank_3 := FALSE; END_IF;
END_REGION

REGION Network 54: Interlock Inload PHE-1 while CIP
   RUNG wire#powerrail
      Contact( "AlwaysTRUE" )
      Contact( "PHE-1 to Stock".CIP_Request )
      R_Coil( "T-85.00".Cmd.Inload_Select_Tank_1 )
   END_RUNG
   // the same network as SCL:
   IF "AlwaysTRUE" AND "PHE-1 to Stock".CIP_Request THEN "T-85.00".Cmd.Inload_Select_Tank_1 := FALSE; END_IF;
END_REGION

REGION Network 55: Interlock Inload PHE-2 while CIP
   RUNG wire#powerrail
      Contact( "AlwaysTRUE" )
      Contact( "PHE-2 to Mix"."CIP Request" )
      R_Coil( "T-81.00".Cmd.Inload_Select_Tank_1 )
   END_RUNG
   // the same network as SCL:
   IF "AlwaysTRUE" AND "PHE-2 to Mix"."CIP Request" THEN "T-81.00".Cmd.Inload_Select_Tank_1 := FALSE; END_IF;
END_REGION

REGION Network 56: Interlock Inload THE-4 while CIP
   RUNG wire#powerrail
      Contact( "AlwaysTRUE" )
      Contact( "Gen_Storage"."THE4 CIP"."CIP Request" )
      wire#w1
      R_Coil( "T-29.00".Cmd.Inload_Select_Tank )
   END_RUNG
   RUNG wire#w1
      R_Coil( "T-23.00".Cmd.Inload_Select_Tank_1 )
   END_RUNG
   RUNG wire#w1
      R_Coil( "T-24.00".Cmd.Inload_Select_Tank_1 )
   END_RUNG
   RUNG wire#w1
      R_Coil( "T-79.00".Cmd.Inload_Select_Tank_1 )
   END_RUNG
   // the same network as SCL:
   IF "AlwaysTRUE" AND "Gen_Storage"."THE4 CIP"."CIP Request" THEN
       "T-29.00".Cmd.Inload_Select_Tank := FALSE;
       "T-23.00".Cmd.Inload_Select_Tank_1 := FALSE;
       "T-24.00".Cmd.Inload_Select_Tank_1 := FALSE;
       "T-79.00".Cmd.Inload_Select_Tank_1 := FALSE;
   END_IF;
END_REGION

REGION Network 57: Interlock Inload THE-5 while CIP
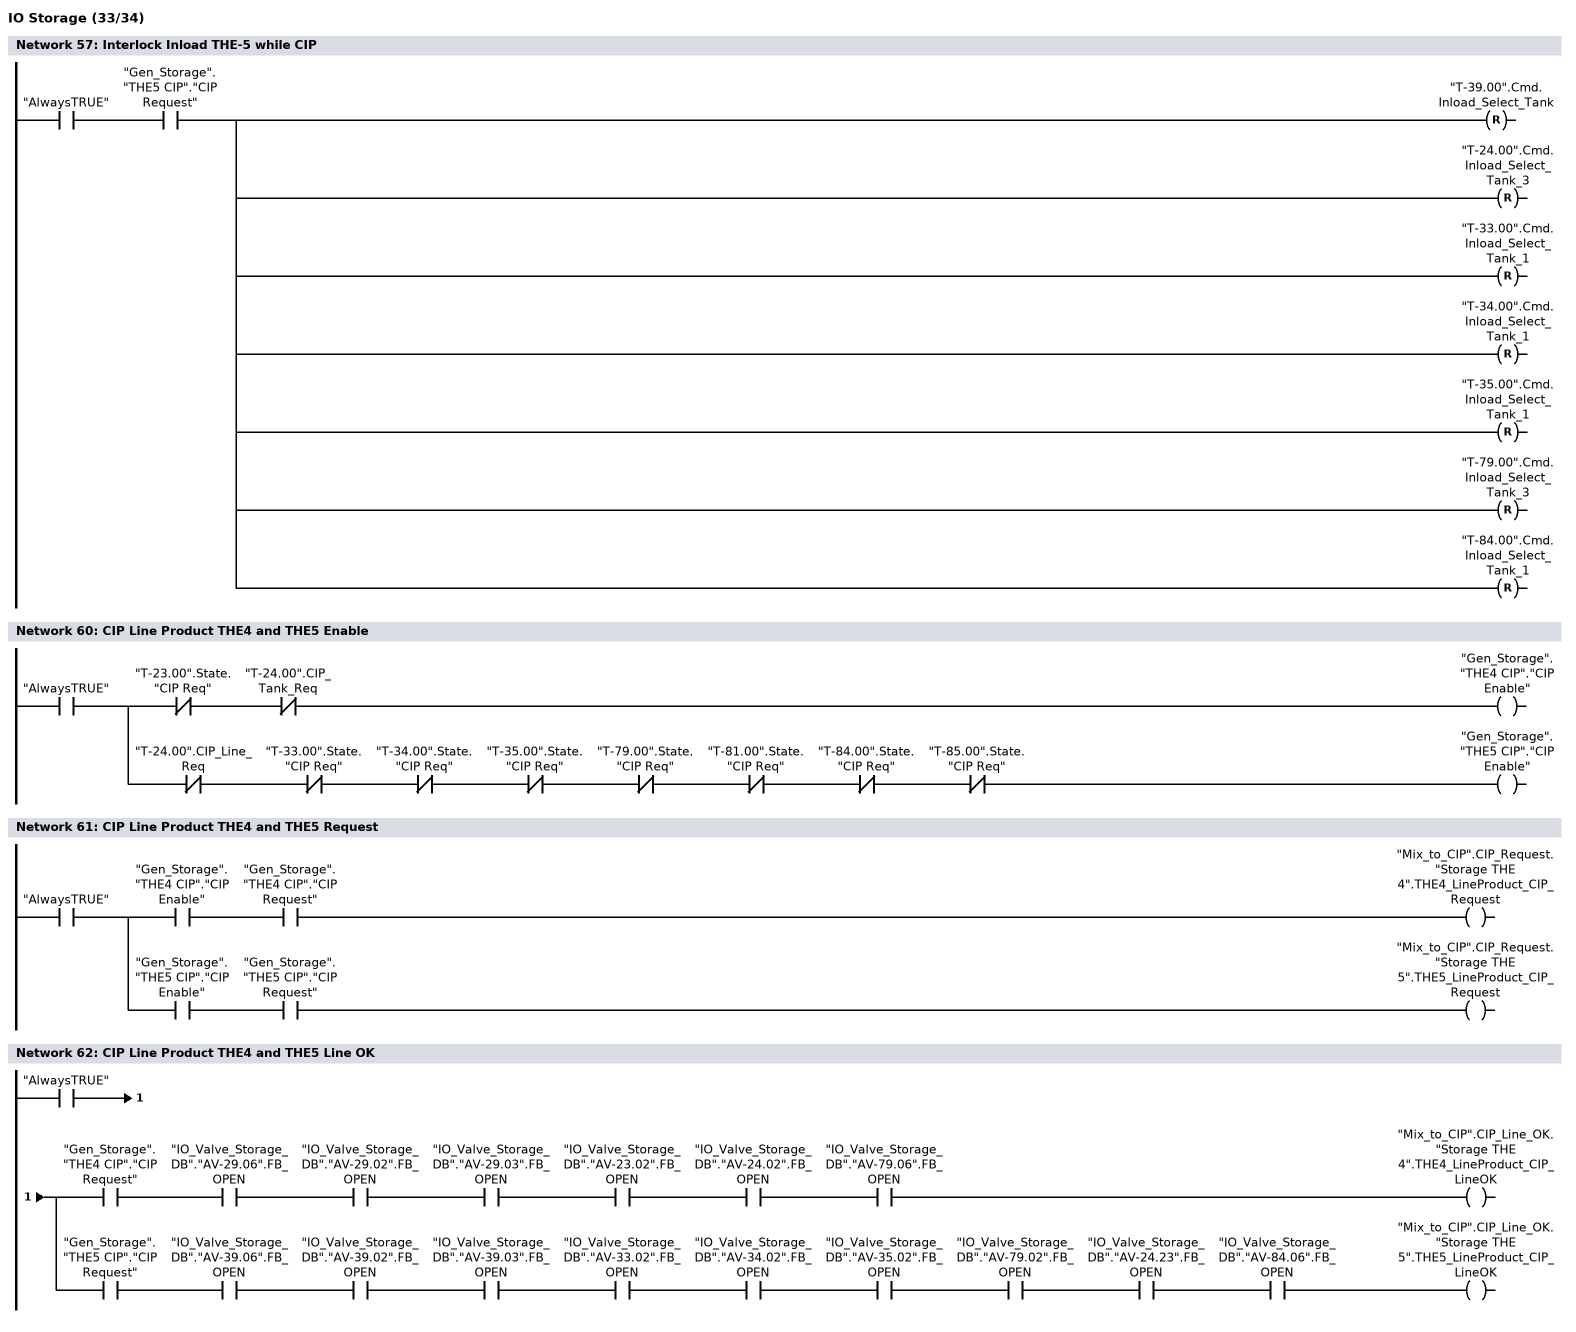
   RUNG wire#powerrail
      Contact( "AlwaysTRUE" )
      Contact( "Gen_Storage"."THE5 CIP"."CIP Request" )
      wire#w1
      R_Coil( "T-39.00".Cmd.Inload_Select_Tank )
   END_RUNG
   RUNG wire#w1
      R_Coil( "T-24.00".Cmd.Inload_Select_Tank_3 )
   END_RUNG
   RUNG wire#w1
      R_Coil( "T-33.00".Cmd.Inload_Select_Tank_1 )
   END_RUNG
   RUNG wire#w1
      R_Coil( "T-34.00".Cmd.Inload_Select_Tank_1 )
   END_RUNG
   RUNG wire#w1
      R_Coil( "T-35.00".Cmd.Inload_Select_Tank_1 )
   END_RUNG
   RUNG wire#w1
      R_Coil( "T-79.00".Cmd.Inload_Select_Tank_3 )
   END_RUNG
   RUNG wire#w1
      R_Coil( "T-84.00".Cmd.Inload_Select_Tank_1 )
   END_RUNG
   // the same network as SCL:
   IF "AlwaysTRUE" AND "Gen_Storage"."THE5 CIP"."CIP Request" THEN
       "T-39.00".Cmd.Inload_Select_Tank := FALSE;
       "T-24.00".Cmd.Inload_Select_Tank_3 := FALSE;
       "T-33.00".Cmd.Inload_Select_Tank_1 := FALSE;
       "T-34.00".Cmd.Inload_Select_Tank_1 := FALSE;
       "T-35.00".Cmd.Inload_Select_Tank_1 := FALSE;
       "T-79.00".Cmd.Inload_Select_Tank_3 := FALSE;
       "T-84.00".Cmd.Inload_Select_Tank_1 := FALSE;
   END_IF;
END_REGION

REGION Network 60: CIP Line Product THE4 and THE5 Enable
   RUNG wire#powerrail
      Contact( "AlwaysTRUE" )
      wire#w1
      I_Contact( "T-23.00".State."CIP Req" )
      I_Contact( "T-24.00".CIP_Tank_Req )
      Coil( "Gen_Storage"."THE4 CIP"."CIP Enable" )
   END_RUNG
   RUNG wire#w1
      I_Contact( "T-24.00".CIP_Line_Req )
      I_Contact( "T-33.00".State."CIP Req" )
      I_Contact( "T-34.00".State."CIP Req" )
      I_Contact( "T-35.00".State."CIP Req" )
      I_Contact( "T-79.00".State."CIP Req" )
      I_Contact( "T-81.00".State."CIP Req" )
      I_Contact( "T-84.00".State."CIP Req" )
      I_Contact( "T-85.00".State."CIP Req" )
      Coil( "Gen_Storage"."THE5 CIP"."CIP Enable" )
   END_RUNG
   // the same network as SCL:
   "Gen_Storage"."THE4 CIP"."CIP Enable" := "AlwaysTRUE" AND NOT "T-23.00".State."CIP Req" AND NOT "T-24.00".CIP_Tank_Req;
   "Gen_Storage"."THE5 CIP"."CIP Enable" := "AlwaysTRUE" AND NOT "T-24.00".CIP_Line_Req AND NOT "T-33.00".State."CIP Req" AND NOT "T-34.00".State."CIP Req" AND NOT "T-35.00".State."CIP Req" AND NOT "T-79.00".State."CIP Req" AND NOT "T-81.00".State."CIP Req" AND NOT "T-84.00".State."CIP Req" AND NOT "T-85.00".State."CIP Req";
END_REGION

REGION Network 61: CIP Line Product THE4 and THE5 Request
   RUNG wire#powerrail
      Contact( "AlwaysTRUE" )
      wire#w1
      Contact( "Gen_Storage"."THE4 CIP"."CIP Enable" )
      Contact( "Gen_Storage"."THE4 CIP"."CIP Request" )
      Coil( "Mix_to_CIP".CIP_Request."Storage THE 4".THE4_LineProduct_CIP_Request )
   END_RUNG
   RUNG wire#w1
      Contact( "Gen_Storage"."THE5 CIP"."CIP Enable" )
      Contact( "Gen_Storage"."THE5 CIP"."CIP Request" )
      Coil( "Mix_to_CIP".CIP_Request."Storage THE 5".THE5_LineProduct_CIP_Request )
   END_RUNG
   // the same network as SCL:
   "Mix_to_CIP".CIP_Request."Storage THE 4".THE4_LineProduct_CIP_Request := "AlwaysTRUE" AND "Gen_Storage"."THE4 CIP"."CIP Enable" AND "Gen_Storage"."THE4 CIP"."CIP Request";
   "Mix_to_CIP".CIP_Request."Storage THE 5".THE5_LineProduct_CIP_Request := "AlwaysTRUE" AND "Gen_Storage"."THE5 CIP"."CIP Enable" AND "Gen_Storage"."THE5 CIP"."CIP Request";
END_REGION

REGION Network 62: CIP Line Product THE4 and THE5 Line OK
   RUNG wire#powerrail
      Contact( "AlwaysTRUE" )
      wire#w1
      Contact( "Gen_Storage"."THE4 CIP"."CIP Request" )
      Contact( "IO_Valve_Storage_DB"."AV-29.06".FB_OPEN )
      Contact( "IO_Valve_Storage_DB"."AV-29.02".FB_OPEN )
      Contact( "IO_Valve_Storage_DB"."AV-29.03".FB_OPEN )
      Contact( "IO_Valve_Storage_DB"."AV-23.02".FB_OPEN )
      Contact( "IO_Valve_Storage_DB"."AV-24.02".FB_OPEN )
      Contact( "IO_Valve_Storage_DB"."AV-79.06".FB_OPEN )
      Coil( "Mix_to_CIP".CIP_Line_OK."Storage THE 4".THE4_LineProduct_CIP_LineOK )
   END_RUNG
   RUNG wire#w1
      Contact( "Gen_Storage"."THE5 CIP"."CIP Request" )
      Contact( "IO_Valve_Storage_DB"."AV-39.06".FB_OPEN )
      Contact( "IO_Valve_Storage_DB"."AV-39.02".FB_OPEN )
      Contact( "IO_Valve_Storage_DB"."AV-39.03".FB_OPEN )
      Contact( "IO_Valve_Storage_DB"."AV-33.02".FB_OPEN )
      Contact( "IO_Valve_Storage_DB"."AV-34.02".FB_OPEN )
      Contact( "IO_Valve_Storage_DB"."AV-35.02".FB_OPEN )
      Contact( "IO_Valve_Storage_DB"."AV-79.02".FB_OPEN )
      Contact( "IO_Valve_Storage_DB"."AV-24.23".FB_OPEN )
      Contact( "IO_Valve_Storage_DB"."AV-84.06".FB_OPEN )
      Coil( "Mix_to_CIP".CIP_Line_OK."Storage THE 5".THE5_LineProduct_CIP_LineOK )
   END_RUNG
   // the same network as SCL:
   "Mix_to_CIP".CIP_Line_OK."Storage THE 4".THE4_LineProduct_CIP_LineOK := "AlwaysTRUE" AND "Gen_Storage"."THE4 CIP"."CIP Request" AND "IO_Valve_Storage_DB"."AV-29.06".FB_OPEN AND "IO_Valve_Storage_DB"."AV-29.02".FB_OPEN AND "IO_Valve_Storage_DB"."AV-29.03".FB_OPEN AND "IO_Valve_Storage_DB"."AV-23.02".FB_OPEN AND "IO_Valve_Storage_DB"."AV-24.02".FB_OPEN AND "IO_Valve_Storage_DB"."AV-79.06".FB_OPEN;
   "Mix_to_CIP".CIP_Line_OK."Storage THE 5".THE5_LineProduct_CIP_LineOK := "AlwaysTRUE" AND "Gen_Storage"."THE5 CIP"."CIP Request" AND "IO_Valve_Storage_DB"."AV-39.06".FB_OPEN AND "IO_Valve_Storage_DB"."AV-39.02".FB_OPEN AND "IO_Valve_Storage_DB"."AV-39.03".FB_OPEN AND "IO_Valve_Storage_DB"."AV-33.02".FB_OPEN AND "IO_Valve_Storage_DB"."AV-34.02".FB_OPEN AND "IO_Valve_Storage_DB"."AV-35.02".FB_OPEN AND "IO_Valve_Storage_DB"."AV-79.02".FB_OPEN AND "IO_Valve_Storage_DB"."AV-24.23".FB_OPEN AND "IO_Valve_Storage_DB"."AV-84.06".FB_OPEN;
END_REGION

REGION Network 63: CIP Line Product THE4 and THE5 Valve Cmd
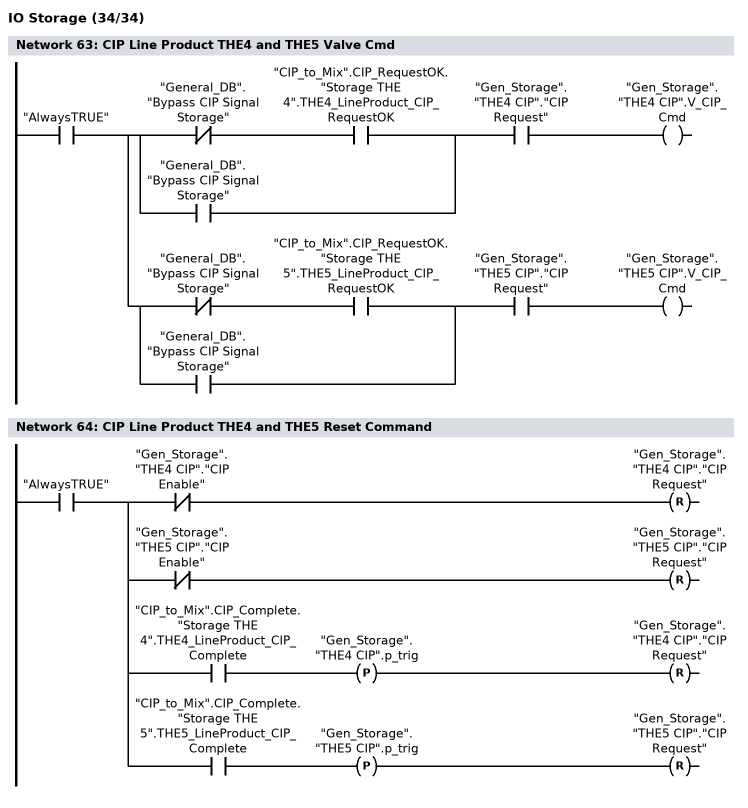
   RUNG wire#powerrail
      Contact( "AlwaysTRUE" )
      wire#w1
      I_Contact( "General_DB"."Bypass CIP Signal Storage" )
      Contact( "CIP_to_Mix".CIP_RequestOK."Storage THE 4".THE4_LineProduct_CIP_RequestOK )
      wire#w2
      Contact( "Gen_Storage"."THE4 CIP"."CIP Request" )
      Coil( "Gen_Storage"."THE4 CIP".V_CIP_Cmd )
   END_RUNG
   RUNG wire#w1
      Contact( "General_DB"."Bypass CIP Signal Storage" )
   END_RUNG wire#w2
   RUNG wire#w1
      I_Contact( "General_DB"."Bypass CIP Signal Storage" )
      Contact( "CIP_to_Mix".CIP_RequestOK."Storage THE 5".THE5_LineProduct_CIP_RequestOK )
      wire#w3
      Contact( "Gen_Storage"."THE5 CIP"."CIP Request" )
      Coil( "Gen_Storage"."THE5 CIP".V_CIP_Cmd )
   END_RUNG
   RUNG wire#w1
      Contact( "General_DB"."Bypass CIP Signal Storage" )
   END_RUNG wire#w3
   // the same network as SCL:
   "Gen_Storage"."THE4 CIP".V_CIP_Cmd := "AlwaysTRUE" AND ((NOT "General_DB"."Bypass CIP Signal Storage" AND "CIP_to_Mix".CIP_RequestOK."Storage THE 4".THE4_LineProduct_CIP_RequestOK) OR "General_DB"."Bypass CIP Signal Storage") AND "Gen_Storage"."THE4 CIP"."CIP Request";
   "Gen_Storage"."THE5 CIP".V_CIP_Cmd := "AlwaysTRUE" AND ((NOT "General_DB"."Bypass CIP Signal Storage" AND "CIP_to_Mix".CIP_RequestOK."Storage THE 5".THE5_LineProduct_CIP_RequestOK) OR "General_DB"."Bypass CIP Signal Storage") AND "Gen_Storage"."THE5 CIP"."CIP Request";
END_REGION

REGION Network 64: CIP Line Product THE4 and THE5 Reset Command
   RUNG wire#powerrail
      Contact( "AlwaysTRUE" )
      wire#w1
      I_Contact( "Gen_Storage"."THE4 CIP"."CIP Enable" )
      R_Coil( "Gen_Storage"."THE4 CIP"."CIP Request" )
   END_RUNG
   RUNG wire#w1
      I_Contact( "Gen_Storage"."THE5 CIP"."CIP Enable" )
      R_Coil( "Gen_Storage"."THE5 CIP"."CIP Request" )
   END_RUNG
   RUNG wire#w1
      Contact( "CIP_to_Mix".CIP_Complete."Storage THE 4".THE4_LineProduct_CIP_Complete )
      P_Trig( "Gen_Storage"."THE4 CIP".p_trig )
      R_Coil( "Gen_Storage"."THE4 CIP"."CIP Request" )
   END_RUNG
   RUNG wire#w1
      Contact( "CIP_to_Mix".CIP_Complete."Storage THE 5".THE5_LineProduct_CIP_Complete )
      P_Trig( "Gen_Storage"."THE5 CIP".p_trig )
      R_Coil( "Gen_Storage"."THE5 CIP"."CIP Request" )
   END_RUNG
   // the same network as SCL:
   IF "AlwaysTRUE" AND NOT "Gen_Storage"."THE4 CIP"."CIP Enable" THEN
       "Gen_Storage"."THE4 CIP"."CIP Request" := FALSE;
   END_IF;
   IF "AlwaysTRUE" AND NOT "Gen_Storage"."THE5 CIP"."CIP Enable" THEN
       "Gen_Storage"."THE5 CIP"."CIP Request" := FALSE;
   END_IF;
   #_w1 := "AlwaysTRUE" AND "CIP_to_Mix".CIP_Complete."Storage THE 4".THE4_LineProduct_CIP_Complete;
   #_w2 := #_w1 AND NOT "Gen_Storage"."THE4 CIP".p_trig;   // rising edge
   "Gen_Storage"."THE4 CIP".p_trig := #_w1;
   IF #_w2 THEN "Gen_Storage"."THE4 CIP"."CIP Request" := FALSE; END_IF;
   #_w3 := "AlwaysTRUE" AND "CIP_to_Mix".CIP_Complete."Storage THE 5".THE5_LineProduct_CIP_Complete;
   #_w4 := #_w3 AND NOT "Gen_Storage"."THE5 CIP".p_trig;   // rising edge
   "Gen_Storage"."THE5 CIP".p_trig := #_w3;
   IF #_w4 THEN "Gen_Storage"."THE5 CIP"."CIP Request" := FALSE; END_IF;
END_REGION
END_FUNCTION

FUNCTION_BLOCK "IO Analog Storage"   // FB11, LAD
{ S7_Optimized_Access := 'FALSE' }
VERSION : 0.1
// stored: AutoNumber true, IsIECCheckEnabled false, SetENOAutomatically false, UDAEnableTagReadback false
   VAR_INPUT
      Init : Bool;
      Reset : Bool;
   END_VAR
   VAR
      "LT-23.01" : "Ana_w_K1K2";
      "LT-24.01" : "Ana_w_K1K2";
      "LT-33.01" : "Ana_w_K1K2";
      "LT-34.01" { S7_SetPoint := 'True'} : "Ana_w_K1K2";
      "LT-35.01" { S7_SetPoint := 'True'} : "Ana_w_K1K2";
      "LT-79.01" { S7_SetPoint := 'True'} : "Ana_w_K1K2";
      "LT-81.01" { S7_SetPoint := 'True'} : "Ana_w_K1K2";
      "LT-84.01" { S7_SetPoint := 'True'} : "Ana_w_K1K2";
      "LT-82.01" { S7_SetPoint := 'True'} : "Ana_w_K1K2";
   END_VAR
BEGIN

REGION Network 1: LT-23.01
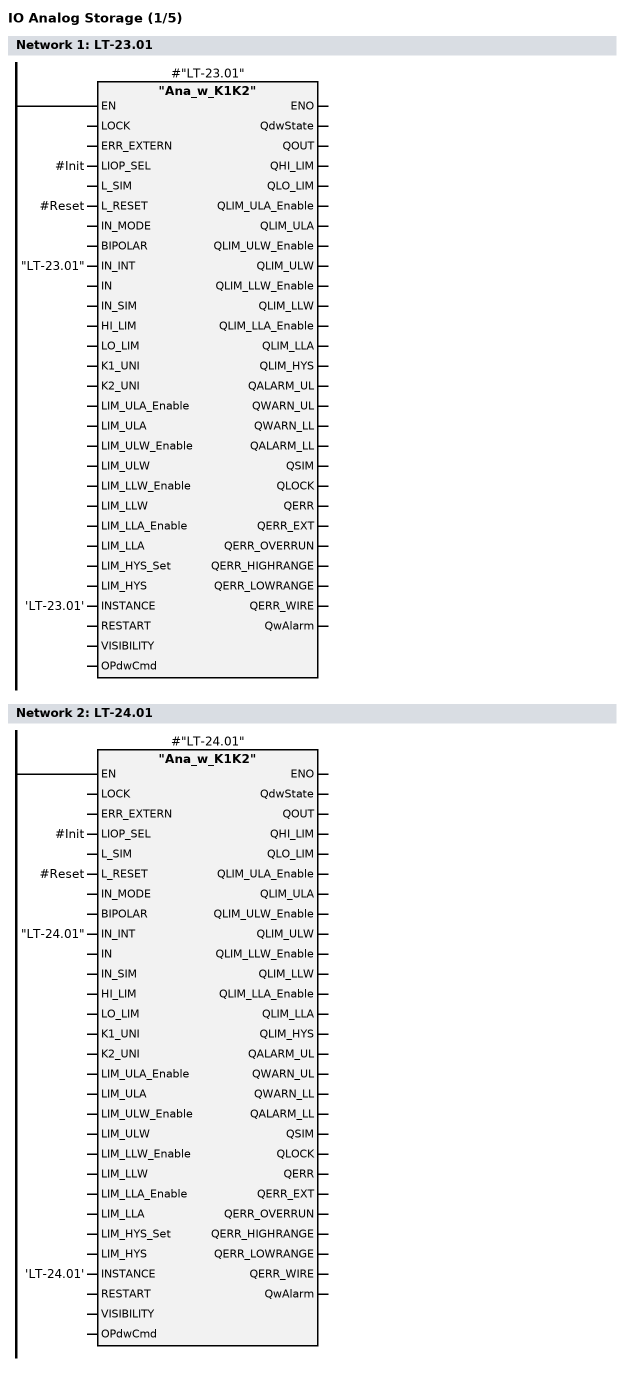
   RUNG wire#powerrail
      #"LT-23.01"(LOCK :=, ERR_EXTERN :=, LIOP_SEL := #Init, L_SIM :=, L_RESET := #Reset, IN_MODE :=, BIPOLAR :=, IN_INT := "LT-23.01", IN :=, IN_SIM :=, HI_LIM :=, LO_LIM :=, K1_UNI :=, K2_UNI :=, LIM_ULA_Enable :=, LIM_ULA :=, LIM_ULW_Enable :=, LIM_ULW :=, LIM_LLW_Enable :=, LIM_LLW :=, LIM_LLA_Enable :=, LIM_LLA :=, LIM_HYS_Set :=, LIM_HYS :=, INSTANCE := 'LT-23.01', RESTART :=, VISIBILITY :=, OPdwCmd :=, QdwState =>, QOUT =>, QHI_LIM =>, QLO_LIM =>, QLIM_ULA_Enable =>, QLIM_ULA =>, QLIM_ULW_Enable =>, QLIM_ULW =>, QLIM_LLW_Enable =>, QLIM_LLW =>, QLIM_LLA_Enable =>, QLIM_LLA =>, QLIM_HYS =>, QALARM_UL =>, QWARN_UL =>, QWARN_LL =>, QALARM_LL =>, QSIM =>, QLOCK =>, QERR =>, QERR_EXT =>, QERR_OVERRUN =>, QERR_HIGHRANGE =>, QERR_LOWRANGE =>, QERR_WIRE =>, QwAlarm =>)
   END_RUNG
   // the same network as SCL:
   #"LT-23.01"(LIOP_SEL := #Init, L_RESET := #Reset, IN_INT := "LT-23.01", INSTANCE := 'LT-23.01');   // "Ana_w_K1K2"
END_REGION

REGION Network 2: LT-24.01
   RUNG wire#powerrail
      #"LT-24.01"(LOCK :=, ERR_EXTERN :=, LIOP_SEL := #Init, L_SIM :=, L_RESET := #Reset, IN_MODE :=, BIPOLAR :=, IN_INT := "LT-24.01", IN :=, IN_SIM :=, HI_LIM :=, LO_LIM :=, K1_UNI :=, K2_UNI :=, LIM_ULA_Enable :=, LIM_ULA :=, LIM_ULW_Enable :=, LIM_ULW :=, LIM_LLW_Enable :=, LIM_LLW :=, LIM_LLA_Enable :=, LIM_LLA :=, LIM_HYS_Set :=, LIM_HYS :=, INSTANCE := 'LT-24.01', RESTART :=, VISIBILITY :=, OPdwCmd :=, QdwState =>, QOUT =>, QHI_LIM =>, QLO_LIM =>, QLIM_ULA_Enable =>, QLIM_ULA =>, QLIM_ULW_Enable =>, QLIM_ULW =>, QLIM_LLW_Enable =>, QLIM_LLW =>, QLIM_LLA_Enable =>, QLIM_LLA =>, QLIM_HYS =>, QALARM_UL =>, QWARN_UL =>, QWARN_LL =>, QALARM_LL =>, QSIM =>, QLOCK =>, QERR =>, QERR_EXT =>, QERR_OVERRUN =>, QERR_HIGHRANGE =>, QERR_LOWRANGE =>, QERR_WIRE =>, QwAlarm =>)
   END_RUNG
   // the same network as SCL:
   #"LT-24.01"(LIOP_SEL := #Init, L_RESET := #Reset, IN_INT := "LT-24.01", INSTANCE := 'LT-24.01');   // "Ana_w_K1K2"
END_REGION

REGION Network 3: LT-33.01
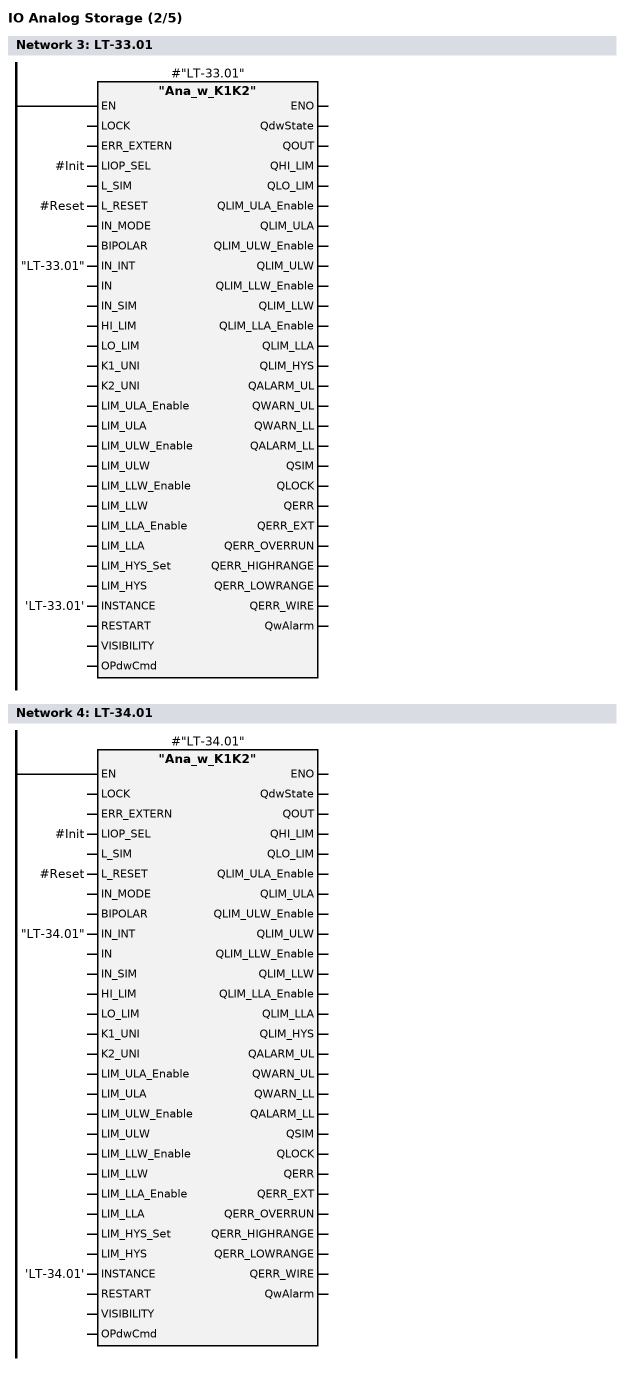
   RUNG wire#powerrail
      #"LT-33.01"(LOCK :=, ERR_EXTERN :=, LIOP_SEL := #Init, L_SIM :=, L_RESET := #Reset, IN_MODE :=, BIPOLAR :=, IN_INT := "LT-33.01", IN :=, IN_SIM :=, HI_LIM :=, LO_LIM :=, K1_UNI :=, K2_UNI :=, LIM_ULA_Enable :=, LIM_ULA :=, LIM_ULW_Enable :=, LIM_ULW :=, LIM_LLW_Enable :=, LIM_LLW :=, LIM_LLA_Enable :=, LIM_LLA :=, LIM_HYS_Set :=, LIM_HYS :=, INSTANCE := 'LT-33.01', RESTART :=, VISIBILITY :=, OPdwCmd :=, QdwState =>, QOUT =>, QHI_LIM =>, QLO_LIM =>, QLIM_ULA_Enable =>, QLIM_ULA =>, QLIM_ULW_Enable =>, QLIM_ULW =>, QLIM_LLW_Enable =>, QLIM_LLW =>, QLIM_LLA_Enable =>, QLIM_LLA =>, QLIM_HYS =>, QALARM_UL =>, QWARN_UL =>, QWARN_LL =>, QALARM_LL =>, QSIM =>, QLOCK =>, QERR =>, QERR_EXT =>, QERR_OVERRUN =>, QERR_HIGHRANGE =>, QERR_LOWRANGE =>, QERR_WIRE =>, QwAlarm =>)
   END_RUNG
   // the same network as SCL:
   #"LT-33.01"(LIOP_SEL := #Init, L_RESET := #Reset, IN_INT := "LT-33.01", INSTANCE := 'LT-33.01');   // "Ana_w_K1K2"
END_REGION

REGION Network 4: LT-34.01
   RUNG wire#powerrail
      #"LT-34.01"(LOCK :=, ERR_EXTERN :=, LIOP_SEL := #Init, L_SIM :=, L_RESET := #Reset, IN_MODE :=, BIPOLAR :=, IN_INT := "LT-34.01", IN :=, IN_SIM :=, HI_LIM :=, LO_LIM :=, K1_UNI :=, K2_UNI :=, LIM_ULA_Enable :=, LIM_ULA :=, LIM_ULW_Enable :=, LIM_ULW :=, LIM_LLW_Enable :=, LIM_LLW :=, LIM_LLA_Enable :=, LIM_LLA :=, LIM_HYS_Set :=, LIM_HYS :=, INSTANCE := 'LT-34.01', RESTART :=, VISIBILITY :=, OPdwCmd :=, QdwState =>, QOUT =>, QHI_LIM =>, QLO_LIM =>, QLIM_ULA_Enable =>, QLIM_ULA =>, QLIM_ULW_Enable =>, QLIM_ULW =>, QLIM_LLW_Enable =>, QLIM_LLW =>, QLIM_LLA_Enable =>, QLIM_LLA =>, QLIM_HYS =>, QALARM_UL =>, QWARN_UL =>, QWARN_LL =>, QALARM_LL =>, QSIM =>, QLOCK =>, QERR =>, QERR_EXT =>, QERR_OVERRUN =>, QERR_HIGHRANGE =>, QERR_LOWRANGE =>, QERR_WIRE =>, QwAlarm =>)
   END_RUNG
   // the same network as SCL:
   #"LT-34.01"(LIOP_SEL := #Init, L_RESET := #Reset, IN_INT := "LT-34.01", INSTANCE := 'LT-34.01');   // "Ana_w_K1K2"
END_REGION

REGION Network 5: LT-35.01
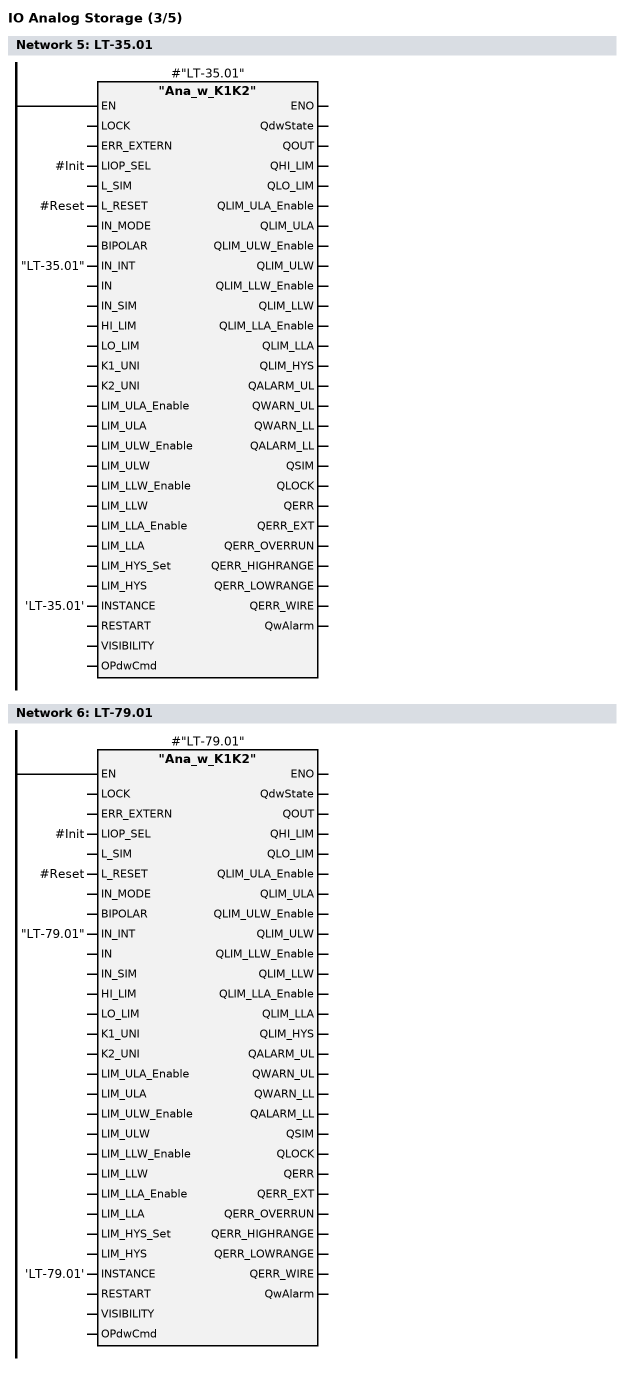
   RUNG wire#powerrail
      #"LT-35.01"(LOCK :=, ERR_EXTERN :=, LIOP_SEL := #Init, L_SIM :=, L_RESET := #Reset, IN_MODE :=, BIPOLAR :=, IN_INT := "LT-35.01", IN :=, IN_SIM :=, HI_LIM :=, LO_LIM :=, K1_UNI :=, K2_UNI :=, LIM_ULA_Enable :=, LIM_ULA :=, LIM_ULW_Enable :=, LIM_ULW :=, LIM_LLW_Enable :=, LIM_LLW :=, LIM_LLA_Enable :=, LIM_LLA :=, LIM_HYS_Set :=, LIM_HYS :=, INSTANCE := 'LT-35.01', RESTART :=, VISIBILITY :=, OPdwCmd :=, QdwState =>, QOUT =>, QHI_LIM =>, QLO_LIM =>, QLIM_ULA_Enable =>, QLIM_ULA =>, QLIM_ULW_Enable =>, QLIM_ULW =>, QLIM_LLW_Enable =>, QLIM_LLW =>, QLIM_LLA_Enable =>, QLIM_LLA =>, QLIM_HYS =>, QALARM_UL =>, QWARN_UL =>, QWARN_LL =>, QALARM_LL =>, QSIM =>, QLOCK =>, QERR =>, QERR_EXT =>, QERR_OVERRUN =>, QERR_HIGHRANGE =>, QERR_LOWRANGE =>, QERR_WIRE =>, QwAlarm =>)
   END_RUNG
   // the same network as SCL:
   #"LT-35.01"(LIOP_SEL := #Init, L_RESET := #Reset, IN_INT := "LT-35.01", INSTANCE := 'LT-35.01');   // "Ana_w_K1K2"
END_REGION

REGION Network 6: LT-79.01
   RUNG wire#powerrail
      #"LT-79.01"(LOCK :=, ERR_EXTERN :=, LIOP_SEL := #Init, L_SIM :=, L_RESET := #Reset, IN_MODE :=, BIPOLAR :=, IN_INT := "LT-79.01", IN :=, IN_SIM :=, HI_LIM :=, LO_LIM :=, K1_UNI :=, K2_UNI :=, LIM_ULA_Enable :=, LIM_ULA :=, LIM_ULW_Enable :=, LIM_ULW :=, LIM_LLW_Enable :=, LIM_LLW :=, LIM_LLA_Enable :=, LIM_LLA :=, LIM_HYS_Set :=, LIM_HYS :=, INSTANCE := 'LT-79.01', RESTART :=, VISIBILITY :=, OPdwCmd :=, QdwState =>, QOUT =>, QHI_LIM =>, QLO_LIM =>, QLIM_ULA_Enable =>, QLIM_ULA =>, QLIM_ULW_Enable =>, QLIM_ULW =>, QLIM_LLW_Enable =>, QLIM_LLW =>, QLIM_LLA_Enable =>, QLIM_LLA =>, QLIM_HYS =>, QALARM_UL =>, QWARN_UL =>, QWARN_LL =>, QALARM_LL =>, QSIM =>, QLOCK =>, QERR =>, QERR_EXT =>, QERR_OVERRUN =>, QERR_HIGHRANGE =>, QERR_LOWRANGE =>, QERR_WIRE =>, QwAlarm =>)
   END_RUNG
   // the same network as SCL:
   #"LT-79.01"(LIOP_SEL := #Init, L_RESET := #Reset, IN_INT := "LT-79.01", INSTANCE := 'LT-79.01');   // "Ana_w_K1K2"
END_REGION

REGION Network 7: LT-81.01
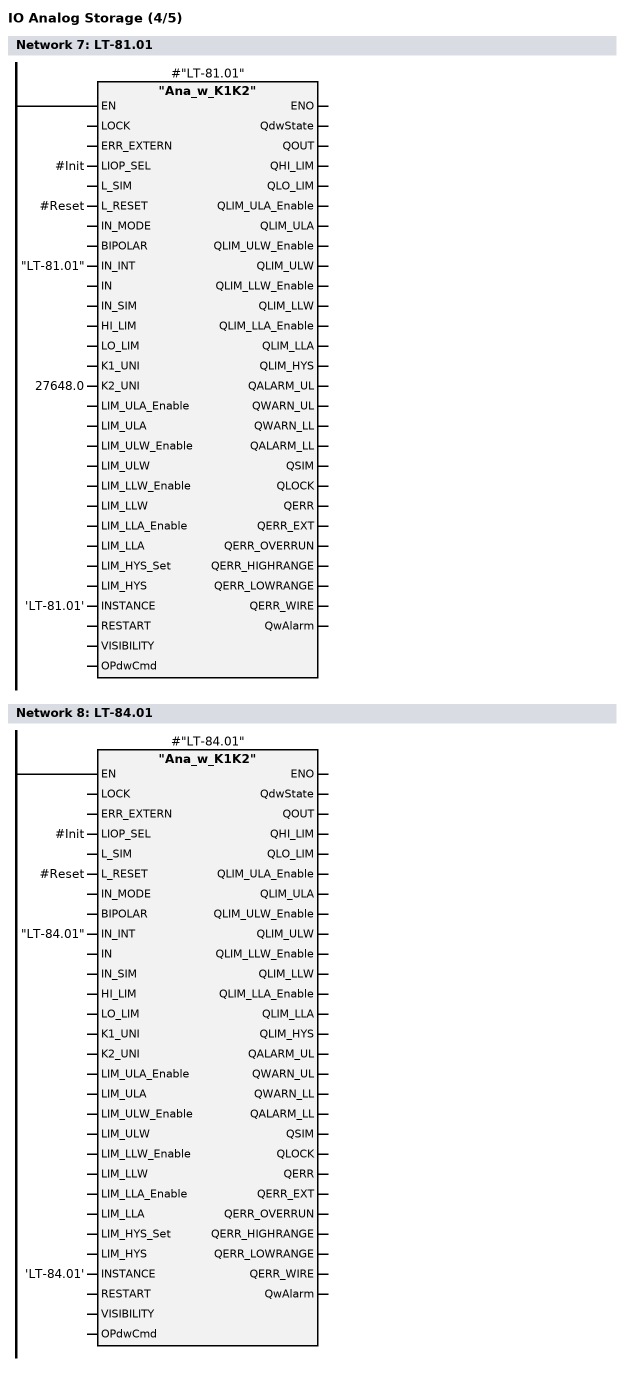
   RUNG wire#powerrail
      #"LT-81.01"(LOCK :=, ERR_EXTERN :=, LIOP_SEL := #Init, L_SIM :=, L_RESET := #Reset, IN_MODE :=, BIPOLAR :=, IN_INT := "LT-81.01", IN :=, IN_SIM :=, HI_LIM :=, LO_LIM :=, K1_UNI :=, K2_UNI := 27648.0, LIM_ULA_Enable :=, LIM_ULA :=, LIM_ULW_Enable :=, LIM_ULW :=, LIM_LLW_Enable :=, LIM_LLW :=, LIM_LLA_Enable :=, LIM_LLA :=, LIM_HYS_Set :=, LIM_HYS :=, INSTANCE := 'LT-81.01', RESTART :=, VISIBILITY :=, OPdwCmd :=, QdwState =>, QOUT =>, QHI_LIM =>, QLO_LIM =>, QLIM_ULA_Enable =>, QLIM_ULA =>, QLIM_ULW_Enable =>, QLIM_ULW =>, QLIM_LLW_Enable =>, QLIM_LLW =>, QLIM_LLA_Enable =>, QLIM_LLA =>, QLIM_HYS =>, QALARM_UL =>, QWARN_UL =>, QWARN_LL =>, QALARM_LL =>, QSIM =>, QLOCK =>, QERR =>, QERR_EXT =>, QERR_OVERRUN =>, QERR_HIGHRANGE =>, QERR_LOWRANGE =>, QERR_WIRE =>, QwAlarm =>)
   END_RUNG
   // the same network as SCL:
   #"LT-81.01"(LIOP_SEL := #Init,   // "Ana_w_K1K2"
               L_RESET := #Reset,
               IN_INT := "LT-81.01",
               K2_UNI := 27648.0,
               INSTANCE := 'LT-81.01');
END_REGION

REGION Network 8: LT-84.01
   RUNG wire#powerrail
      #"LT-84.01"(LOCK :=, ERR_EXTERN :=, LIOP_SEL := #Init, L_SIM :=, L_RESET := #Reset, IN_MODE :=, BIPOLAR :=, IN_INT := "LT-84.01", IN :=, IN_SIM :=, HI_LIM :=, LO_LIM :=, K1_UNI :=, K2_UNI :=, LIM_ULA_Enable :=, LIM_ULA :=, LIM_ULW_Enable :=, LIM_ULW :=, LIM_LLW_Enable :=, LIM_LLW :=, LIM_LLA_Enable :=, LIM_LLA :=, LIM_HYS_Set :=, LIM_HYS :=, INSTANCE := 'LT-84.01', RESTART :=, VISIBILITY :=, OPdwCmd :=, QdwState =>, QOUT =>, QHI_LIM =>, QLO_LIM =>, QLIM_ULA_Enable =>, QLIM_ULA =>, QLIM_ULW_Enable =>, QLIM_ULW =>, QLIM_LLW_Enable =>, QLIM_LLW =>, QLIM_LLA_Enable =>, QLIM_LLA =>, QLIM_HYS =>, QALARM_UL =>, QWARN_UL =>, QWARN_LL =>, QALARM_LL =>, QSIM =>, QLOCK =>, QERR =>, QERR_EXT =>, QERR_OVERRUN =>, QERR_HIGHRANGE =>, QERR_LOWRANGE =>, QERR_WIRE =>, QwAlarm =>)
   END_RUNG
   // the same network as SCL:
   #"LT-84.01"(LIOP_SEL := #Init, L_RESET := #Reset, IN_INT := "LT-84.01", INSTANCE := 'LT-84.01');   // "Ana_w_K1K2"
END_REGION

REGION Network 9: LT-82.01
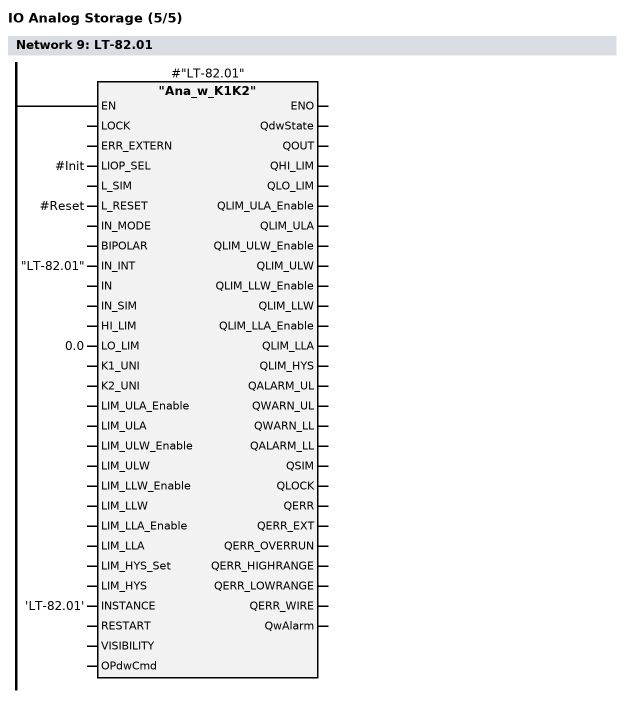
   RUNG wire#powerrail
      #"LT-82.01"(LOCK :=, ERR_EXTERN :=, LIOP_SEL := #Init, L_SIM :=, L_RESET := #Reset, IN_MODE :=, BIPOLAR :=, IN_INT := "LT-82.01", IN :=, IN_SIM :=, HI_LIM :=, LO_LIM := 0.0, K1_UNI :=, K2_UNI :=, LIM_ULA_Enable :=, LIM_ULA :=, LIM_ULW_Enable :=, LIM_ULW :=, LIM_LLW_Enable :=, LIM_LLW :=, LIM_LLA_Enable :=, LIM_LLA :=, LIM_HYS_Set :=, LIM_HYS :=, INSTANCE := 'LT-82.01', RESTART :=, VISIBILITY :=, OPdwCmd :=, QdwState =>, QOUT =>, QHI_LIM =>, QLO_LIM =>, QLIM_ULA_Enable =>, QLIM_ULA =>, QLIM_ULW_Enable =>, QLIM_ULW =>, QLIM_LLW_Enable =>, QLIM_LLW =>, QLIM_LLA_Enable =>, QLIM_LLA =>, QLIM_HYS =>, QALARM_UL =>, QWARN_UL =>, QWARN_LL =>, QALARM_LL =>, QSIM =>, QLOCK =>, QERR =>, QERR_EXT =>, QERR_OVERRUN =>, QERR_HIGHRANGE =>, QERR_LOWRANGE =>, QERR_WIRE =>, QwAlarm =>)
   END_RUNG
   // the same network as SCL:
   #"LT-82.01"(LIOP_SEL := #Init,   // "Ana_w_K1K2"
               L_RESET := #Reset,
               IN_INT := "LT-82.01",
               LO_LIM := 0.0,
               INSTANCE := 'LT-82.01');
END_REGION
END_FUNCTION_BLOCK

FUNCTION_BLOCK "IO_Valve_Storage"   // FB1, LAD
{ S7_Optimized_Access := 'FALSE' }
VERSION : 0.1
// stored: AutoNumber true, IsIECCheckEnabled false, SetENOAutomatically false, UDAEnableTagReadback false
   VAR_INPUT
      lock : Bool;
      Init : Bool;
      Reset : Bool;
   END_VAR
   VAR
      "AV-23.01" { S7_SetPoint := 'True'} : "Valve";   // AUTO BUTTERFLY VALVE MAIN INLET PRODUCT TO STORAGE TANK T-23.00
      "AV-23.02" { S7_SetPoint := 'True'} : "Valve";   // AUTO BUTTERFLY VALVE CIP SUPPLY TO STORAGE TANK T-23.00 VIA PIPE INLET
      "AV-23.03" { S7_SetPoint := 'True'} : "Valve";   // AUTO BUTTERFLY VALVE INLET PRODUCT TO STORAGE TANK T-23.00
      "AV-23.04" { S7_SetPoint := 'True'} : "Valve";   // AUTO BUTTERFLY VALVE INLET PRODUCT FROM JBT TO STORAGE TANKS
      "AV-23.05" { S7_SetPoint := 'True'} : "Valve";   // AUTO BUTTERFLY VALVE INLET CIP PRODUCT FROM THE-4 TO STORAGE
      "AV-23.06" { S7_SetPoint := 'True'} : "Valve";   // AUTO BUTTERFLY VALVE OUTLET PRODUCT FROM STORAGE TANK T-23.00
      "AV-23.07" { S7_SetPoint := 'True'} : "Valve";   // AUTO BUTTERFLY VALVE CIP SUPPLY LINE STORAGE TANK T-23.00
      "AV-23.08" { S7_SetPoint := 'True'} : "Valve";   // AUTO BUTTERFLY VALVE CIP SUPPLY STORAGE TANK T-23.00 VIA SPRAY BALL
      "AV-24.01" { S7_SetPoint := 'True'} : "Valve";   // AUTO BUTTERFLY VALVE MAIN INLET PRODUCT TO STORAGE TANK T-24.00
      "AV-24.02" { S7_SetPoint := 'True'} : "Valve";   // AUTO BUTTERFLY VALVE CIP SUPPLY TO STORAGE TANK T-24.00 VIA PIPE INLET
      "AV-24.03" { S7_SetPoint := 'True'} : "Valve";   // AUTO BUTTERFLY VALVE INLET PRODUCT TO STORAGE TANK T-24.00
      "AV-24.04" { S7_SetPoint := 'True'} : "Valve";   // AUTO BUTTERFLY VALVE OUTLET PRODUCT FROM STORAGE TANK T-24.00
      "AV-24.05" { S7_SetPoint := 'True'} : "Valve";   // AUTO BUTTERFLY VALVE CIP SUPPLY LINE STORAGE TANK T-24.00
      "AV-24.06" { S7_SetPoint := 'True'} : "Valve";   // AUTO BUTTERFLY VALVE CIP SUPPLY STORAGE TANK T-24.00 VIA SPRAY BALL
      "AV-24.13" { S7_SetPoint := 'True'} : "Valve";   // AUTO BUTTERFLY VALVE MAIN INLET PRODUCT TO STORAGE TANK T-25.00
      "AV-24.14" { S7_SetPoint := 'True'} : "Valve";   // AUTO BUTTERFLY VALVE CIP SUPPLY TO STORAGE TANK T-25.00 VIA PIPE INLET
      "AV-29.01" { S7_SetPoint := 'True'} : "Valve";   // AUTO BUTTERFLY VALVE INLET PRODUCT TO STORAGE TANK T-25.00
      "AV-29.02" { S7_SetPoint := 'True'} : "Valve";   // AUTO BUTTERFLY VALVE OUTLET PRODUCT FROM STORAGE TANK T-25.00
      "AV-29.03" { S7_SetPoint := 'True'} : "Valve";   // AUTO BUTTERFLY VALVE CIP SUPPLY LINE STORAGE TANK T-25.00
      "AV-29.04" { S7_SetPoint := 'True'} : "Valve";   // AUTO BUTTERFLY VALVE CIP SUPPLY STORAGE TANK T-25.00 VIA SPRAY BALL
      "AV-29.06" { S7_SetPoint := 'True'} : "Valve";   // AUTO BUTTERFLY VALVE CIP SUPPLY STORAGE TANK T-25.00 VIA SPRAY BALL
      "AV-33.01" { S7_SetPoint := 'True'} : "Valve";   // AUTO BUTTERFLY VALVE CIP SUPPLY STORAGE TANKS FROM CIP SUPPLY LINE 3
      "AV-33.02" { S7_SetPoint := 'True'} : "Valve";   // AUTO BUTTERFLY VALVE CIP SUPPLY STORAGE TANK THE-4 JBT FROM CIP SUPPLY LINE 3
      "AV-33.03" { S7_SetPoint := 'True'} : "Valve";   // AUTO BUTTERFLY VALVE CIP SUPPLY STORAGE TANK THE-5 JBT FROM CIP SUPPLY LINE 3
      "AV-33.04" { S7_SetPoint := 'True'} : "Valve";   // AUTO BUTTERFLY VALVE MAIN CIP SUPPLY PRODUCT FROM THE-4 TO STORAGE
      "AV-33.05" { S7_SetPoint := 'True'} : "Valve";   // AUTO BUTTERFLY VALVE MAIN CIP SUPPLY TO STORAGE TANK T-23.00
      "AV-33.06" { S7_SetPoint := 'True'} : "Valve";   // AUTO BUTTERFLY VALVE MAIN CIP SUPPLY LINE STORAGE TANK T-23.00
      "AV-33.07" { S7_SetPoint := 'True'} : "Valve";   // AUTO BUTTERFLY VALVE MAIN CIP SUPPLY TO STORAGE TANK T-24.00
      "AV-33.08" { S7_SetPoint := 'True'} : "Valve";   // AUTO BUTTERFLY VALVE MAIN CIP SUPPLY LINE STORAGE TANK T-24.00
      "AV-33.09" { S7_SetPoint := 'True'} : "Valve";   // AUTO BUTTERFLY VALVE MAIN CIP SUPPLY TO STORAGE TANK T-25.00
      "AV-33.10" { S7_SetPoint := 'True'} : "Valve";
      "AV-33.11" { S7_SetPoint := 'True'} : "Valve";
      "AV-34.01" { S7_SetPoint := 'True'} : "Valve";
      "AV-34.02" { S7_SetPoint := 'True'} : "Valve";
      "AV-34.03" { S7_SetPoint := 'True'} : "Valve";
      "AV-34.04" { S7_SetPoint := 'True'} : "Valve";
      "AV-34.05" { S7_SetPoint := 'True'} : "Valve";
      "AV-34.06" { S7_SetPoint := 'True'} : "Valve";
      "AV-34.07" { S7_SetPoint := 'True'} : "Valve";
      "AV-34.08" { S7_SetPoint := 'True'} : "Valve";
      "AV-34.09" { S7_SetPoint := 'True'} : "Valve";
      "AV-34.10" { S7_SetPoint := 'True'} : "Valve";
      "AV-34.11" { S7_SetPoint := 'True'} : "Valve";
      "AV-34.12" { S7_SetPoint := 'True'} : "Valve";
      "AV-35.01" { S7_SetPoint := 'True'} : "Valve";
      "AV-35.02" { S7_SetPoint := 'True'} : "Valve";
      "AV-35.03" { S7_SetPoint := 'True'} : "Valve";
      "AV-35.04" { S7_SetPoint := 'True'} : "Valve";
      "AV-35.05" { S7_SetPoint := 'True'} : "Valve";
      "AV-35.06" { S7_SetPoint := 'True'} : "Valve";
      "AV-35.07" { S7_SetPoint := 'True'} : "Valve";
      "AV-35.08" { S7_SetPoint := 'True'} : "Valve";
      "AV-39.01" { S7_SetPoint := 'True'} : "Valve";
      "AV-39.02" { S7_SetPoint := 'True'} : "Valve";
      "AV-39.03" { S7_SetPoint := 'True'} : "Valve";
      "AV-39.04" { S7_SetPoint := 'True'} : "Valve";
      "AV-39.06" { S7_SetPoint := 'True'} : "Valve";
      "AV-24.15" { S7_SetPoint := 'True'} : "Valve";
      "AV-24.16" { S7_SetPoint := 'True'} : "Valve";
      "AV-79.01" { S7_SetPoint := 'True'} : "Valve";
      "AV-79.02" { S7_SetPoint := 'True'} : "Valve";
      "AV-79.03" { S7_SetPoint := 'True'} : "Valve";
      "AV-79.04" { S7_SetPoint := 'True'} : "Valve";
      "AV-79.05" { S7_SetPoint := 'True'} : "Valve";
      "AV-79.06" { S7_SetPoint := 'True'} : "Valve";
      "AV-79.07" { S7_SetPoint := 'True'} : "Valve";
      "AV-79.08" { S7_SetPoint := 'True'} : "Valve";
      "AV-79.09" { S7_SetPoint := 'True'} : "Valve";
      "AV-79.10" { S7_SetPoint := 'True'} : "Valve";
      "AV-79.13" { S7_SetPoint := 'True'} : "Valve";
      "AV-79.14" { S7_SetPoint := 'True'} : "Valve";
      "AV-79.15" { S7_SetPoint := 'True'} : "Valve";
      "AV-79.16" { S7_SetPoint := 'True'} : "Valve";
      "AV-79.17" { S7_SetPoint := 'True'} : "Valve";
      "AV-81.01" { S7_SetPoint := 'True'} : "Valve";
      "AV-81.02" { S7_SetPoint := 'True'} : "Valve";
      "AV-81.03" { S7_SetPoint := 'True'} : "Valve";
      "AV-81.04" { S7_SetPoint := 'True'} : "Valve";
      "AV-81.05" { S7_SetPoint := 'True'} : "Valve";
      "AV-81.06" { S7_SetPoint := 'True'} : "Valve";
      "AV-81.07" { S7_SetPoint := 'True'} : "Valve";
      "AV-81.08" { S7_SetPoint := 'True'} : "Valve";
      "AV-81.09" { S7_SetPoint := 'True'} : "Valve";
      "AV-81.10" { S7_SetPoint := 'True'} : "Valve";
      "AV-81.12" { S7_SetPoint := 'True'} : "Valve";
      "AV-81.13" { S7_SetPoint := 'True'} : "Valve";
      "AV-81.14" { S7_SetPoint := 'True'} : "Valve";
      "AV-85.01" { S7_SetPoint := 'True'} : "Valve";
      "AV-85.02" { S7_SetPoint := 'True'} : "Valve";
      "AV-85.03" { S7_SetPoint := 'True'} : "Valve";
      "AV-85.04" { S7_SetPoint := 'True'} : "Valve";
      "AV-85.13" { S7_SetPoint := 'True'} : "Valve";
      "AV-85.12" { S7_SetPoint := 'True'} : "Valve";
      "AV-85.14" { S7_SetPoint := 'True'} : "Valve";
      "AV-85.15" { S7_SetPoint := 'True'} : "Valve";
      "AV-85.05" { S7_SetPoint := 'True'} : "Valve";
      "AV-85.06" { S7_SetPoint := 'True'} : "Valve";
      "AV-85.16" { S7_SetPoint := 'True'} : "Valve";
      "AV-85.17" { S7_SetPoint := 'True'} : "Valve";
      "AV-85.18" { S7_SetPoint := 'True'} : "Valve";
      "AV-85.09" { S7_SetPoint := 'True'} : "Valve";
      "AV-85.08" { S7_SetPoint := 'True'} : "Valve";
      "AV-85.10" { S7_SetPoint := 'True'} : "Valve";
      "AV-85.11" { S7_SetPoint := 'True'} : "Valve";
      "AV-84.05" { S7_SetPoint := 'True'} : "Valve";
      "AV-84.06" { S7_SetPoint := 'True'} : "Valve";
      "AV-84.07" { S7_SetPoint := 'True'} : "Valve";
      "AV-84.08" { S7_SetPoint := 'True'} : "Valve";
      "AV-84.09" { S7_SetPoint := 'True'} : "Valve";
      "AV-84.10" { S7_SetPoint := 'True'} : "Valve";
      "AV-84.12" { S7_SetPoint := 'True'} : "Valve";
      "AV-84.13" { S7_SetPoint := 'True'} : "Valve";
      "AV-84.14" { S7_SetPoint := 'True'} : "Valve";
      "AV-24.09" { S7_SetPoint := 'True'} : "Valve";
      "AV-24.17" { S7_SetPoint := 'True'} : "Valve";
      "AV-24.18" { S7_SetPoint := 'True'} : "Valve";
      "AV-24.19" { S7_SetPoint := 'True'} : "Valve";
      "AV-24.20" { S7_SetPoint := 'True'} : "Valve";
      "AV-24.21" { S7_SetPoint := 'True'} : "Valve";
      "AV-24.22" { S7_SetPoint := 'True'} : "Valve";
      "AV-24.23" { S7_SetPoint := 'True'} : "Valve";
      "AV-24.24" { S7_SetPoint := 'True'} : "Valve";
      "AV-79.21" { S7_SetPoint := 'True'} : "Valve";
      "AV-79.18" { S7_SetPoint := 'True'} : "Valve";
      "AV-79.19" { S7_SetPoint := 'True'} : "Valve";
      "AV-79.20" { S7_SetPoint := 'True'} : "Valve";
   END_VAR
BEGIN

REGION Network 1: AV-23.01
